REGION Network 63: CONTADOR DE SEGURIDAD DE PRESENCIA - CNTSeg_pHsMx
   RUNG wire#powerrail
      #CNTSeg_pHsMx(IN := wire#w4, R := wire#w7, PV := #V_CNTSeg_pHsMx, BaseUnidades_ms := "CTE_BaseUnidades_1ms", QU =>, QD =>, CVU =>, CVD =>)
   END_RUNG
   RUNG wire#powerrail
      Contact( #Mx_ET10 )
      wire#w1
      Contact( #MAnt_DescargaAct )
      wire#w3
      Contact( #Avance_TR1 )
   END_RUNG wire#w4
   RUNG wire#powerrail
      Contact( #Mx_ET16 )
      wire#w2
      Contact( "ON" )
   END_RUNG wire#w1
   RUNG wire#powerrail
      Contact( #Mx_ET17 )
   END_RUNG wire#w2
   RUNG wire#powerrail
      Contact( #Mx_ET02 )
   END_RUNG wire#w2
   RUNG wire#powerrail
      Contact( #Mx_ET11 )
   END_RUNG wire#w3
   RUNG wire#powerrail
      Contact( #Mx_ET12 )
   END_RUNG wire#w3
   RUNG wire#powerrail
      I_Contact( #Mx_ET10 )
      wire#w5
      I_Contact( #Mx_ET11 )
      I_Contact( #Mx_ET12 )
      wire#w6
      I_Contact( #Mx_ET16 )
      I_Contact( #Mx_ET17 )
      I_Contact( #Mx_ET02 )
   END_RUNG wire#w7
   RUNG wire#powerrail
      I_Contact( #MAnt_DescargaAct )
   END_RUNG wire#w5
   RUNG wire#w6
      I_Contact( #MAnt_DescargaAct )
   END_RUNG wire#w7
   // the same network as SCL:
   #CNTSeg_pHsMx(IN := (((#Mx_ET10 OR ((#Mx_ET16 OR #Mx_ET17 OR #Mx_ET02) AND "ON")) AND #MAnt_DescargaAct) OR #Mx_ET11 OR #Mx_ET12) AND #Avance_TR1,   // "FB910_CNT_UHS"
                 R := (NOT #Mx_ET10 OR NOT #MAnt_DescargaAct) AND NOT #Mx_ET11 AND NOT #Mx_ET12 AND ((NOT #Mx_ET16 AND NOT #Mx_ET17 AND NOT #Mx_ET02) OR NOT #MAnt_DescargaAct),
                 PV := #V_CNTSeg_pHsMx,
                 BaseUnidades_ms := "CTE_BaseUnidades_1ms");
END_REGION

REGION Network 64: CONTADOR DE PRESENCIA - CNT_pHsMx
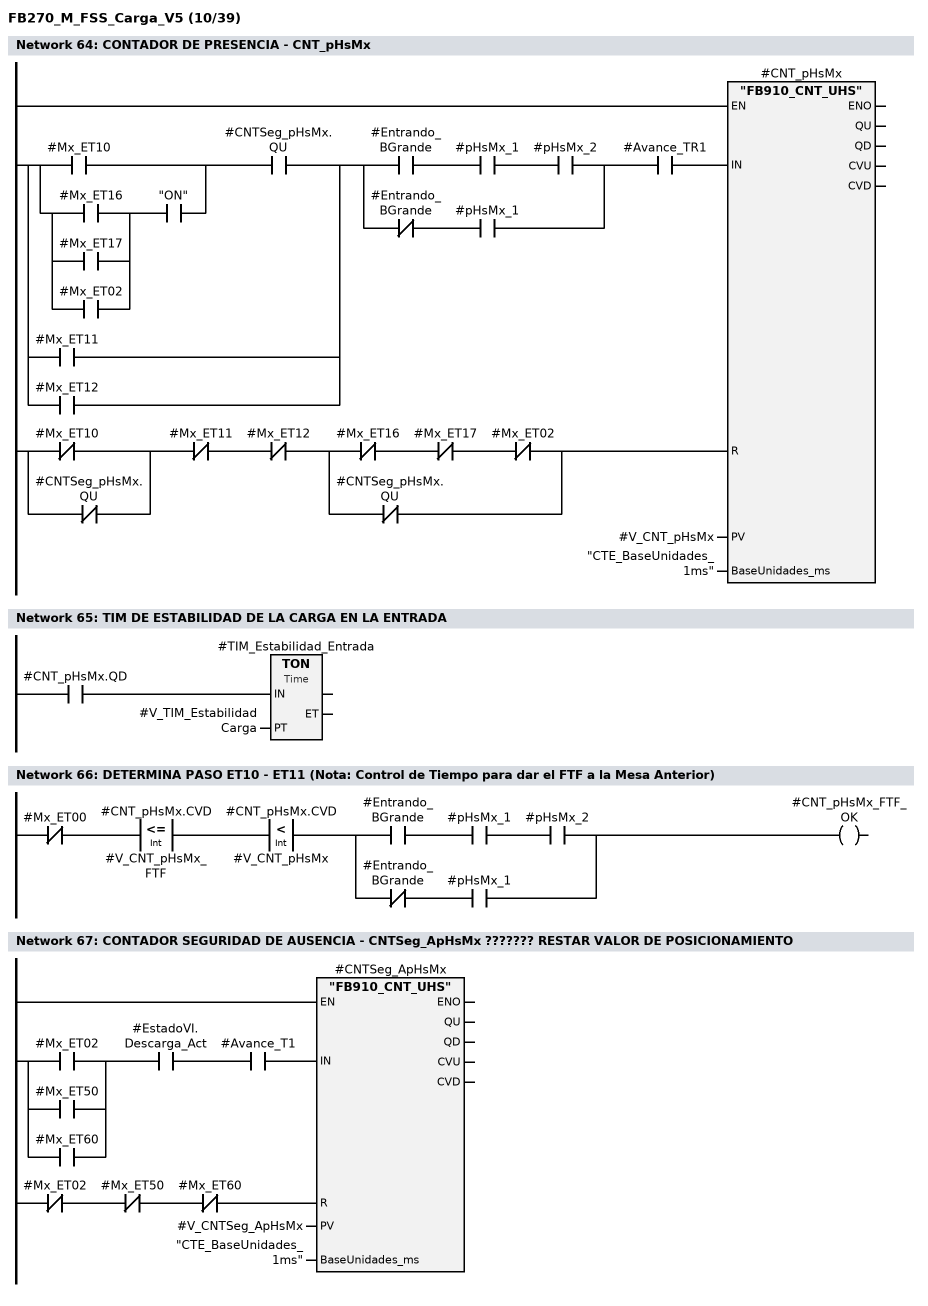
   RUNG wire#powerrail
      #CNT_pHsMx(IN := wire#w5, R := wire#w8, PV := #V_CNT_pHsMx, BaseUnidades_ms := "CTE_BaseUnidades_1ms", QU =>, QD =>, CVU =>, CVD =>)
   END_RUNG
   RUNG wire#powerrail
      Contact( #Mx_ET10 )
      wire#w1
      Contact( #CNTSeg_pHsMx.QU )
      wire#w3
      Contact( #Entrando_BGrande )
      Contact( #pHsMx_1 )
      Contact( #pHsMx_2 )
      wire#w4
      Contact( #Avance_TR1 )
   END_RUNG wire#w5
   RUNG wire#powerrail
      Contact( #Mx_ET16 )
      wire#w2
      Contact( "ON" )
   END_RUNG wire#w1
   RUNG wire#powerrail
      Contact( #Mx_ET17 )
   END_RUNG wire#w2
   RUNG wire#powerrail
      Contact( #Mx_ET02 )
   END_RUNG wire#w2
   RUNG wire#powerrail
      Contact( #Mx_ET11 )
   END_RUNG wire#w3
   RUNG wire#powerrail
      Contact( #Mx_ET12 )
   END_RUNG wire#w3
   RUNG wire#w3
      I_Contact( #Entrando_BGrande )
      Contact( #pHsMx_1 )
   END_RUNG wire#w4
   RUNG wire#powerrail
      I_Contact( #Mx_ET10 )
      wire#w6
      I_Contact( #Mx_ET11 )
      I_Contact( #Mx_ET12 )
      wire#w7
      I_Contact( #Mx_ET16 )
      I_Contact( #Mx_ET17 )
      I_Contact( #Mx_ET02 )
   END_RUNG wire#w8
   RUNG wire#powerrail
      I_Contact( #CNTSeg_pHsMx.QU )
   END_RUNG wire#w6
   RUNG wire#w7
      I_Contact( #CNTSeg_pHsMx.QU )
   END_RUNG wire#w8
   // the same network as SCL:
   #CNT_pHsMx(IN := (((#Mx_ET10 OR ((#Mx_ET16 OR #Mx_ET17 OR #Mx_ET02) AND "ON")) AND #CNTSeg_pHsMx.QU) OR #Mx_ET11 OR #Mx_ET12) AND ((#Entrando_BGrande AND #pHsMx_1 AND #pHsMx_2) OR (NOT #Entrando_BGrande AND #pHsMx_1)) AND #Avance_TR1,   // "FB910_CNT_UHS"
              R := (NOT #Mx_ET10 OR NOT #CNTSeg_pHsMx.QU) AND NOT #Mx_ET11 AND NOT #Mx_ET12 AND ((NOT #Mx_ET16 AND NOT #Mx_ET17 AND NOT #Mx_ET02) OR NOT #CNTSeg_pHsMx.QU),
              PV := #V_CNT_pHsMx,
              BaseUnidades_ms := "CTE_BaseUnidades_1ms");
END_REGION

REGION Network 65: TIM DE ESTABILIDAD DE LA CARGA EN LA ENTRADA
   RUNG wire#powerrail
      Contact( #CNT_pHsMx.QD )
      { S7_Templates := "time_type := Time" } #TIM_Estabilidad_Entrada.TON(pt := #V_TIM_EstabilidadCarga, et =>)
   END_RUNG
   // the same network as SCL:
   #TIM_Estabilidad_Entrada(IN := #CNT_pHsMx.QD, PT := #V_TIM_EstabilidadCarga);   // TON
END_REGION

REGION Network 66: DETERMINA PASO ET10 - ET11 (Nota: Control de Tiempo para dar el FTF a la Mesa Anterior)
   RUNG wire#powerrail
      I_Contact( #Mx_ET00 )
      { S7_Templates := "SrcType := Int" } LE_Contact(in1 := #CNT_pHsMx.CVD, in2 := #V_CNT_pHsMx_FTF)
      { S7_Templates := "SrcType := Int" } LT_Contact(in1 := #CNT_pHsMx.CVD, in2 := #V_CNT_pHsMx)
      wire#w1
      Contact( #Entrando_BGrande )
      Contact( #pHsMx_1 )
      Contact( #pHsMx_2 )
      wire#w2
      Coil( #CNT_pHsMx_FTF_OK )
   END_RUNG
   RUNG wire#w1
      I_Contact( #Entrando_BGrande )
      Contact( #pHsMx_1 )
   END_RUNG wire#w2
   // the same network as SCL:
   #CNT_pHsMx_FTF_OK := NOT #Mx_ET00 AND (#CNT_pHsMx.CVD <= #V_CNT_pHsMx_FTF) AND (#CNT_pHsMx.CVD < #V_CNT_pHsMx) AND ((#Entrando_BGrande AND #pHsMx_1 AND #pHsMx_2) OR (NOT #Entrando_BGrande AND #pHsMx_1));
END_REGION

REGION Network 67: CONTADOR SEGURIDAD DE AUSENCIA - CNTSeg_ApHsMx ??????? RESTAR VALOR DE POSICIONAMIENTO
   RUNG wire#powerrail
      #CNTSeg_ApHsMx(IN := wire#w2, R := wire#w3, PV := #V_CNTSeg_ApHsMx, BaseUnidades_ms := "CTE_BaseUnidades_1ms", QU =>, QD =>, CVU =>, CVD =>)
   END_RUNG
   RUNG wire#powerrail
      Contact( #Mx_ET02 )
      wire#w1
      Contact( #EstadoVI.Descarga_Act )
      Contact( #Avance_T1 )
   END_RUNG wire#w2
   RUNG wire#powerrail
      Contact( #Mx_ET50 )
   END_RUNG wire#w1
   RUNG wire#powerrail
      Contact( #Mx_ET60 )
   END_RUNG wire#w1
   RUNG wire#powerrail
      I_Contact( #Mx_ET02 )
      I_Contact( #Mx_ET50 )
      I_Contact( #Mx_ET60 )
   END_RUNG wire#w3
   // the same network as SCL:
   #CNTSeg_ApHsMx(IN := (#Mx_ET02 OR #Mx_ET50 OR #Mx_ET60) AND #EstadoVI.Descarga_Act AND #Avance_T1,   // "FB910_CNT_UHS"
                  R := NOT #Mx_ET02 AND NOT #Mx_ET50 AND NOT #Mx_ET60,
                  PV := #V_CNTSeg_ApHsMx,
                  BaseUnidades_ms := "CTE_BaseUnidades_1ms");
END_REGION

REGION Network 68: CONTADOR DE LA AUSENCIA - CNT_ApHsMX
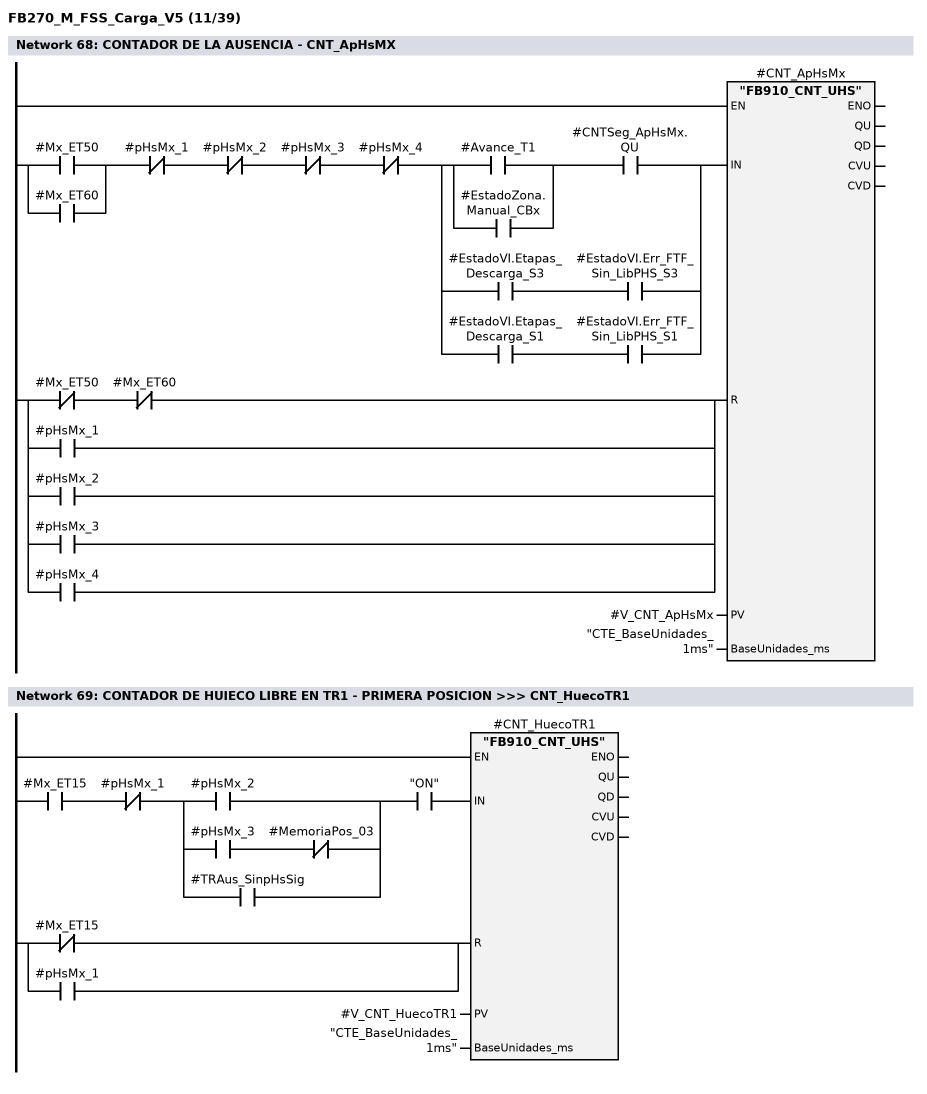
   RUNG wire#powerrail
      #CNT_ApHsMx(IN := wire#w4, R := wire#w5, PV := #V_CNT_ApHsMx, BaseUnidades_ms := "CTE_BaseUnidades_1ms", QU =>, QD =>, CVU =>, CVD =>)
   END_RUNG
   RUNG wire#powerrail
      Contact( #Mx_ET50 )
      wire#w1
      I_Contact( #pHsMx_1 )
      I_Contact( #pHsMx_2 )
      I_Contact( #pHsMx_3 )
      I_Contact( #pHsMx_4 )
      wire#w2
      Contact( #Avance_T1 )
      wire#w3
      Contact( #CNTSeg_ApHsMx.QU )
   END_RUNG wire#w4
   RUNG wire#powerrail
      Contact( #Mx_ET60 )
   END_RUNG wire#w1
   RUNG wire#w2
      Contact( #EstadoZona.Manual_CBx )
   END_RUNG wire#w3
   RUNG wire#w2
      Contact( #EstadoVI.Etapas_Descarga_S3 )
      Contact( #EstadoVI.Err_FTF_Sin_LibPHS_S3 )
   END_RUNG wire#w4
   RUNG wire#w2
      Contact( #EstadoVI.Etapas_Descarga_S1 )
      Contact( #EstadoVI.Err_FTF_Sin_LibPHS_S1 )
   END_RUNG wire#w4
   RUNG wire#powerrail
      I_Contact( #Mx_ET50 )
      I_Contact( #Mx_ET60 )
   END_RUNG wire#w5
   RUNG wire#powerrail
      Contact( #pHsMx_1 )
   END_RUNG wire#w5
   RUNG wire#powerrail
      Contact( #pHsMx_2 )
   END_RUNG wire#w5
   RUNG wire#powerrail
      Contact( #pHsMx_3 )
   END_RUNG wire#w5
   RUNG wire#powerrail
      Contact( #pHsMx_4 )
   END_RUNG wire#w5
   // the same network as SCL:
   #CNT_ApHsMx(IN := (#Mx_ET50 OR #Mx_ET60) AND NOT #pHsMx_1 AND NOT #pHsMx_2 AND NOT #pHsMx_3 AND NOT #pHsMx_4 AND (((#Avance_T1 OR #EstadoZona.Manual_CBx) AND #CNTSeg_ApHsMx.QU) OR (#EstadoVI.Etapas_Descarga_S3 AND #EstadoVI.Err_FTF_Sin_LibPHS_S3) OR (#EstadoVI.Etapas_Descarga_S1 AND #EstadoVI.Err_FTF_Sin_LibPHS_S1)),   // "FB910_CNT_UHS"
               R := (NOT #Mx_ET50 AND NOT #Mx_ET60) OR #pHsMx_1 OR #pHsMx_2 OR #pHsMx_3 OR #pHsMx_4,
               PV := #V_CNT_ApHsMx,
               BaseUnidades_ms := "CTE_BaseUnidades_1ms");
END_REGION

REGION Network 69: CONTADOR DE HUIECO LIBRE EN TR1 - PRIMERA POSICION >>> CNT_HuecoTR1
   RUNG wire#powerrail
      #CNT_HuecoTR1(IN := wire#w3, R := wire#w4, PV := #V_CNT_HuecoTR1, BaseUnidades_ms := "CTE_BaseUnidades_1ms", QU =>, QD =>, CVU =>, CVD =>)
   END_RUNG
   RUNG wire#powerrail
      Contact( #Mx_ET15 )
      I_Contact( #pHsMx_1 )
      wire#w1
      Contact( #pHsMx_2 )
      wire#w2
      Contact( "ON" )
   END_RUNG wire#w3
   RUNG wire#w1
      Contact( #pHsMx_3 )
      I_Contact( #MemoriaPos_03 )
   END_RUNG wire#w2
   RUNG wire#w1
      Contact( #TRAus_SinpHsSig )
   END_RUNG wire#w2
   RUNG wire#powerrail
      I_Contact( #Mx_ET15 )
   END_RUNG wire#w4
   RUNG wire#powerrail
      Contact( #pHsMx_1 )
   END_RUNG wire#w4
   // the same network as SCL:
   #CNT_HuecoTR1(IN := #Mx_ET15 AND NOT #pHsMx_1 AND (#pHsMx_2 OR (#pHsMx_3 AND NOT #MemoriaPos_03) OR #TRAus_SinpHsSig) AND "ON",   // "FB910_CNT_UHS"
                 R := NOT #Mx_ET15 OR #pHsMx_1,
                 PV := #V_CNT_HuecoTR1,
                 BaseUnidades_ms := "CTE_BaseUnidades_1ms");
END_REGION

REGION Network 70: CONTADOR DE HUIECO LIBRE EN TR2 - SEGUNDA POSICION >>> CNT_HuecoTR2
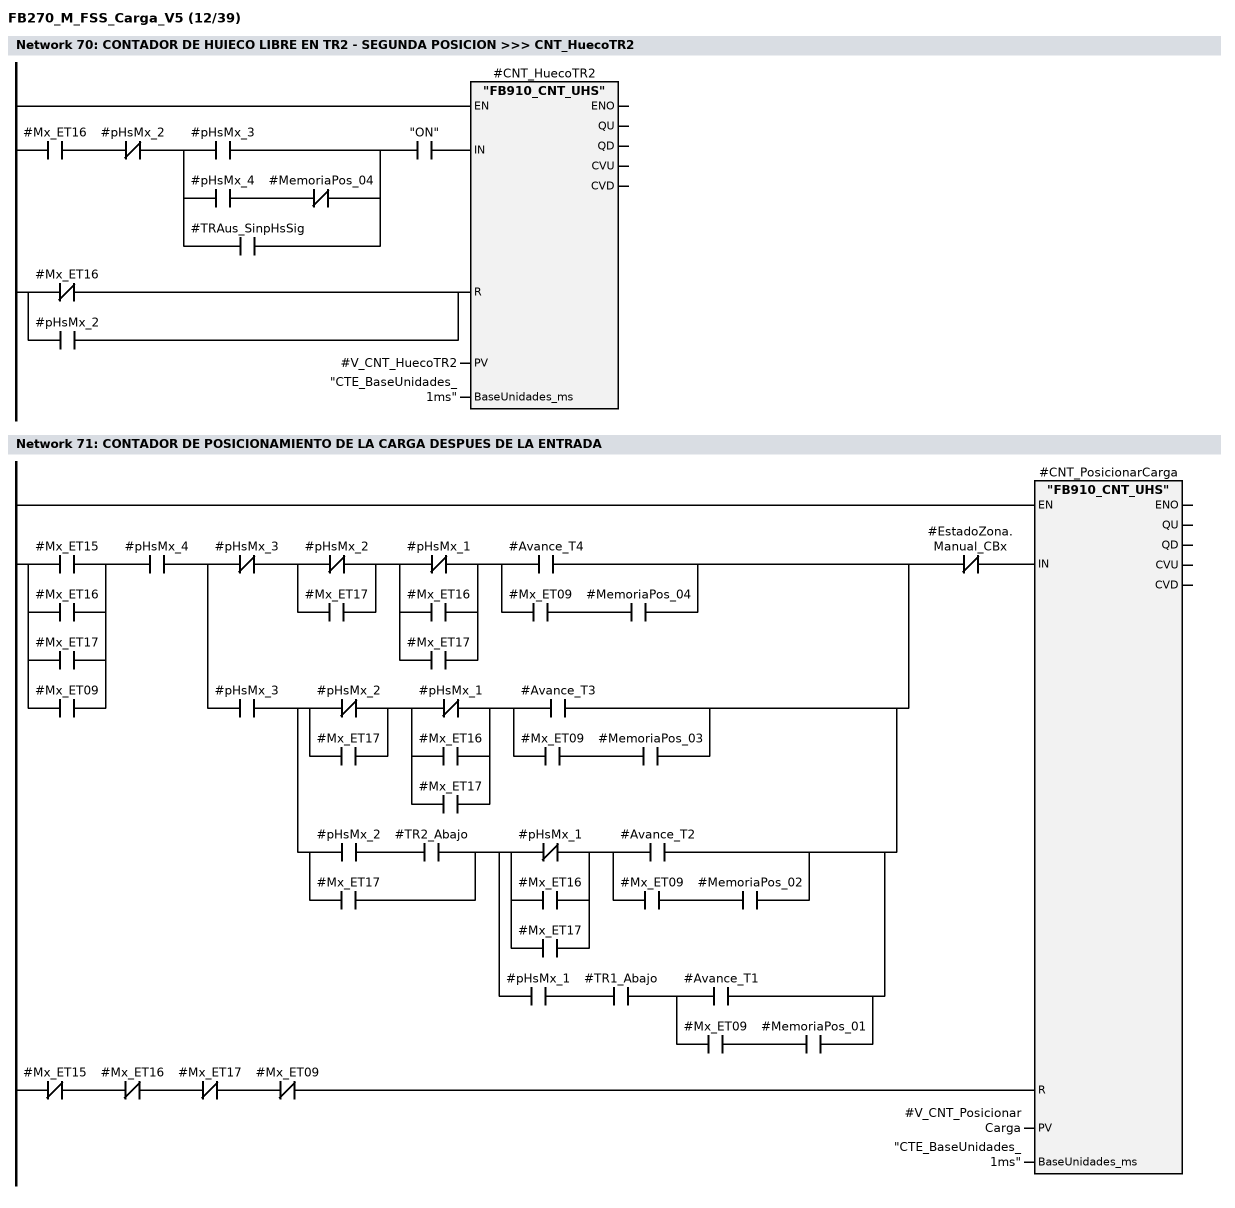
   RUNG wire#powerrail
      #CNT_HuecoTR2(IN := wire#w3, R := wire#w4, PV := #V_CNT_HuecoTR2, BaseUnidades_ms := "CTE_BaseUnidades_1ms", QU =>, QD =>, CVU =>, CVD =>)
   END_RUNG
   RUNG wire#powerrail
      Contact( #Mx_ET16 )
      I_Contact( #pHsMx_2 )
      wire#w1
      Contact( #pHsMx_3 )
      wire#w2
      Contact( "ON" )
   END_RUNG wire#w3
   RUNG wire#w1
      Contact( #pHsMx_4 )
      I_Contact( #MemoriaPos_04 )
   END_RUNG wire#w2
   RUNG wire#w1
      Contact( #TRAus_SinpHsSig )
   END_RUNG wire#w2
   RUNG wire#powerrail
      I_Contact( #Mx_ET16 )
   END_RUNG wire#w4
   RUNG wire#powerrail
      Contact( #pHsMx_2 )
   END_RUNG wire#w4
   // the same network as SCL:
   #CNT_HuecoTR2(IN := #Mx_ET16 AND NOT #pHsMx_2 AND (#pHsMx_3 OR (#pHsMx_4 AND NOT #MemoriaPos_04) OR #TRAus_SinpHsSig) AND "ON",   // "FB910_CNT_UHS"
                 R := NOT #Mx_ET16 OR #pHsMx_2,
                 PV := #V_CNT_HuecoTR2,
                 BaseUnidades_ms := "CTE_BaseUnidades_1ms");
END_REGION

REGION Network 71: CONTADOR DE POSICIONAMIENTO DE LA CARGA DESPUES DE LA ENTRADA
   RUNG wire#powerrail
      #CNT_PosicionarCarga(IN := wire#w13, R := wire#w14, PV := #V_CNT_PosicionarCarga, BaseUnidades_ms := "CTE_BaseUnidades_1ms", QU =>, QD =>, CVU =>, CVD =>)
   END_RUNG
   RUNG wire#powerrail
      Contact( #Mx_ET15 )
      wire#w1
      Contact( #pHsMx_4 )
      wire#w2
      I_Contact( #pHsMx_3 )
      wire#w3
      I_Contact( #pHsMx_2 )
      wire#w4
      I_Contact( #pHsMx_1 )
      wire#w5
      Contact( #Avance_T4 )
      wire#w6
      I_Contact( #EstadoZona.Manual_CBx )
   END_RUNG wire#w13
   RUNG wire#powerrail
      Contact( #Mx_ET16 )
   END_RUNG wire#w1
   RUNG wire#powerrail
      Contact( #Mx_ET17 )
   END_RUNG wire#w1
   RUNG wire#powerrail
      Contact( #Mx_ET09 )
   END_RUNG wire#w1
   RUNG wire#w3
      Contact( #Mx_ET17 )
   END_RUNG wire#w4
   RUNG wire#w4
      Contact( #Mx_ET16 )
   END_RUNG wire#w5
   RUNG wire#w4
      Contact( #Mx_ET17 )
   END_RUNG wire#w5
   RUNG wire#w5
      Contact( #Mx_ET09 )
      Contact( #MemoriaPos_04 )
   END_RUNG wire#w6
   RUNG wire#w2
      Contact( #pHsMx_3 )
      wire#w7
      I_Contact( #pHsMx_2 )
      wire#w8
      I_Contact( #pHsMx_1 )
      wire#w9
      Contact( #Avance_T3 )
   END_RUNG wire#w6
   RUNG wire#w7
      Contact( #Mx_ET17 )
   END_RUNG wire#w8
   RUNG wire#w8
      Contact( #Mx_ET16 )
   END_RUNG wire#w9
   RUNG wire#w8
      Contact( #Mx_ET17 )
   END_RUNG wire#w9
   RUNG wire#w9
      Contact( #Mx_ET09 )
      Contact( #MemoriaPos_03 )
   END_RUNG wire#w6
   RUNG wire#w7
      Contact( #pHsMx_2 )
      Contact( #TR2_Abajo )
      wire#w10
      I_Contact( #pHsMx_1 )
      wire#w11
      Contact( #Avance_T2 )
   END_RUNG wire#w6
   RUNG wire#w7
      Contact( #Mx_ET17 )
   END_RUNG wire#w10
   RUNG wire#w10
      Contact( #Mx_ET16 )
   END_RUNG wire#w11
   RUNG wire#w10
      Contact( #Mx_ET17 )
   END_RUNG wire#w11
   RUNG wire#w11
      Contact( #Mx_ET09 )
      Contact( #MemoriaPos_02 )
   END_RUNG wire#w6
   RUNG wire#w10
      Contact( #pHsMx_1 )
      Contact( #TR1_Abajo )
      wire#w12
      Contact( #Avance_T1 )
   END_RUNG wire#w6
   RUNG wire#w12
      Contact( #Mx_ET09 )
      Contact( #MemoriaPos_01 )
   END_RUNG wire#w6
   RUNG wire#powerrail
      I_Contact( #Mx_ET15 )
      I_Contact( #Mx_ET16 )
      I_Contact( #Mx_ET17 )
      I_Contact( #Mx_ET09 )
   END_RUNG wire#w14
   // the same network as SCL:
   #CNT_PosicionarCarga(IN := (#Mx_ET15 OR #Mx_ET16 OR #Mx_ET17 OR #Mx_ET09) AND #pHsMx_4 AND ((NOT #pHsMx_3 AND (NOT #pHsMx_2 OR #Mx_ET17) AND (NOT #pHsMx_1 OR #Mx_ET16 OR #Mx_ET17) AND (#Avance_T4 OR (#Mx_ET09 AND #MemoriaPos_04))) OR (#pHsMx_3 AND (((NOT #pHsMx_2 OR #Mx_ET17) AND (NOT #pHsMx_1 OR #Mx_ET16 OR #Mx_ET17) AND (#Avance_T3 OR (#Mx_ET09 AND #MemoriaPos_03))) OR (((#pHsMx_2 AND #TR2_Abajo) OR #Mx_ET17) AND (((NOT #pHsMx_1 OR #Mx_ET16 OR #Mx_ET17) AND (#Avance_T2 OR (#Mx_ET09 AND #MemoriaPos_02))) OR (#pHsMx_1 AND #TR1_Abajo AND (#Avance_T1 OR (#Mx_ET09 AND #MemoriaPos_01)))))))) AND NOT #EstadoZona.Manual_CBx,   // "FB910_CNT_UHS"
                        R := NOT #Mx_ET15 AND NOT #Mx_ET16 AND NOT #Mx_ET17 AND NOT #Mx_ET09,
                        PV := #V_CNT_PosicionarCarga,
                        BaseUnidades_ms := "CTE_BaseUnidades_1ms");
END_REGION

REGION Network 72: CONTADOR DE PREPARACION DE CARGA PARA SALIDA POR S1
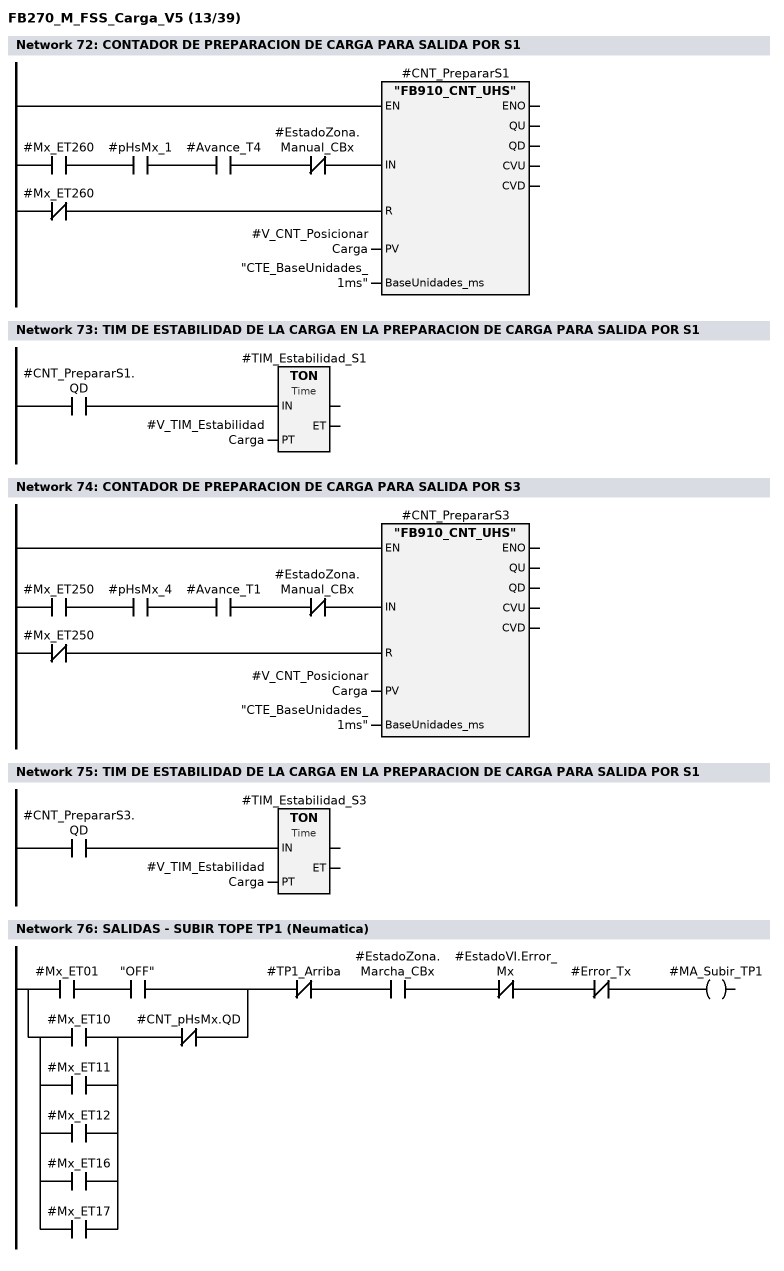
   RUNG wire#powerrail
      #CNT_PrepararS1(IN := wire#w1, R := wire#w2, PV := #V_CNT_PosicionarCarga, BaseUnidades_ms := "CTE_BaseUnidades_1ms", QU =>, QD =>, CVU =>, CVD =>)
   END_RUNG
   RUNG wire#powerrail
      Contact( #Mx_ET260 )
      Contact( #pHsMx_1 )
      Contact( #Avance_T4 )
      I_Contact( #EstadoZona.Manual_CBx )
   END_RUNG wire#w1
   RUNG wire#powerrail
      I_Contact( #Mx_ET260 )
   END_RUNG wire#w2
   // the same network as SCL:
   #CNT_PrepararS1(IN := #Mx_ET260 AND #pHsMx_1 AND #Avance_T4 AND NOT #EstadoZona.Manual_CBx,   // "FB910_CNT_UHS"
                   R := NOT #Mx_ET260,
                   PV := #V_CNT_PosicionarCarga,
                   BaseUnidades_ms := "CTE_BaseUnidades_1ms");
END_REGION

REGION Network 73: TIM DE ESTABILIDAD DE LA CARGA EN LA PREPARACION DE CARGA PARA SALIDA POR S1
   RUNG wire#powerrail
      Contact( #CNT_PrepararS1.QD )
      { S7_Templates := "time_type := Time" } #TIM_Estabilidad_S1.TON(pt := #V_TIM_EstabilidadCarga, et =>)
   END_RUNG
   // the same network as SCL:
   #TIM_Estabilidad_S1(IN := #CNT_PrepararS1.QD, PT := #V_TIM_EstabilidadCarga);   // TON
END_REGION

REGION Network 74: CONTADOR DE PREPARACION DE CARGA PARA SALIDA POR S3
   RUNG wire#powerrail
      #CNT_PrepararS3(IN := wire#w1, R := wire#w2, PV := #V_CNT_PosicionarCarga, BaseUnidades_ms := "CTE_BaseUnidades_1ms", QU =>, QD =>, CVU =>, CVD =>)
   END_RUNG
   RUNG wire#powerrail
      Contact( #Mx_ET250 )
      Contact( #pHsMx_4 )
      Contact( #Avance_T1 )
      I_Contact( #EstadoZona.Manual_CBx )
   END_RUNG wire#w1
   RUNG wire#powerrail
      I_Contact( #Mx_ET250 )
   END_RUNG wire#w2
   // the same network as SCL:
   #CNT_PrepararS3(IN := #Mx_ET250 AND #pHsMx_4 AND #Avance_T1 AND NOT #EstadoZona.Manual_CBx,   // "FB910_CNT_UHS"
                   R := NOT #Mx_ET250,
                   PV := #V_CNT_PosicionarCarga,
                   BaseUnidades_ms := "CTE_BaseUnidades_1ms");
END_REGION

REGION Network 75: TIM DE ESTABILIDAD DE LA CARGA EN LA PREPARACION DE CARGA PARA SALIDA POR S1
   RUNG wire#powerrail
      Contact( #CNT_PrepararS3.QD )
      { S7_Templates := "time_type := Time" } #TIM_Estabilidad_S3.TON(pt := #V_TIM_EstabilidadCarga, et =>)
   END_RUNG
   // the same network as SCL:
   #TIM_Estabilidad_S3(IN := #CNT_PrepararS3.QD, PT := #V_TIM_EstabilidadCarga);   // TON
END_REGION

REGION Network 76: SALIDAS - SUBIR TOPE TP1 (Neumatica)
   RUNG wire#powerrail
      Contact( #Mx_ET01 )
      Contact( "OFF" )
      wire#w1
      I_Contact( #TP1_Arriba )
      Contact( #EstadoZona.Marcha_CBx )
      I_Contact( #EstadoVI.Error_Mx )
      I_Contact( #Error_Tx )
      Coil( #MA_Subir_TP1 )
   END_RUNG
   RUNG wire#powerrail
      Contact( #Mx_ET10 )
      wire#w2
      I_Contact( #CNT_pHsMx.QD )
   END_RUNG wire#w1
   RUNG wire#powerrail
      Contact( #Mx_ET11 )
   END_RUNG wire#w2
   RUNG wire#powerrail
      Contact( #Mx_ET12 )
   END_RUNG wire#w2
   RUNG wire#powerrail
      Contact( #Mx_ET16 )
   END_RUNG wire#w2
   RUNG wire#powerrail
      Contact( #Mx_ET17 )
   END_RUNG wire#w2
   // the same network as SCL:
   #MA_Subir_TP1 := ((#Mx_ET01 AND "OFF") OR ((#Mx_ET10 OR #Mx_ET11 OR #Mx_ET12 OR #Mx_ET16 OR #Mx_ET17) AND NOT #CNT_pHsMx.QD)) AND NOT #TP1_Arriba AND #EstadoZona.Marcha_CBx AND NOT #EstadoVI.Error_Mx AND NOT #Error_Tx;
END_REGION

REGION Network 77: SALIDAS - BAJAR TOPE TP1 (Neumatica)
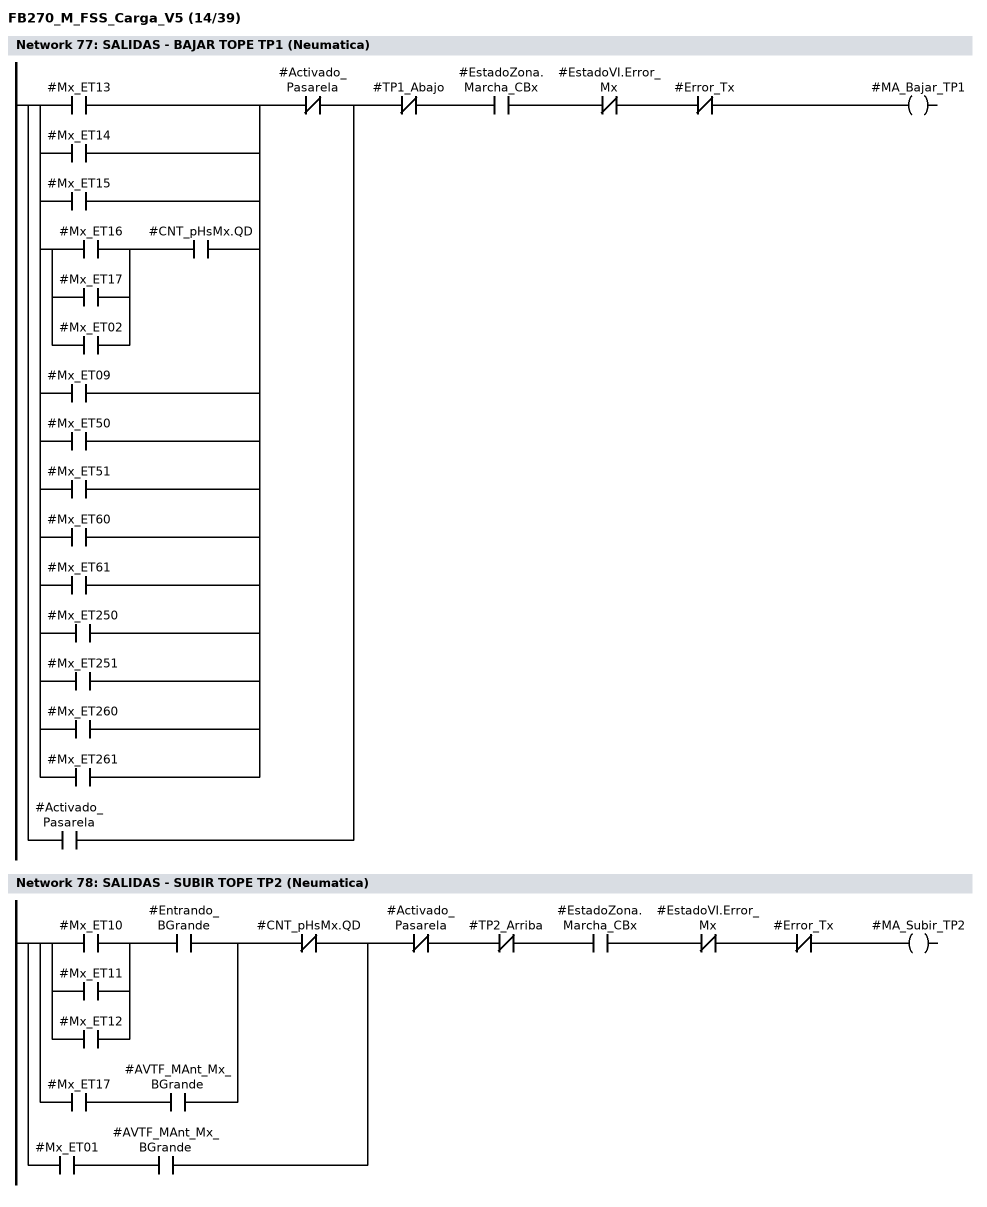
   RUNG wire#powerrail
      Contact( #Mx_ET13 )
      wire#w1
      I_Contact( #Activado_Pasarela )
      wire#w3
      I_Contact( #TP1_Abajo )
      Contact( #EstadoZona.Marcha_CBx )
      I_Contact( #EstadoVI.Error_Mx )
      I_Contact( #Error_Tx )
      Coil( #MA_Bajar_TP1 )
   END_RUNG
   RUNG wire#powerrail
      Contact( #Mx_ET14 )
   END_RUNG wire#w1
   RUNG wire#powerrail
      Contact( #Mx_ET15 )
   END_RUNG wire#w1
   RUNG wire#powerrail
      Contact( #Mx_ET16 )
      wire#w2
      Contact( #CNT_pHsMx.QD )
   END_RUNG wire#w1
   RUNG wire#powerrail
      Contact( #Mx_ET17 )
   END_RUNG wire#w2
   RUNG wire#powerrail
      Contact( #Mx_ET02 )
   END_RUNG wire#w2
   RUNG wire#powerrail
      Contact( #Mx_ET09 )
   END_RUNG wire#w1
   RUNG wire#powerrail
      Contact( #Mx_ET50 )
   END_RUNG wire#w1
   RUNG wire#powerrail
      Contact( #Mx_ET51 )
   END_RUNG wire#w1
   RUNG wire#powerrail
      Contact( #Mx_ET60 )
   END_RUNG wire#w1
   RUNG wire#powerrail
      Contact( #Mx_ET61 )
   END_RUNG wire#w1
   RUNG wire#powerrail
      Contact( #Mx_ET250 )
   END_RUNG wire#w1
   RUNG wire#powerrail
      Contact( #Mx_ET251 )
   END_RUNG wire#w1
   RUNG wire#powerrail
      Contact( #Mx_ET260 )
   END_RUNG wire#w1
   RUNG wire#powerrail
      Contact( #Mx_ET261 )
   END_RUNG wire#w1
   RUNG wire#powerrail
      Contact( #Activado_Pasarela )
   END_RUNG wire#w3
   // the same network as SCL:
   #MA_Bajar_TP1 := (((#Mx_ET13 OR #Mx_ET14 OR #Mx_ET15 OR ((#Mx_ET16 OR #Mx_ET17 OR #Mx_ET02) AND #CNT_pHsMx.QD) OR #Mx_ET09 OR #Mx_ET50 OR #Mx_ET51 OR #Mx_ET60 OR #Mx_ET61 OR #Mx_ET250 OR #Mx_ET251 OR #Mx_ET260 OR #Mx_ET261) AND NOT #Activado_Pasarela) OR #Activado_Pasarela) AND NOT #TP1_Abajo AND #EstadoZona.Marcha_CBx AND NOT #EstadoVI.Error_Mx AND NOT #Error_Tx;
END_REGION

REGION Network 78: SALIDAS - SUBIR TOPE TP2 (Neumatica)
   RUNG wire#powerrail
      Contact( #Mx_ET10 )
      wire#w1
      Contact( #Entrando_BGrande )
      wire#w2
      I_Contact( #CNT_pHsMx.QD )
      wire#w3
      I_Contact( #Activado_Pasarela )
      I_Contact( #TP2_Arriba )
      Contact( #EstadoZona.Marcha_CBx )
      I_Contact( #EstadoVI.Error_Mx )
      I_Contact( #Error_Tx )
      Coil( #MA_Subir_TP2 )
   END_RUNG
   RUNG wire#powerrail
      Contact( #Mx_ET11 )
   END_RUNG wire#w1
   RUNG wire#powerrail
      Contact( #Mx_ET12 )
   END_RUNG wire#w1
   RUNG wire#powerrail
      Contact( #Mx_ET17 )
      Contact( #AVTF_MAnt_Mx_BGrande )
   END_RUNG wire#w2
   RUNG wire#powerrail
      Contact( #Mx_ET01 )
      Contact( #AVTF_MAnt_Mx_BGrande )
   END_RUNG wire#w3
   // the same network as SCL:
   #MA_Subir_TP2 := (((((#Mx_ET10 OR #Mx_ET11 OR #Mx_ET12) AND #Entrando_BGrande) OR (#Mx_ET17 AND #AVTF_MAnt_Mx_BGrande)) AND NOT #CNT_pHsMx.QD) OR (#Mx_ET01 AND #AVTF_MAnt_Mx_BGrande)) AND NOT #Activado_Pasarela AND NOT #TP2_Arriba AND #EstadoZona.Marcha_CBx AND NOT #EstadoVI.Error_Mx AND NOT #Error_Tx;
END_REGION

REGION Network 79: SALIDAS - BAJAR TOPE TP2 (Neumatica)
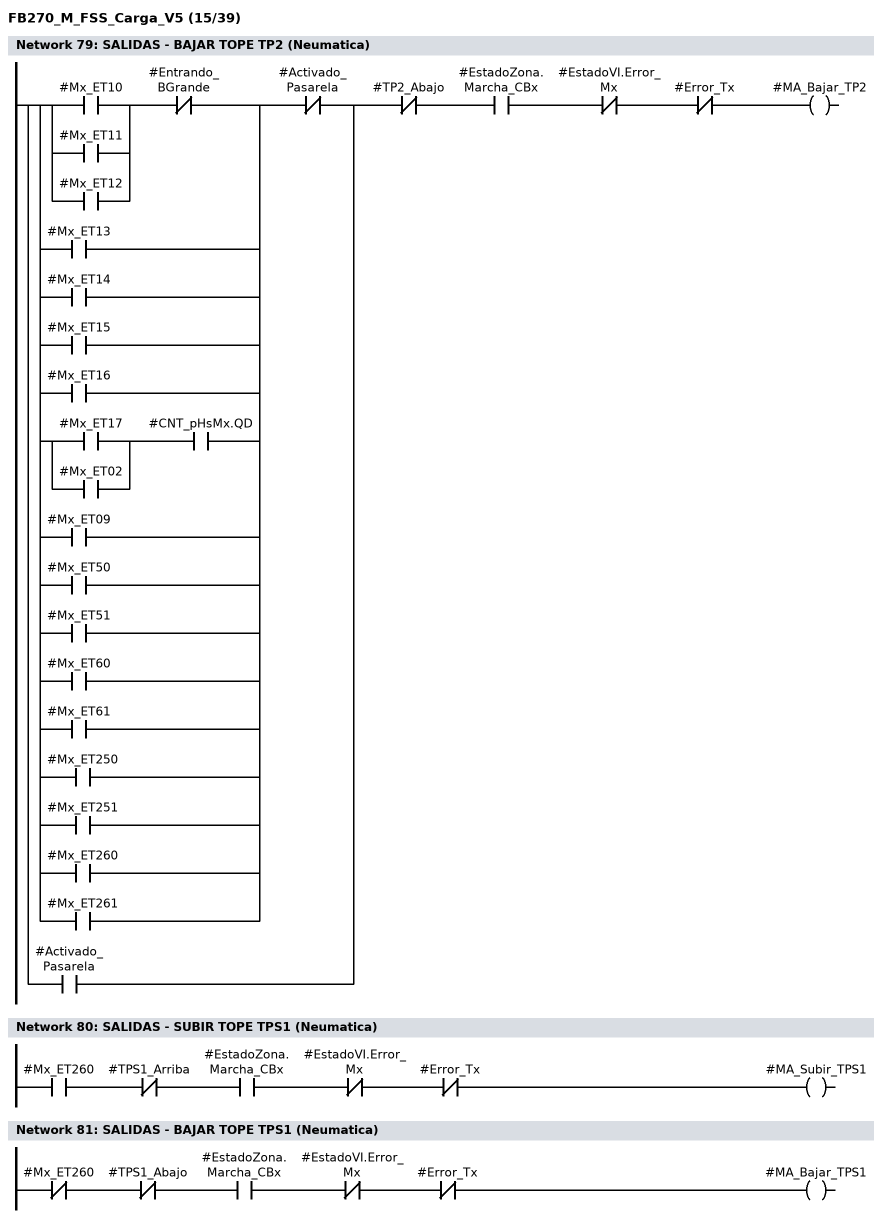
   RUNG wire#powerrail
      Contact( #Mx_ET10 )
      wire#w1
      I_Contact( #Entrando_BGrande )
      wire#w2
      I_Contact( #Activado_Pasarela )
      wire#w4
      I_Contact( #TP2_Abajo )
      Contact( #EstadoZona.Marcha_CBx )
      I_Contact( #EstadoVI.Error_Mx )
      I_Contact( #Error_Tx )
      Coil( #MA_Bajar_TP2 )
   END_RUNG
   RUNG wire#powerrail
      Contact( #Mx_ET11 )
   END_RUNG wire#w1
   RUNG wire#powerrail
      Contact( #Mx_ET12 )
   END_RUNG wire#w1
   RUNG wire#powerrail
      Contact( #Mx_ET13 )
   END_RUNG wire#w2
   RUNG wire#powerrail
      Contact( #Mx_ET14 )
   END_RUNG wire#w2
   RUNG wire#powerrail
      Contact( #Mx_ET15 )
   END_RUNG wire#w2
   RUNG wire#powerrail
      Contact( #Mx_ET16 )
   END_RUNG wire#w2
   RUNG wire#powerrail
      Contact( #Mx_ET17 )
      wire#w3
      Contact( #CNT_pHsMx.QD )
   END_RUNG wire#w2
   RUNG wire#powerrail
      Contact( #Mx_ET02 )
   END_RUNG wire#w3
   RUNG wire#powerrail
      Contact( #Mx_ET09 )
   END_RUNG wire#w2
   RUNG wire#powerrail
      Contact( #Mx_ET50 )
   END_RUNG wire#w2
   RUNG wire#powerrail
      Contact( #Mx_ET51 )
   END_RUNG wire#w2
   RUNG wire#powerrail
      Contact( #Mx_ET60 )
   END_RUNG wire#w2
   RUNG wire#powerrail
      Contact( #Mx_ET61 )
   END_RUNG wire#w2
   RUNG wire#powerrail
      Contact( #Mx_ET250 )
   END_RUNG wire#w2
   RUNG wire#powerrail
      Contact( #Mx_ET251 )
   END_RUNG wire#w2
   RUNG wire#powerrail
      Contact( #Mx_ET260 )
   END_RUNG wire#w2
   RUNG wire#powerrail
      Contact( #Mx_ET261 )
   END_RUNG wire#w2
   RUNG wire#powerrail
      Contact( #Activado_Pasarela )
   END_RUNG wire#w4
   // the same network as SCL:
   #MA_Bajar_TP2 := (((((#Mx_ET10 OR #Mx_ET11 OR #Mx_ET12) AND NOT #Entrando_BGrande) OR #Mx_ET13 OR #Mx_ET14 OR #Mx_ET15 OR #Mx_ET16 OR ((#Mx_ET17 OR #Mx_ET02) AND #CNT_pHsMx.QD) OR #Mx_ET09 OR #Mx_ET50 OR #Mx_ET51 OR #Mx_ET60 OR #Mx_ET61 OR #Mx_ET250 OR #Mx_ET251 OR #Mx_ET260 OR #Mx_ET261) AND NOT #Activado_Pasarela) OR #Activado_Pasarela) AND NOT #TP2_Abajo AND #EstadoZona.Marcha_CBx AND NOT #EstadoVI.Error_Mx AND NOT #Error_Tx;
END_REGION

REGION Network 80: SALIDAS - SUBIR TOPE TPS1 (Neumatica)
   RUNG wire#powerrail
      Contact( #Mx_ET260 )
      I_Contact( #TPS1_Arriba )
      Contact( #EstadoZona.Marcha_CBx )
      I_Contact( #EstadoVI.Error_Mx )
      I_Contact( #Error_Tx )
      Coil( #MA_Subir_TPS1 )
   END_RUNG
   // the same network as SCL:
   #MA_Subir_TPS1 := #Mx_ET260 AND NOT #TPS1_Arriba AND #EstadoZona.Marcha_CBx AND NOT #EstadoVI.Error_Mx AND NOT #Error_Tx;
END_REGION

REGION Network 81: SALIDAS - BAJAR TOPE TPS1 (Neumatica)
   RUNG wire#powerrail
      I_Contact( #Mx_ET260 )
      I_Contact( #TPS1_Abajo )
      Contact( #EstadoZona.Marcha_CBx )
      I_Contact( #EstadoVI.Error_Mx )
      I_Contact( #Error_Tx )
      Coil( #MA_Bajar_TPS1 )
   END_RUNG
   // the same network as SCL:
   #MA_Bajar_TPS1 := NOT #Mx_ET260 AND NOT #TPS1_Abajo AND #EstadoZona.Marcha_CBx AND NOT #EstadoVI.Error_Mx AND NOT #Error_Tx;
END_REGION

REGION Network 82: SALIDAS - SUBIR TOPE TPS3 (Neumatica)
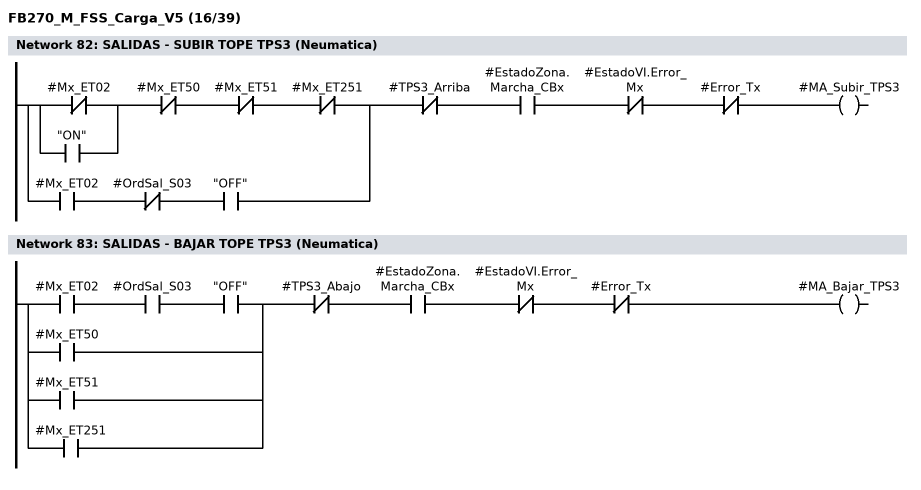
   RUNG wire#powerrail
      I_Contact( #Mx_ET02 )
      wire#w1
      I_Contact( #Mx_ET50 )
      I_Contact( #Mx_ET51 )
      I_Contact( #Mx_ET251 )
      wire#w2
      I_Contact( #TPS3_Arriba )
      Contact( #EstadoZona.Marcha_CBx )
      I_Contact( #EstadoVI.Error_Mx )
      I_Contact( #Error_Tx )
      Coil( #MA_Subir_TPS3 )
   END_RUNG
   RUNG wire#powerrail
      Contact( "ON" )
   END_RUNG wire#w1
   RUNG wire#powerrail
      Contact( #Mx_ET02 )
      I_Contact( #OrdSal_S03 )
      Contact( "OFF" )
   END_RUNG wire#w2
   // the same network as SCL:
   #MA_Subir_TPS3 := (((NOT #Mx_ET02 OR "ON") AND NOT #Mx_ET50 AND NOT #Mx_ET51 AND NOT #Mx_ET251) OR (#Mx_ET02 AND NOT #OrdSal_S03 AND "OFF")) AND NOT #TPS3_Arriba AND #EstadoZona.Marcha_CBx AND NOT #EstadoVI.Error_Mx AND NOT #Error_Tx;
END_REGION

REGION Network 83: SALIDAS - BAJAR TOPE TPS3 (Neumatica)
   RUNG wire#powerrail
      Contact( #Mx_ET02 )
      Contact( #OrdSal_S03 )
      Contact( "OFF" )
      wire#w1
      I_Contact( #TPS3_Abajo )
      Contact( #EstadoZona.Marcha_CBx )
      I_Contact( #EstadoVI.Error_Mx )
      I_Contact( #Error_Tx )
      Coil( #MA_Bajar_TPS3 )
   END_RUNG
   RUNG wire#powerrail
      Contact( #Mx_ET50 )
   END_RUNG wire#w1
   RUNG wire#powerrail
      Contact( #Mx_ET51 )
   END_RUNG wire#w1
   RUNG wire#powerrail
      Contact( #Mx_ET251 )
   END_RUNG wire#w1
   // the same network as SCL:
   #MA_Bajar_TPS3 := ((#Mx_ET02 AND #OrdSal_S03 AND "OFF") OR #Mx_ET50 OR #Mx_ET51 OR #Mx_ET251) AND NOT #TPS3_Abajo AND #EstadoZona.Marcha_CBx AND NOT #EstadoVI.Error_Mx AND NOT #Error_Tx;
END_REGION

REGION Network 84: VARIABLES AUXILIARES - Posición Correcta de los Transfers
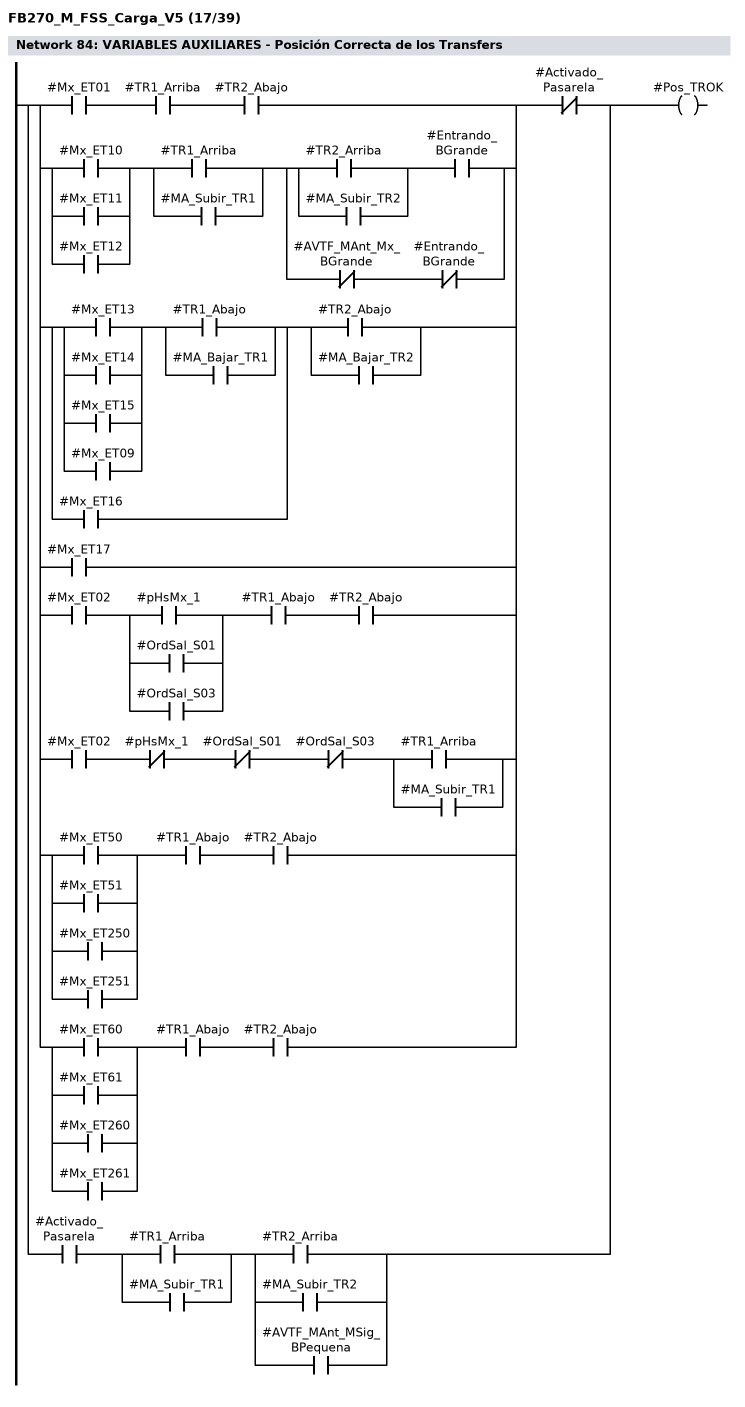
   RUNG wire#powerrail
      Contact( #Mx_ET01 )
      Contact( #TR1_Arriba )
      Contact( #TR2_Abajo )
      wire#w1
      I_Contact( #Activado_Pasarela )
      wire#w12
      Coil( #Pos_TROK )
   END_RUNG
   RUNG wire#powerrail
      Contact( #Mx_ET10 )
      wire#w2
      Contact( #TR1_Arriba )
      wire#w3
      Contact( #TR2_Arriba )
      wire#w4
      Contact( #Entrando_BGrande )
   END_RUNG wire#w1
   RUNG wire#powerrail
      Contact( #Mx_ET11 )
   END_RUNG wire#w2
   RUNG wire#powerrail
      Contact( #Mx_ET12 )
   END_RUNG wire#w2
   RUNG wire#w2
      Contact( #MA_Subir_TR1 )
   END_RUNG wire#w3
   RUNG wire#w3
      Contact( #MA_Subir_TR2 )
   END_RUNG wire#w4
   RUNG wire#w3
      I_Contact( #AVTF_MAnt_Mx_BGrande )
      I_Contact( #Entrando_BGrande )
   END_RUNG wire#w1
   RUNG wire#powerrail
      Contact( #Mx_ET13 )
      wire#w5
      Contact( #TR1_Abajo )
      wire#w6
      Contact( #TR2_Abajo )
   END_RUNG wire#w1
   RUNG wire#powerrail
      Contact( #Mx_ET14 )
   END_RUNG wire#w5
   RUNG wire#powerrail
      Contact( #Mx_ET15 )
   END_RUNG wire#w5
   RUNG wire#powerrail
      Contact( #Mx_ET09 )
   END_RUNG wire#w5
   RUNG wire#w5
      Contact( #MA_Bajar_TR1 )
   END_RUNG wire#w6
   RUNG wire#powerrail
      Contact( #Mx_ET16 )
   END_RUNG wire#w6
   RUNG wire#w6
      Contact( #MA_Bajar_TR2 )
   END_RUNG wire#w1
   RUNG wire#powerrail
      Contact( #Mx_ET17 )
   END_RUNG wire#w1
   RUNG wire#powerrail
      Contact( #Mx_ET02 )
      wire#w7
      Contact( #pHsMx_1 )
      wire#w8
      Contact( #TR1_Abajo )
      Contact( #TR2_Abajo )
   END_RUNG wire#w1
   RUNG wire#w7
      Contact( #OrdSal_S01 )
   END_RUNG wire#w8
   RUNG wire#w7
      Contact( #OrdSal_S03 )
   END_RUNG wire#w8
   RUNG wire#powerrail
      Contact( #Mx_ET02 )
      I_Contact( #pHsMx_1 )
      I_Contact( #OrdSal_S01 )
      I_Contact( #OrdSal_S03 )
      wire#w9
      Contact( #TR1_Arriba )
   END_RUNG wire#w1
   RUNG wire#w9
      Contact( #MA_Subir_TR1 )
   END_RUNG wire#w1
   RUNG wire#powerrail
      Contact( #Mx_ET50 )
      wire#w10
      Contact( #TR1_Abajo )
      Contact( #TR2_Abajo )
   END_RUNG wire#w1
   RUNG wire#powerrail
      Contact( #Mx_ET51 )
   END_RUNG wire#w10
   RUNG wire#powerrail
      Contact( #Mx_ET250 )
   END_RUNG wire#w10
   RUNG wire#powerrail
      Contact( #Mx_ET251 )
   END_RUNG wire#w10
   RUNG wire#powerrail
      Contact( #Mx_ET60 )
      wire#w11
      Contact( #TR1_Abajo )
      Contact( #TR2_Abajo )
   END_RUNG wire#w1
   RUNG wire#powerrail
      Contact( #Mx_ET61 )
   END_RUNG wire#w11
   RUNG wire#powerrail
      Contact( #Mx_ET260 )
   END_RUNG wire#w11
   RUNG wire#powerrail
      Contact( #Mx_ET261 )
   END_RUNG wire#w11
   RUNG wire#powerrail
      Contact( #Activado_Pasarela )
      wire#w13
      Contact( #TR1_Arriba )
      wire#w14
      Contact( #TR2_Arriba )
   END_RUNG wire#w12
   RUNG wire#w13
      Contact( #MA_Subir_TR1 )
   END_RUNG wire#w14
   RUNG wire#w14
      Contact( #MA_Subir_TR2 )
   END_RUNG wire#w12
   RUNG wire#w14
      Contact( #AVTF_MAnt_MSig_BPequena )
   END_RUNG wire#w12
   // the same network as SCL:
   #Pos_TROK := (((#Mx_ET01 AND #TR1_Arriba AND #TR2_Abajo) OR ((#Mx_ET10 OR #Mx_ET11 OR #Mx_ET12) AND (#TR1_Arriba OR #MA_Subir_TR1) AND (((#TR2_Arriba OR #MA_Subir_TR2) AND #Entrando_BGrande) OR (NOT #AVTF_MAnt_Mx_BGrande AND NOT #Entrando_BGrande))) OR ((((#Mx_ET13 OR #Mx_ET14 OR #Mx_ET15 OR #Mx_ET09) AND (#TR1_Abajo OR #MA_Bajar_TR1)) OR #Mx_ET16) AND (#TR2_Abajo OR #MA_Bajar_TR2)) OR #Mx_ET17 OR (#Mx_ET02 AND (#pHsMx_1 OR #OrdSal_S01 OR #OrdSal_S03) AND #TR1_Abajo AND #TR2_Abajo) OR (#Mx_ET02 AND NOT #pHsMx_1 AND NOT #OrdSal_S01 AND NOT #OrdSal_S03 AND (#TR1_Arriba OR #MA_Subir_TR1)) OR ((#Mx_ET50 OR #Mx_ET51 OR #Mx_ET250 OR #Mx_ET251) AND #TR1_Abajo AND #TR2_Abajo) OR ((#Mx_ET60 OR #Mx_ET61 OR #Mx_ET260 OR #Mx_ET261) AND #TR1_Abajo AND #TR2_Abajo)) AND NOT #Activado_Pasarela) OR (#Activado_Pasarela AND (#TR1_Arriba OR #MA_Subir_TR1) AND (#TR2_Arriba OR #MA_Subir_TR2 OR #AVTF_MAnt_MSig_BPequena));
END_REGION

REGION Network 85: VARIABLES AUXILIARES - Posición Correcta de los Topes
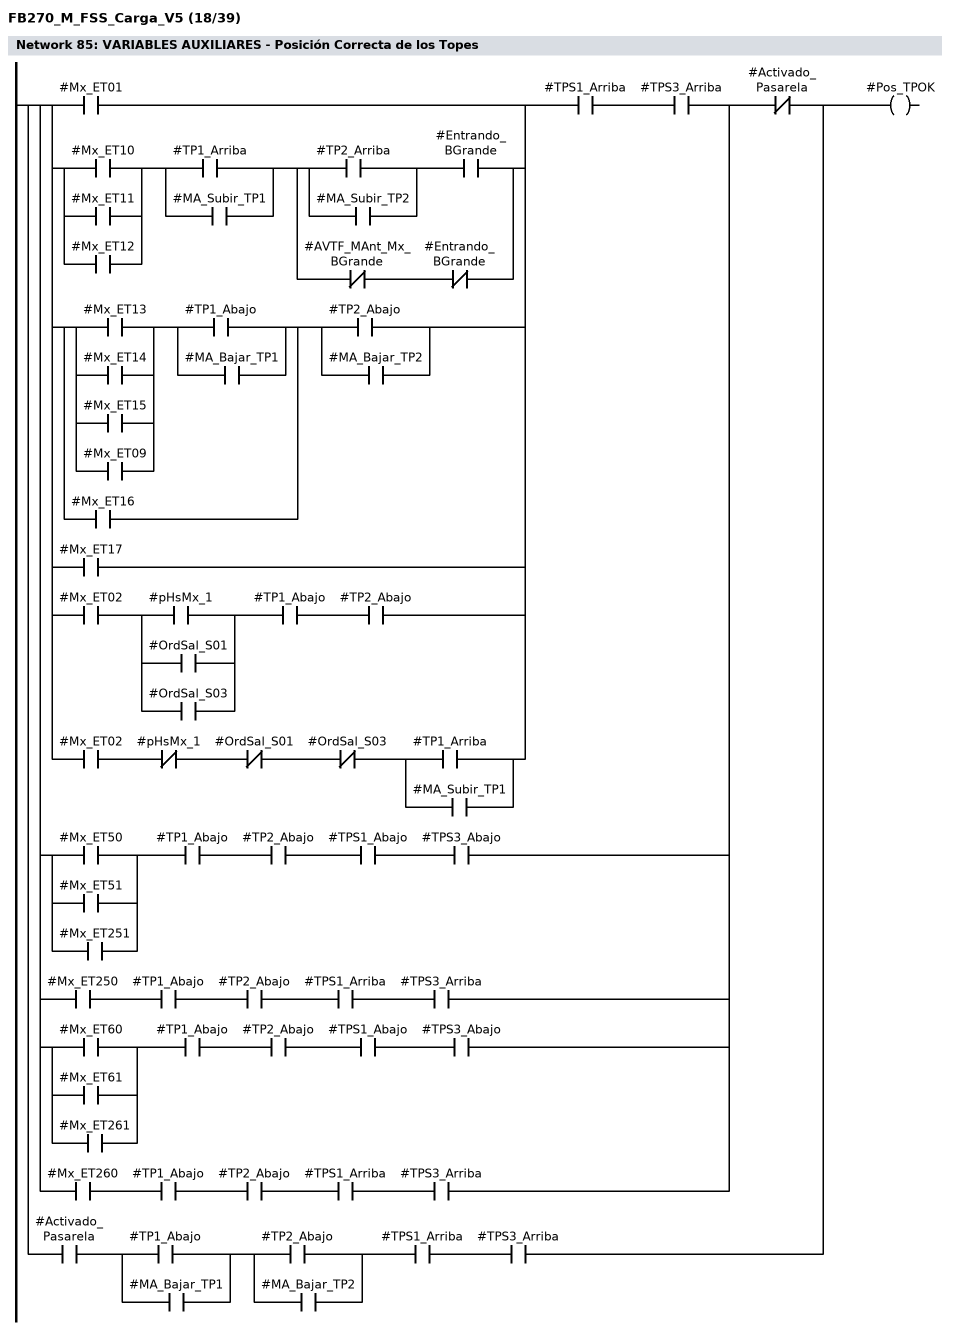
   RUNG wire#powerrail
      Contact( #Mx_ET01 )
      wire#w1
      Contact( #TPS1_Arriba )
      Contact( #TPS3_Arriba )
      wire#w10
      I_Contact( #Activado_Pasarela )
      wire#w13
      Coil( #Pos_TPOK )
   END_RUNG
   RUNG wire#powerrail
      Contact( #Mx_ET10 )
      wire#w2
      Contact( #TP1_Arriba )
      wire#w3
      Contact( #TP2_Arriba )
      wire#w4
      Contact( #Entrando_BGrande )
   END_RUNG wire#w1
   RUNG wire#powerrail
      Contact( #Mx_ET11 )
   END_RUNG wire#w2
   RUNG wire#powerrail
      Contact( #Mx_ET12 )
   END_RUNG wire#w2
   RUNG wire#w2
      Contact( #MA_Subir_TP1 )
   END_RUNG wire#w3
   RUNG wire#w3
      Contact( #MA_Subir_TP2 )
   END_RUNG wire#w4
   RUNG wire#w3
      I_Contact( #AVTF_MAnt_Mx_BGrande )
      I_Contact( #Entrando_BGrande )
   END_RUNG wire#w1
   RUNG wire#powerrail
      Contact( #Mx_ET13 )
      wire#w5
      Contact( #TP1_Abajo )
      wire#w6
      Contact( #TP2_Abajo )
   END_RUNG wire#w1
   RUNG wire#powerrail
      Contact( #Mx_ET14 )
   END_RUNG wire#w5
   RUNG wire#powerrail
      Contact( #Mx_ET15 )
   END_RUNG wire#w5
   RUNG wire#powerrail
      Contact( #Mx_ET09 )
   END_RUNG wire#w5
   RUNG wire#w5
      Contact( #MA_Bajar_TP1 )
   END_RUNG wire#w6
   RUNG wire#powerrail
      Contact( #Mx_ET16 )
   END_RUNG wire#w6
   RUNG wire#w6
      Contact( #MA_Bajar_TP2 )
   END_RUNG wire#w1
   RUNG wire#powerrail
      Contact( #Mx_ET17 )
   END_RUNG wire#w1
   RUNG wire#powerrail
      Contact( #Mx_ET02 )
      wire#w7
      Contact( #pHsMx_1 )
      wire#w8
      Contact( #TP1_Abajo )
      Contact( #TP2_Abajo )
   END_RUNG wire#w1
   RUNG wire#w7
      Contact( #OrdSal_S01 )
   END_RUNG wire#w8
   RUNG wire#w7
      Contact( #OrdSal_S03 )
   END_RUNG wire#w8
   RUNG wire#powerrail
      Contact( #Mx_ET02 )
      I_Contact( #pHsMx_1 )
      I_Contact( #OrdSal_S01 )
      I_Contact( #OrdSal_S03 )
      wire#w9
      Contact( #TP1_Arriba )
   END_RUNG wire#w1
   RUNG wire#w9
      Contact( #MA_Subir_TP1 )
   END_RUNG wire#w1
   RUNG wire#powerrail
      Contact( #Mx_ET50 )
      wire#w11
      Contact( #TP1_Abajo )
      Contact( #TP2_Abajo )
      Contact( #TPS1_Abajo )
      Contact( #TPS3_Abajo )
   END_RUNG wire#w10
   RUNG wire#powerrail
      Contact( #Mx_ET51 )
   END_RUNG wire#w11
   RUNG wire#powerrail
      Contact( #Mx_ET251 )
   END_RUNG wire#w11
   RUNG wire#powerrail
      Contact( #Mx_ET250 )
      Contact( #TP1_Abajo )
      Contact( #TP2_Abajo )
      Contact( #TPS1_Arriba )
      Contact( #TPS3_Arriba )
   END_RUNG wire#w10
   RUNG wire#powerrail
      Contact( #Mx_ET60 )
      wire#w12
      Contact( #TP1_Abajo )
      Contact( #TP2_Abajo )
      Contact( #TPS1_Abajo )
      Contact( #TPS3_Abajo )
   END_RUNG wire#w10
   RUNG wire#powerrail
      Contact( #Mx_ET61 )
   END_RUNG wire#w12
   RUNG wire#powerrail
      Contact( #Mx_ET261 )
   END_RUNG wire#w12
   RUNG wire#powerrail
      Contact( #Mx_ET260 )
      Contact( #TP1_Abajo )
      Contact( #TP2_Abajo )
      Contact( #TPS1_Arriba )
      Contact( #TPS3_Arriba )
   END_RUNG wire#w10
   RUNG wire#powerrail
      Contact( #Activado_Pasarela )
      wire#w14
      Contact( #TP1_Abajo )
      wire#w15
      Contact( #TP2_Abajo )
      wire#w16
      Contact( #TPS1_Arriba )
      Contact( #TPS3_Arriba )
   END_RUNG wire#w13
   RUNG wire#w14
      Contact( #MA_Bajar_TP1 )
   END_RUNG wire#w15
   RUNG wire#w15
      Contact( #MA_Bajar_TP2 )
   END_RUNG wire#w16
   // the same network as SCL:
   #Pos_TPOK := ((((#Mx_ET01 OR ((#Mx_ET10 OR #Mx_ET11 OR #Mx_ET12) AND (#TP1_Arriba OR #MA_Subir_TP1) AND (((#TP2_Arriba OR #MA_Subir_TP2) AND #Entrando_BGrande) OR (NOT #AVTF_MAnt_Mx_BGrande AND NOT #Entrando_BGrande))) OR ((((#Mx_ET13 OR #Mx_ET14 OR #Mx_ET15 OR #Mx_ET09) AND (#TP1_Abajo OR #MA_Bajar_TP1)) OR #Mx_ET16) AND (#TP2_Abajo OR #MA_Bajar_TP2)) OR #Mx_ET17 OR (#Mx_ET02 AND (#pHsMx_1 OR #OrdSal_S01 OR #OrdSal_S03) AND #TP1_Abajo AND #TP2_Abajo) OR (#Mx_ET02 AND NOT #pHsMx_1 AND NOT #OrdSal_S01 AND NOT #OrdSal_S03 AND (#TP1_Arriba OR #MA_Subir_TP1))) AND #TPS1_Arriba AND #TPS3_Arriba) OR ((#Mx_ET50 OR #Mx_ET51 OR #Mx_ET251) AND #TP1_Abajo AND #TP2_Abajo AND #TPS1_Abajo AND #TPS3_Abajo) OR (#Mx_ET250 AND #TP1_Abajo AND #TP2_Abajo AND #TPS1_Arriba AND #TPS3_Arriba) OR ((#Mx_ET60 OR #Mx_ET61 OR #Mx_ET261) AND #TP1_Abajo AND #TP2_Abajo AND #TPS1_Abajo AND #TPS3_Abajo) OR (#Mx_ET260 AND #TP1_Abajo AND #TP2_Abajo AND #TPS1_Arriba AND #TPS3_Arriba)) AND NOT #Activado_Pasarela) OR (#Activado_Pasarela AND (#TP1_Abajo OR #MA_Bajar_TP1) AND (#TP2_Abajo OR #MA_Bajar_TP2) AND #TPS1_Arriba AND #TPS3_Arriba);
END_REGION

REGION Network 86: VARIABLES AUXILIARES - Fin de Reset
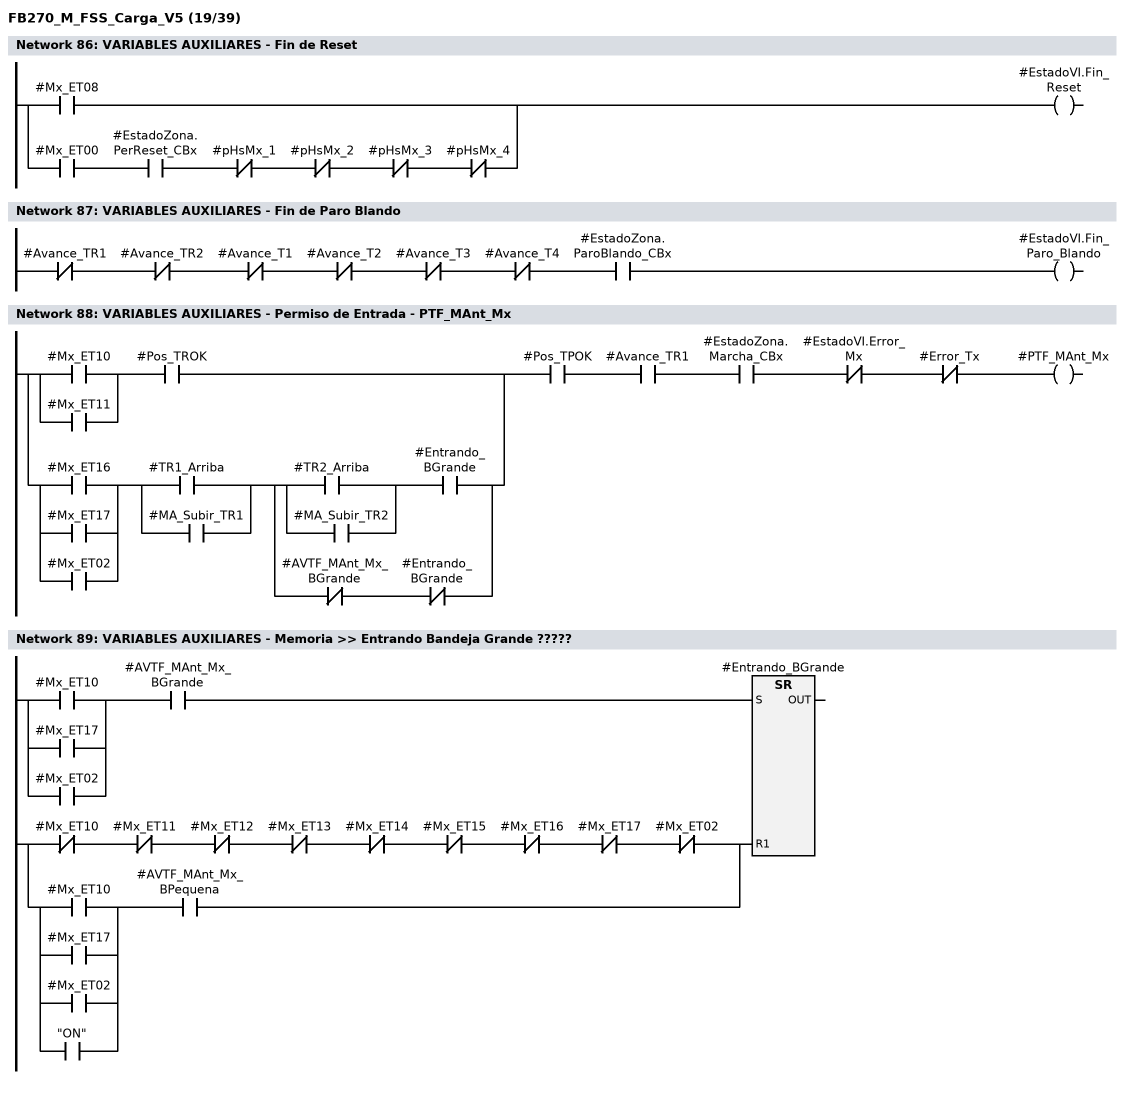
   RUNG wire#powerrail
      Contact( #Mx_ET08 )
      wire#w1
      Coil( #EstadoVI.Fin_Reset )
   END_RUNG
   RUNG wire#powerrail
      Contact( #Mx_ET00 )
      Contact( #EstadoZona.PerReset_CBx )
      I_Contact( #pHsMx_1 )
      I_Contact( #pHsMx_2 )
      I_Contact( #pHsMx_3 )
      I_Contact( #pHsMx_4 )
   END_RUNG wire#w1
   // the same network as SCL:
   #EstadoVI.Fin_Reset := #Mx_ET08 OR (#Mx_ET00 AND #EstadoZona.PerReset_CBx AND NOT #pHsMx_1 AND NOT #pHsMx_2 AND NOT #pHsMx_3 AND NOT #pHsMx_4);
END_REGION

REGION Network 87: VARIABLES AUXILIARES - Fin de Paro Blando
   RUNG wire#powerrail
      I_Contact( #Avance_TR1 )
      I_Contact( #Avance_TR2 )
      I_Contact( #Avance_T1 )
      I_Contact( #Avance_T2 )
      I_Contact( #Avance_T3 )
      I_Contact( #Avance_T4 )
      Contact( #EstadoZona.ParoBlando_CBx )
      Coil( #EstadoVI.Fin_Paro_Blando )
   END_RUNG
   // the same network as SCL:
   #EstadoVI.Fin_Paro_Blando := NOT #Avance_TR1 AND NOT #Avance_TR2 AND NOT #Avance_T1 AND NOT #Avance_T2 AND NOT #Avance_T3 AND NOT #Avance_T4 AND #EstadoZona.ParoBlando_CBx;
END_REGION

REGION Network 88: VARIABLES AUXILIARES - Permiso de Entrada - PTF_MAnt_Mx
   RUNG wire#powerrail
      Contact( #Mx_ET10 )
      wire#w1
      Contact( #Pos_TROK )
      wire#w2
      Contact( #Pos_TPOK )
      Contact( #Avance_TR1 )
      Contact( #EstadoZona.Marcha_CBx )
      I_Contact( #EstadoVI.Error_Mx )
      I_Contact( #Error_Tx )
      Coil( #PTF_MAnt_Mx )
   END_RUNG
   RUNG wire#powerrail
      Contact( #Mx_ET11 )
   END_RUNG wire#w1
   RUNG wire#powerrail
      Contact( #Mx_ET16 )
      wire#w3
      Contact( #TR1_Arriba )
      wire#w4
      Contact( #TR2_Arriba )
      wire#w5
      Contact( #Entrando_BGrande )
   END_RUNG wire#w2
   RUNG wire#powerrail
      Contact( #Mx_ET17 )
   END_RUNG wire#w3
   RUNG wire#powerrail
      Contact( #Mx_ET02 )
   END_RUNG wire#w3
   RUNG wire#w3
      Contact( #MA_Subir_TR1 )
   END_RUNG wire#w4
   RUNG wire#w4
      Contact( #MA_Subir_TR2 )
   END_RUNG wire#w5
   RUNG wire#w4
      I_Contact( #AVTF_MAnt_Mx_BGrande )
      I_Contact( #Entrando_BGrande )
   END_RUNG wire#w2
   // the same network as SCL:
   #PTF_MAnt_Mx := (((#Mx_ET10 OR #Mx_ET11) AND #Pos_TROK) OR ((#Mx_ET16 OR #Mx_ET17 OR #Mx_ET02) AND (#TR1_Arriba OR #MA_Subir_TR1) AND (((#TR2_Arriba OR #MA_Subir_TR2) AND #Entrando_BGrande) OR (NOT #AVTF_MAnt_Mx_BGrande AND NOT #Entrando_BGrande)))) AND #Pos_TPOK AND #Avance_TR1 AND #EstadoZona.Marcha_CBx AND NOT #EstadoVI.Error_Mx AND NOT #Error_Tx;
END_REGION

REGION Network 89: VARIABLES AUXILIARES - Memoria >> Entrando Bandeja Grande ?????
   RUNG wire#powerrail
      Contact( #Mx_ET10 )
      wire#w1
      Contact( #AVTF_MAnt_Mx_BGrande )
      S_SR(operand := #Entrando_BGrande, r1 := wire#w3)
   END_RUNG
   RUNG wire#powerrail
      Contact( #Mx_ET17 )
   END_RUNG wire#w1
   RUNG wire#powerrail
      Contact( #Mx_ET02 )
   END_RUNG wire#w1
   RUNG wire#powerrail
      I_Contact( #Mx_ET10 )
      I_Contact( #Mx_ET11 )
      I_Contact( #Mx_ET12 )
      I_Contact( #Mx_ET13 )
      I_Contact( #Mx_ET14 )
      I_Contact( #Mx_ET15 )
      I_Contact( #Mx_ET16 )
      I_Contact( #Mx_ET17 )
      I_Contact( #Mx_ET02 )
   END_RUNG wire#w3
   RUNG wire#powerrail
      Contact( #Mx_ET10 )
      wire#w2
      Contact( #AVTF_MAnt_Mx_BPequena )
   END_RUNG wire#w3
   RUNG wire#powerrail
      Contact( #Mx_ET17 )
   END_RUNG wire#w2
   RUNG wire#powerrail
      Contact( #Mx_ET02 )
   END_RUNG wire#w2
   RUNG wire#powerrail
      Contact( "ON" )
   END_RUNG wire#w2
   // the same network as SCL:
   IF (#Mx_ET10 OR #Mx_ET17 OR #Mx_ET02) AND #AVTF_MAnt_Mx_BGrande THEN
       #Entrando_BGrande := TRUE;   // SR flip-flop
   END_IF;
   IF (NOT #Mx_ET10 AND NOT #Mx_ET11 AND NOT #Mx_ET12 AND NOT #Mx_ET13 AND NOT #Mx_ET14 AND NOT #Mx_ET15 AND NOT #Mx_ET16 AND NOT #Mx_ET17 AND NOT #Mx_ET02) OR ((#Mx_ET10 OR #Mx_ET17 OR #Mx_ET02 OR "ON") AND #AVTF_MAnt_Mx_BPequena) THEN
       #Entrando_BGrande := FALSE;
   END_IF;
END_REGION

REGION Network 90: VARIABLES AUXILIARES - Memoria de Carga Posicionada >> SET
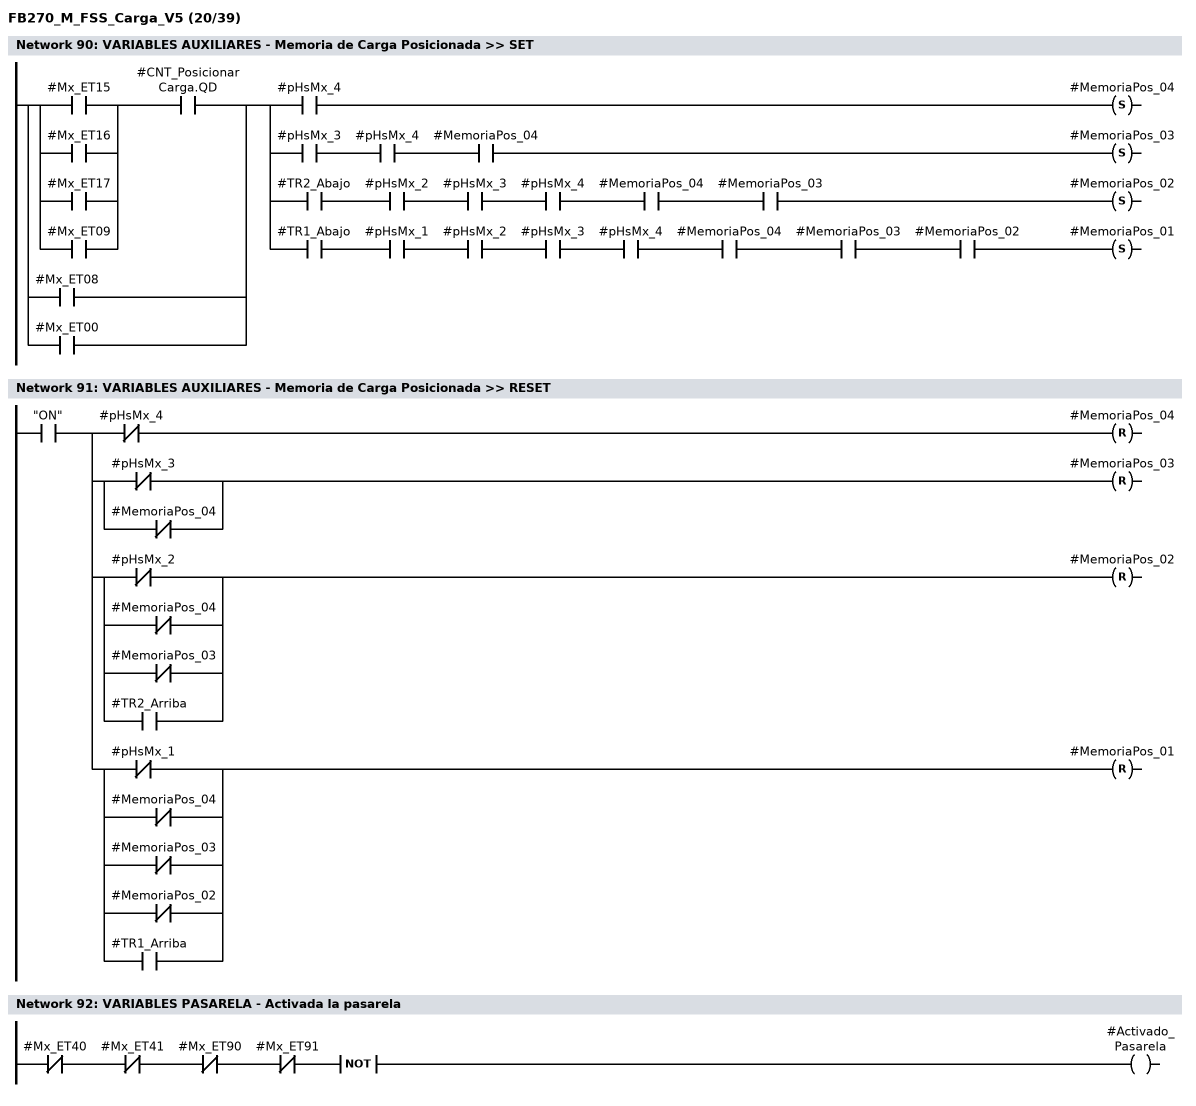
   RUNG wire#powerrail
      Contact( #Mx_ET15 )
      wire#w1
      Contact( #CNT_PosicionarCarga.QD )
      wire#w2
      Contact( #pHsMx_4 )
      S_Coil( #MemoriaPos_04 )
   END_RUNG
   RUNG wire#powerrail
      Contact( #Mx_ET16 )
   END_RUNG wire#w1
   RUNG wire#powerrail
      Contact( #Mx_ET17 )
   END_RUNG wire#w1
   RUNG wire#powerrail
      Contact( #Mx_ET09 )
   END_RUNG wire#w1
   RUNG wire#powerrail
      Contact( #Mx_ET08 )
   END_RUNG wire#w2
   RUNG wire#powerrail
      Contact( #Mx_ET00 )
   END_RUNG wire#w2
   RUNG wire#w2
      Contact( #pHsMx_3 )
      Contact( #pHsMx_4 )
      Contact( #MemoriaPos_04 )
      S_Coil( #MemoriaPos_03 )
   END_RUNG
   RUNG wire#w2
      Contact( #TR2_Abajo )
      Contact( #pHsMx_2 )
      Contact( #pHsMx_3 )
      Contact( #pHsMx_4 )
      Contact( #MemoriaPos_04 )
      Contact( #MemoriaPos_03 )
      S_Coil( #MemoriaPos_02 )
   END_RUNG
   RUNG wire#w2
      Contact( #TR1_Abajo )
      Contact( #pHsMx_1 )
      Contact( #pHsMx_2 )
      Contact( #pHsMx_3 )
      Contact( #pHsMx_4 )
      Contact( #MemoriaPos_04 )
      Contact( #MemoriaPos_03 )
      Contact( #MemoriaPos_02 )
      S_Coil( #MemoriaPos_01 )
   END_RUNG
   // the same network as SCL:
   #_w1 := ((#Mx_ET15 OR #Mx_ET16 OR #Mx_ET17 OR #Mx_ET09) AND #CNT_PosicionarCarga.QD) OR #Mx_ET08 OR #Mx_ET00;
   IF #_w1 AND #pHsMx_4 THEN #MemoriaPos_04 := TRUE; END_IF;
   IF #_w1 AND #pHsMx_3 AND #pHsMx_4 AND #MemoriaPos_04 THEN #MemoriaPos_03 := TRUE; END_IF;
   IF #_w1 AND #TR2_Abajo AND #pHsMx_2 AND #pHsMx_3 AND #pHsMx_4 AND #MemoriaPos_04 AND #MemoriaPos_03 THEN
       #MemoriaPos_02 := TRUE;
   END_IF;
   IF #_w1 AND #TR1_Abajo AND #pHsMx_1 AND #pHsMx_2 AND #pHsMx_3 AND #pHsMx_4 AND #MemoriaPos_04 AND #MemoriaPos_03 AND #MemoriaPos_02 THEN
       #MemoriaPos_01 := TRUE;
   END_IF;
END_REGION

REGION Network 91: VARIABLES AUXILIARES - Memoria de Carga Posicionada >> RESET
   RUNG wire#powerrail
      Contact( "ON" )
      wire#w1
      I_Contact( #pHsMx_4 )
      R_Coil( #MemoriaPos_04 )
   END_RUNG
   RUNG wire#w1
      I_Contact( #pHsMx_3 )
      wire#w2
      R_Coil( #MemoriaPos_03 )
   END_RUNG
   RUNG wire#w1
      I_Contact( #MemoriaPos_04 )
   END_RUNG wire#w2
   RUNG wire#w1
      I_Contact( #pHsMx_2 )
      wire#w3
      R_Coil( #MemoriaPos_02 )
   END_RUNG
   RUNG wire#w1
      I_Contact( #MemoriaPos_04 )
   END_RUNG wire#w3
   RUNG wire#w1
      I_Contact( #MemoriaPos_03 )
   END_RUNG wire#w3
   RUNG wire#w1
      Contact( #TR2_Arriba )
   END_RUNG wire#w3
   RUNG wire#w1
      I_Contact( #pHsMx_1 )
      wire#w4
      R_Coil( #MemoriaPos_01 )
   END_RUNG
   RUNG wire#w1
      I_Contact( #MemoriaPos_04 )
   END_RUNG wire#w4
   RUNG wire#w1
      I_Contact( #MemoriaPos_03 )
   END_RUNG wire#w4
   RUNG wire#w1
      I_Contact( #MemoriaPos_02 )
   END_RUNG wire#w4
   RUNG wire#w1
      Contact( #TR1_Arriba )
   END_RUNG wire#w4
   // the same network as SCL:
   IF "ON" AND NOT #pHsMx_4 THEN #MemoriaPos_04 := FALSE; END_IF;
   IF "ON" AND (NOT #pHsMx_3 OR NOT #MemoriaPos_04) THEN #MemoriaPos_03 := FALSE; END_IF;
   IF "ON" AND (NOT #pHsMx_2 OR NOT #MemoriaPos_04 OR NOT #MemoriaPos_03 OR #TR2_Arriba) THEN
       #MemoriaPos_02 := FALSE;
   END_IF;
   IF "ON" AND (NOT #pHsMx_1 OR NOT #MemoriaPos_04 OR NOT #MemoriaPos_03 OR NOT #MemoriaPos_02 OR #TR1_Arriba) THEN
       #MemoriaPos_01 := FALSE;
   END_IF;
END_REGION

REGION Network 92: VARIABLES PASARELA - Activada la pasarela
   RUNG wire#powerrail
      I_Contact( #Mx_ET40 )
      I_Contact( #Mx_ET41 )
      I_Contact( #Mx_ET90 )
      I_Contact( #Mx_ET91 )
      Not()
      Coil( #Activado_Pasarela )
   END_RUNG
   // the same network as SCL:
   #Activado_Pasarela := NOT (NOT #Mx_ET40 AND NOT #Mx_ET41 AND NOT #Mx_ET90 AND NOT #Mx_ET91);
END_REGION

REGION Network 93: CONTADOR DE PRESENCIA EN PASARELA - CENTRADO DE LA CARGA >>> CNT_PresenciaPasarela
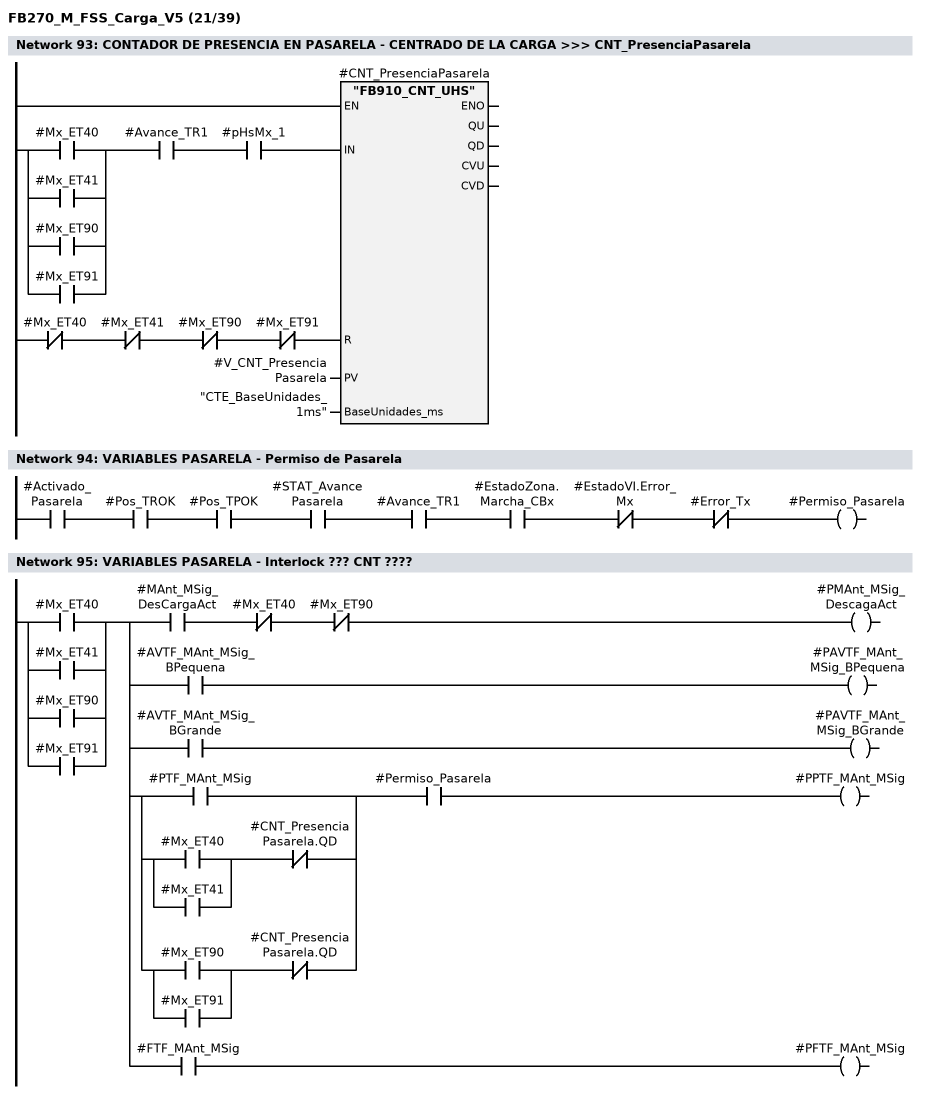
   RUNG wire#powerrail
      #CNT_PresenciaPasarela(IN := wire#w2, R := wire#w3, PV := #V_CNT_PresenciaPasarela, BaseUnidades_ms := "CTE_BaseUnidades_1ms", QU =>, QD =>, CVU =>, CVD =>)
   END_RUNG
   RUNG wire#powerrail
      Contact( #Mx_ET40 )
      wire#w1
      Contact( #Avance_TR1 )
      Contact( #pHsMx_1 )
   END_RUNG wire#w2
   RUNG wire#powerrail
      Contact( #Mx_ET41 )
   END_RUNG wire#w1
   RUNG wire#powerrail
      Contact( #Mx_ET90 )
   END_RUNG wire#w1
   RUNG wire#powerrail
      Contact( #Mx_ET91 )
   END_RUNG wire#w1
   RUNG wire#powerrail
      I_Contact( #Mx_ET40 )
      I_Contact( #Mx_ET41 )
      I_Contact( #Mx_ET90 )
      I_Contact( #Mx_ET91 )
   END_RUNG wire#w3
   // the same network as SCL:
   #CNT_PresenciaPasarela(IN := (#Mx_ET40 OR #Mx_ET41 OR #Mx_ET90 OR #Mx_ET91) AND #Avance_TR1 AND #pHsMx_1,   // "FB910_CNT_UHS"
                          R := NOT #Mx_ET40 AND NOT #Mx_ET41 AND NOT #Mx_ET90 AND NOT #Mx_ET91,
                          PV := #V_CNT_PresenciaPasarela,
                          BaseUnidades_ms := "CTE_BaseUnidades_1ms");
END_REGION

REGION Network 94: VARIABLES PASARELA - Permiso de Pasarela
   RUNG wire#powerrail
      Contact( #Activado_Pasarela )
      Contact( #Pos_TROK )
      Contact( #Pos_TPOK )
      Contact( #STAT_AvancePasarela )
      Contact( #Avance_TR1 )
      Contact( #EstadoZona.Marcha_CBx )
      I_Contact( #EstadoVI.Error_Mx )
      I_Contact( #Error_Tx )
      Coil( #Permiso_Pasarela )
   END_RUNG
   // the same network as SCL:
   #Permiso_Pasarela := #Activado_Pasarela AND #Pos_TROK AND #Pos_TPOK AND #STAT_AvancePasarela AND #Avance_TR1 AND #EstadoZona.Marcha_CBx AND NOT #EstadoVI.Error_Mx AND NOT #Error_Tx;
END_REGION

REGION Network 95: VARIABLES PASARELA - Interlock ??? CNT ????
   RUNG wire#powerrail
      Contact( #Mx_ET40 )
      wire#w1
      Contact( #MAnt_MSig_DesCargaAct )
      I_Contact( #Mx_ET40 )
      I_Contact( #Mx_ET90 )
      Coil( #PMAnt_MSig_DescagaAct )
   END_RUNG
   RUNG wire#powerrail
      Contact( #Mx_ET41 )
   END_RUNG wire#w1
   RUNG wire#powerrail
      Contact( #Mx_ET90 )
   END_RUNG wire#w1
   RUNG wire#powerrail
      Contact( #Mx_ET91 )
   END_RUNG wire#w1
   RUNG wire#w1
      Contact( #AVTF_MAnt_MSig_BPequena )
      Coil( #PAVTF_MAnt_MSig_BPequena )
   END_RUNG
   RUNG wire#w1
      Contact( #AVTF_MAnt_MSig_BGrande )
      Coil( #PAVTF_MAnt_MSig_BGrande )
   END_RUNG
   RUNG wire#w1
      Contact( #PTF_MAnt_MSig )
      wire#w2
      Contact( #Permiso_Pasarela )
      Coil( #PPTF_MAnt_MSig )
   END_RUNG
   RUNG wire#w1
      Contact( #Mx_ET40 )
      wire#w3
      I_Contact( #CNT_PresenciaPasarela.QD )
   END_RUNG wire#w2
   RUNG wire#w1
      Contact( #Mx_ET41 )
   END_RUNG wire#w3
   RUNG wire#w1
      Contact( #Mx_ET90 )
      wire#w4
      I_Contact( #CNT_PresenciaPasarela.QD )
   END_RUNG wire#w2
   RUNG wire#w1
      Contact( #Mx_ET91 )
   END_RUNG wire#w4
   RUNG wire#w1
      Contact( #FTF_MAnt_MSig )
      Coil( #PFTF_MAnt_MSig )
   END_RUNG
   // the same network as SCL:
   #_w1 := #Mx_ET40 OR #Mx_ET41 OR #Mx_ET90 OR #Mx_ET91;
   #PMAnt_MSig_DescagaAct := #_w1 AND #MAnt_MSig_DesCargaAct AND NOT #Mx_ET40 AND NOT #Mx_ET90;
   #PAVTF_MAnt_MSig_BPequena := #_w1 AND #AVTF_MAnt_MSig_BPequena;
   #PAVTF_MAnt_MSig_BGrande := #_w1 AND #AVTF_MAnt_MSig_BGrande;
   #PPTF_MAnt_MSig := #_w1 AND (#PTF_MAnt_MSig OR ((#Mx_ET40 OR #Mx_ET41) AND NOT #CNT_PresenciaPasarela.QD) OR ((#Mx_ET90 OR #Mx_ET91) AND NOT #CNT_PresenciaPasarela.QD)) AND #Permiso_Pasarela;
   #PFTF_MAnt_MSig := #_w1 AND #FTF_MAnt_MSig;
END_REGION

REGION Network 96: MENSAJES - PRESENCIA
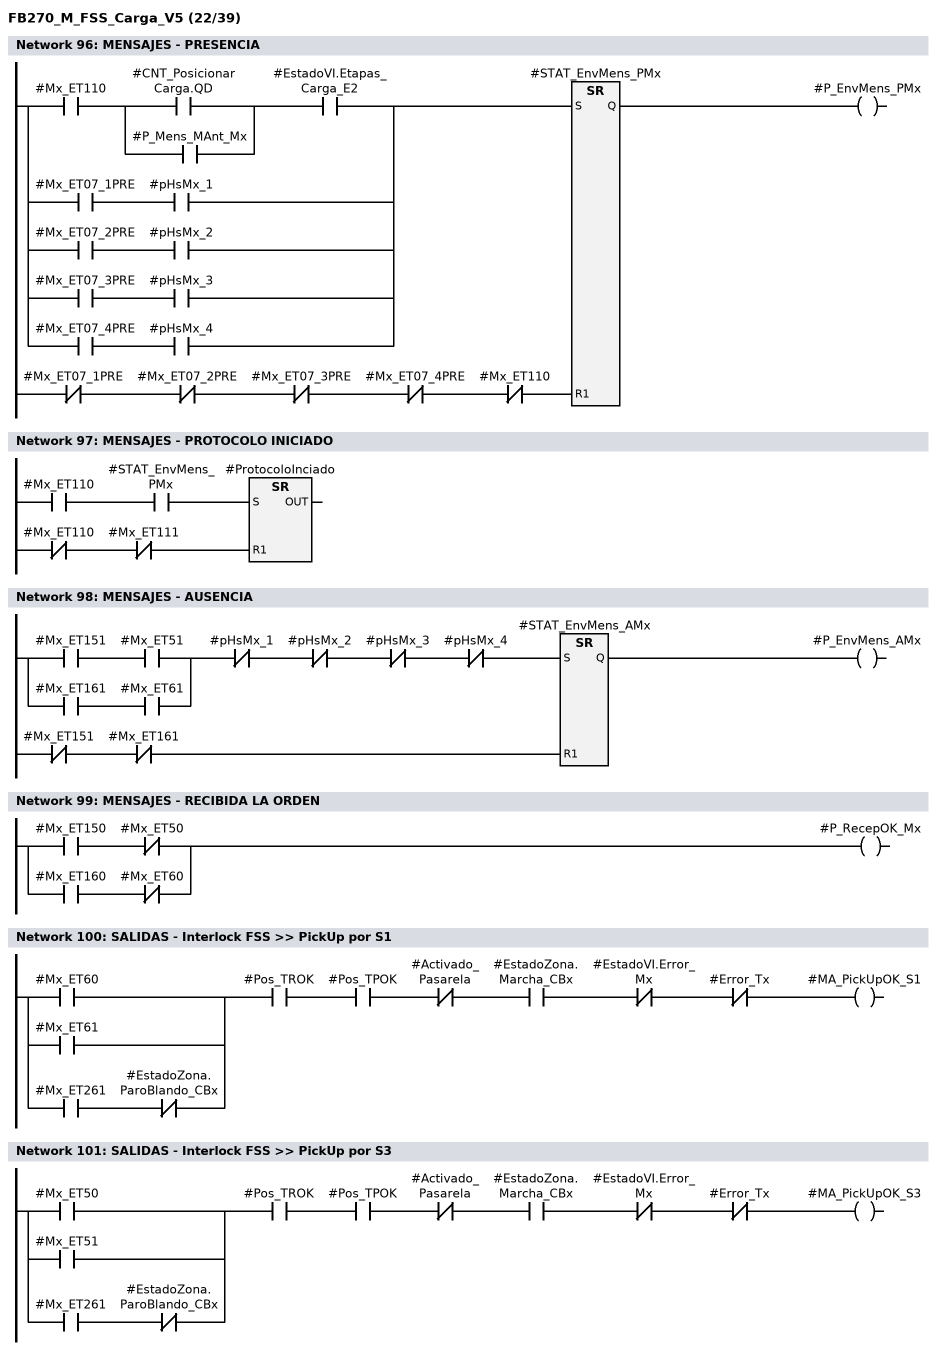
   RUNG wire#powerrail
      Contact( #Mx_ET110 )
      wire#w1
      Contact( #CNT_PosicionarCarga.QD )
      wire#w2
      Contact( #EstadoVI.Etapas_Carga_E2 )
      wire#w3
      S_SR(operand := #STAT_EnvMens_PMx, r1 := wire#w4)
      Coil( #P_EnvMens_PMx )
   END_RUNG
   RUNG wire#w1
      Contact( #P_Mens_MAnt_Mx )
   END_RUNG wire#w2
   RUNG wire#powerrail
      Contact( #Mx_ET07_1PRE )
      Contact( #pHsMx_1 )
   END_RUNG wire#w3
   RUNG wire#powerrail
      Contact( #Mx_ET07_2PRE )
      Contact( #pHsMx_2 )
   END_RUNG wire#w3
   RUNG wire#powerrail
      Contact( #Mx_ET07_3PRE )
      Contact( #pHsMx_3 )
   END_RUNG wire#w3
   RUNG wire#powerrail
      Contact( #Mx_ET07_4PRE )
      Contact( #pHsMx_4 )
   END_RUNG wire#w3
   RUNG wire#powerrail
      I_Contact( #Mx_ET07_1PRE )
      I_Contact( #Mx_ET07_2PRE )
      I_Contact( #Mx_ET07_3PRE )
      I_Contact( #Mx_ET07_4PRE )
      I_Contact( #Mx_ET110 )
   END_RUNG wire#w4
   // the same network as SCL:
   IF (#Mx_ET110 AND (#CNT_PosicionarCarga.QD OR #P_Mens_MAnt_Mx) AND #EstadoVI.Etapas_Carga_E2) OR (#Mx_ET07_1PRE AND #pHsMx_1) OR (#Mx_ET07_2PRE AND #pHsMx_2) OR (#Mx_ET07_3PRE AND #pHsMx_3) OR (#Mx_ET07_4PRE AND #pHsMx_4) THEN
       #STAT_EnvMens_PMx := TRUE;   // SR flip-flop
   END_IF;
   IF NOT #Mx_ET07_1PRE AND NOT #Mx_ET07_2PRE AND NOT #Mx_ET07_3PRE AND NOT #Mx_ET07_4PRE AND NOT #Mx_ET110 THEN
       #STAT_EnvMens_PMx := FALSE;
   END_IF;
   #P_EnvMens_PMx := #STAT_EnvMens_PMx;
END_REGION

REGION Network 97: MENSAJES - PROTOCOLO INICIADO
   RUNG wire#powerrail
      Contact( #Mx_ET110 )
      Contact( #STAT_EnvMens_PMx )
      S_SR(operand := #ProtocoloInciado, r1 := wire#w1)
   END_RUNG
   RUNG wire#powerrail
      I_Contact( #Mx_ET110 )
      I_Contact( #Mx_ET111 )
   END_RUNG wire#w1
   // the same network as SCL:
   IF #Mx_ET110 AND #STAT_EnvMens_PMx THEN
       #ProtocoloInciado := TRUE;   // SR flip-flop
   END_IF;
   IF NOT #Mx_ET110 AND NOT #Mx_ET111 THEN #ProtocoloInciado := FALSE; END_IF;
END_REGION

REGION Network 98: MENSAJES - AUSENCIA
   RUNG wire#powerrail
      Contact( #Mx_ET151 )
      Contact( #Mx_ET51 )
      wire#w1
      I_Contact( #pHsMx_1 )
      I_Contact( #pHsMx_2 )
      I_Contact( #pHsMx_3 )
      I_Contact( #pHsMx_4 )
      S_SR(operand := #STAT_EnvMens_AMx, r1 := wire#w2)
      Coil( #P_EnvMens_AMx )
   END_RUNG
   RUNG wire#powerrail
      Contact( #Mx_ET161 )
      Contact( #Mx_ET61 )
   END_RUNG wire#w1
   RUNG wire#powerrail
      I_Contact( #Mx_ET151 )
      I_Contact( #Mx_ET161 )
   END_RUNG wire#w2
   // the same network as SCL:
   IF ((#Mx_ET151 AND #Mx_ET51) OR (#Mx_ET161 AND #Mx_ET61)) AND NOT #pHsMx_1 AND NOT #pHsMx_2 AND NOT #pHsMx_3 AND NOT #pHsMx_4 THEN
       #STAT_EnvMens_AMx := TRUE;   // SR flip-flop
   END_IF;
   IF NOT #Mx_ET151 AND NOT #Mx_ET161 THEN #STAT_EnvMens_AMx := FALSE; END_IF;
   #P_EnvMens_AMx := #STAT_EnvMens_AMx;
END_REGION

REGION Network 99: MENSAJES - RECIBIDA LA ORDEN
   RUNG wire#powerrail
      Contact( #Mx_ET150 )
      I_Contact( #Mx_ET50 )
      wire#w1
      Coil( #P_RecepOK_Mx )
   END_RUNG
   RUNG wire#powerrail
      Contact( #Mx_ET160 )
      I_Contact( #Mx_ET60 )
   END_RUNG wire#w1
   // the same network as SCL:
   #P_RecepOK_Mx := (#Mx_ET150 AND NOT #Mx_ET50) OR (#Mx_ET160 AND NOT #Mx_ET60);
END_REGION

REGION Network 100: SALIDAS - Interlock FSS >> PickUp por S1
   RUNG wire#powerrail
      Contact( #Mx_ET60 )
      wire#w1
      Contact( #Pos_TROK )
      Contact( #Pos_TPOK )
      I_Contact( #Activado_Pasarela )
      Contact( #EstadoZona.Marcha_CBx )
      I_Contact( #EstadoVI.Error_Mx )
      I_Contact( #Error_Tx )
      Coil( #MA_PickUpOK_S1 )
   END_RUNG
   RUNG wire#powerrail
      Contact( #Mx_ET61 )
   END_RUNG wire#w1
   RUNG wire#powerrail
      Contact( #Mx_ET261 )
      I_Contact( #EstadoZona.ParoBlando_CBx )
   END_RUNG wire#w1
   // the same network as SCL:
   #MA_PickUpOK_S1 := (#Mx_ET60 OR #Mx_ET61 OR (#Mx_ET261 AND NOT #EstadoZona.ParoBlando_CBx)) AND #Pos_TROK AND #Pos_TPOK AND NOT #Activado_Pasarela AND #EstadoZona.Marcha_CBx AND NOT #EstadoVI.Error_Mx AND NOT #Error_Tx;
END_REGION

REGION Network 101: SALIDAS - Interlock FSS >> PickUp por S3
   RUNG wire#powerrail
      Contact( #Mx_ET50 )
      wire#w1
      Contact( #Pos_TROK )
      Contact( #Pos_TPOK )
      I_Contact( #Activado_Pasarela )
      Contact( #EstadoZona.Marcha_CBx )
      I_Contact( #EstadoVI.Error_Mx )
      I_Contact( #Error_Tx )
      Coil( #MA_PickUpOK_S3 )
   END_RUNG
   RUNG wire#powerrail
      Contact( #Mx_ET51 )
   END_RUNG wire#w1
   RUNG wire#powerrail
      Contact( #Mx_ET261 )
      I_Contact( #EstadoZona.ParoBlando_CBx )
   END_RUNG wire#w1
   // the same network as SCL:
   #MA_PickUpOK_S3 := (#Mx_ET50 OR #Mx_ET51 OR (#Mx_ET261 AND NOT #EstadoZona.ParoBlando_CBx)) AND #Pos_TROK AND #Pos_TPOK AND NOT #Activado_Pasarela AND #EstadoZona.Marcha_CBx AND NOT #EstadoVI.Error_Mx AND NOT #Error_Tx;
END_REGION

REGION Network 102: VARIABLES INTERNAS - AVANCE DE CARGA
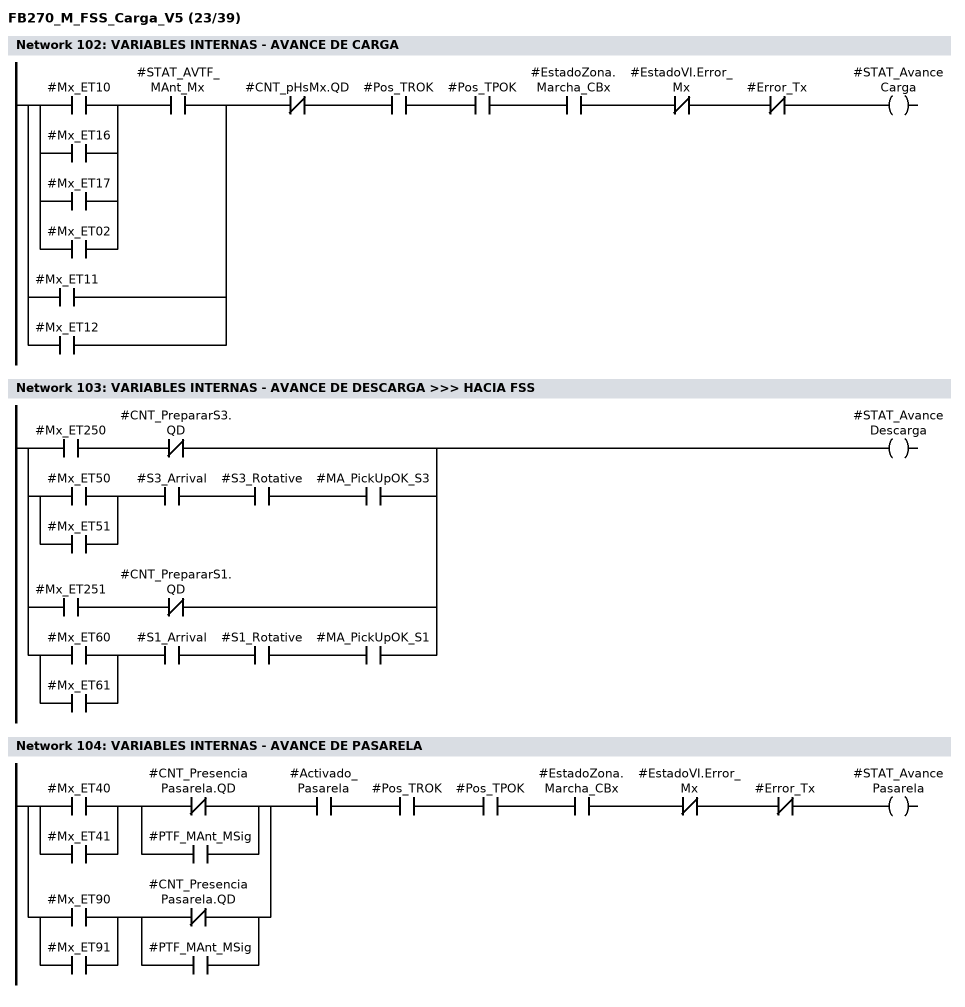
   RUNG wire#powerrail
      Contact( #Mx_ET10 )
      wire#w1
      Contact( #STAT_AVTF_MAnt_Mx )
      wire#w2
      I_Contact( #CNT_pHsMx.QD )
      Contact( #Pos_TROK )
      Contact( #Pos_TPOK )
      Contact( #EstadoZona.Marcha_CBx )
      I_Contact( #EstadoVI.Error_Mx )
      I_Contact( #Error_Tx )
      Coil( #STAT_AvanceCarga )
   END_RUNG
   RUNG wire#powerrail
      Contact( #Mx_ET16 )
   END_RUNG wire#w1
   RUNG wire#powerrail
      Contact( #Mx_ET17 )
   END_RUNG wire#w1
   RUNG wire#powerrail
      Contact( #Mx_ET02 )
   END_RUNG wire#w1
   RUNG wire#powerrail
      Contact( #Mx_ET11 )
   END_RUNG wire#w2
   RUNG wire#powerrail
      Contact( #Mx_ET12 )
   END_RUNG wire#w2
   // the same network as SCL:
   #STAT_AvanceCarga := (((#Mx_ET10 OR #Mx_ET16 OR #Mx_ET17 OR #Mx_ET02) AND #STAT_AVTF_MAnt_Mx) OR #Mx_ET11 OR #Mx_ET12) AND NOT #CNT_pHsMx.QD AND #Pos_TROK AND #Pos_TPOK AND #EstadoZona.Marcha_CBx AND NOT #EstadoVI.Error_Mx AND NOT #Error_Tx;
END_REGION

REGION Network 103: VARIABLES INTERNAS - AVANCE DE DESCARGA >>> HACIA FSS
   RUNG wire#powerrail
      Contact( #Mx_ET250 )
      I_Contact( #CNT_PrepararS3.QD )
      wire#w1
      Coil( #STAT_AvanceDescarga )
   END_RUNG
   RUNG wire#powerrail
      Contact( #Mx_ET50 )
      wire#w2
      Contact( #S3_Arrival )
      Contact( #S3_Rotative )
      Contact( #MA_PickUpOK_S3 )
   END_RUNG wire#w1
   RUNG wire#powerrail
      Contact( #Mx_ET51 )
   END_RUNG wire#w2
   RUNG wire#powerrail
      Contact( #Mx_ET251 )
      I_Contact( #CNT_PrepararS1.QD )
   END_RUNG wire#w1
   RUNG wire#powerrail
      Contact( #Mx_ET60 )
      wire#w3
      Contact( #S1_Arrival )
      Contact( #S1_Rotative )
      Contact( #MA_PickUpOK_S1 )
   END_RUNG wire#w1
   RUNG wire#powerrail
      Contact( #Mx_ET61 )
   END_RUNG wire#w3
   // the same network as SCL:
   #STAT_AvanceDescarga := (#Mx_ET250 AND NOT #CNT_PrepararS3.QD) OR ((#Mx_ET50 OR #Mx_ET51) AND #S3_Arrival AND #S3_Rotative AND #MA_PickUpOK_S3) OR (#Mx_ET251 AND NOT #CNT_PrepararS1.QD) OR ((#Mx_ET60 OR #Mx_ET61) AND #S1_Arrival AND #S1_Rotative AND #MA_PickUpOK_S1);
END_REGION

REGION Network 104: VARIABLES INTERNAS - AVANCE DE PASARELA
   RUNG wire#powerrail
      Contact( #Mx_ET40 )
      wire#w1
      I_Contact( #CNT_PresenciaPasarela.QD )
      wire#w2
      Contact( #Activado_Pasarela )
      Contact( #Pos_TROK )
      Contact( #Pos_TPOK )
      Contact( #EstadoZona.Marcha_CBx )
      I_Contact( #EstadoVI.Error_Mx )
      I_Contact( #Error_Tx )
      Coil( #STAT_AvancePasarela )
   END_RUNG
   RUNG wire#powerrail
      Contact( #Mx_ET41 )
   END_RUNG wire#w1
   RUNG wire#w1
      Contact( #PTF_MAnt_MSig )
   END_RUNG wire#w2
   RUNG wire#powerrail
      Contact( #Mx_ET90 )
      wire#w3
      I_Contact( #CNT_PresenciaPasarela.QD )
   END_RUNG wire#w2
   RUNG wire#powerrail
      Contact( #Mx_ET91 )
   END_RUNG wire#w3
   RUNG wire#w3
      Contact( #PTF_MAnt_MSig )
   END_RUNG wire#w2
   // the same network as SCL:
   #STAT_AvancePasarela := (((#Mx_ET40 OR #Mx_ET41) AND (NOT #CNT_PresenciaPasarela.QD OR #PTF_MAnt_MSig)) OR ((#Mx_ET90 OR #Mx_ET91) AND (NOT #CNT_PresenciaPasarela.QD OR #PTF_MAnt_MSig))) AND #Activado_Pasarela AND #Pos_TROK AND #Pos_TPOK AND #EstadoZona.Marcha_CBx AND NOT #EstadoVI.Error_Mx AND NOT #Error_Tx;
END_REGION

REGION Network 105: VARIABLES INTERNAS - VELOCIDAD BIT 00 >> RODILLOS 00-LenSima 01-Repos 10-Len 11-Rap
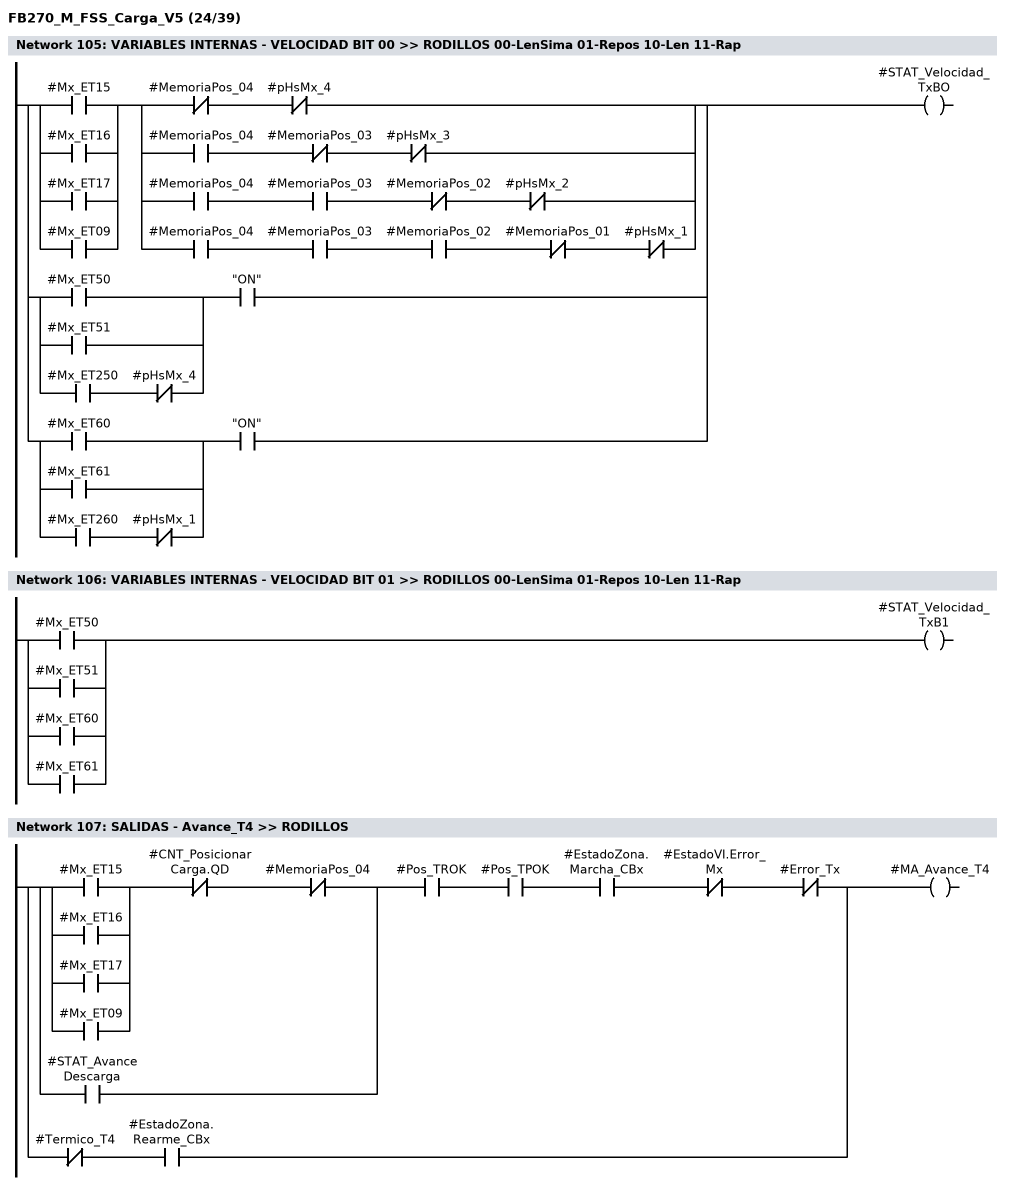
   RUNG wire#powerrail
      Contact( #Mx_ET15 )
      wire#w1
      I_Contact( #MemoriaPos_04 )
      I_Contact( #pHsMx_4 )
      wire#w2
      Coil( #STAT_Velocidad_TxBO )
   END_RUNG
   RUNG wire#powerrail
      Contact( #Mx_ET16 )
   END_RUNG wire#w1
   RUNG wire#powerrail
      Contact( #Mx_ET17 )
   END_RUNG wire#w1
   RUNG wire#powerrail
      Contact( #Mx_ET09 )
   END_RUNG wire#w1
   RUNG wire#w1
      Contact( #MemoriaPos_04 )
      I_Contact( #MemoriaPos_03 )
      I_Contact( #pHsMx_3 )
   END_RUNG wire#w2
   RUNG wire#w1
      Contact( #MemoriaPos_04 )
      Contact( #MemoriaPos_03 )
      I_Contact( #MemoriaPos_02 )
      I_Contact( #pHsMx_2 )
   END_RUNG wire#w2
   RUNG wire#w1
      Contact( #MemoriaPos_04 )
      Contact( #MemoriaPos_03 )
      Contact( #MemoriaPos_02 )
      I_Contact( #MemoriaPos_01 )
      I_Contact( #pHsMx_1 )
   END_RUNG wire#w2
   RUNG wire#powerrail
      Contact( #Mx_ET50 )
      wire#w3
      Contact( "ON" )
   END_RUNG wire#w2
   RUNG wire#powerrail
      Contact( #Mx_ET51 )
   END_RUNG wire#w3
   RUNG wire#powerrail
      Contact( #Mx_ET250 )
      I_Contact( #pHsMx_4 )
   END_RUNG wire#w3
   RUNG wire#powerrail
      Contact( #Mx_ET60 )
      wire#w4
      Contact( "ON" )
   END_RUNG wire#w2
   RUNG wire#powerrail
      Contact( #Mx_ET61 )
   END_RUNG wire#w4
   RUNG wire#powerrail
      Contact( #Mx_ET260 )
      I_Contact( #pHsMx_1 )
   END_RUNG wire#w4
   // the same network as SCL:
   #STAT_Velocidad_TxBO := ((#Mx_ET15 OR #Mx_ET16 OR #Mx_ET17 OR #Mx_ET09) AND ((NOT #MemoriaPos_04 AND NOT #pHsMx_4) OR (#MemoriaPos_04 AND NOT #MemoriaPos_03 AND NOT #pHsMx_3) OR (#MemoriaPos_04 AND #MemoriaPos_03 AND NOT #MemoriaPos_02 AND NOT #pHsMx_2) OR (#MemoriaPos_04 AND #MemoriaPos_03 AND #MemoriaPos_02 AND NOT #MemoriaPos_01 AND NOT #pHsMx_1))) OR ((#Mx_ET50 OR #Mx_ET51 OR (#Mx_ET250 AND NOT #pHsMx_4)) AND "ON") OR ((#Mx_ET60 OR #Mx_ET61 OR (#Mx_ET260 AND NOT #pHsMx_1)) AND "ON");
END_REGION

REGION Network 106: VARIABLES INTERNAS - VELOCIDAD BIT 01 >> RODILLOS 00-LenSima 01-Repos 10-Len 11-Rap
   RUNG wire#powerrail
      Contact( #Mx_ET50 )
      wire#w1
      Coil( #STAT_Velocidad_TxB1 )
   END_RUNG
   RUNG wire#powerrail
      Contact( #Mx_ET51 )
   END_RUNG wire#w1
   RUNG wire#powerrail
      Contact( #Mx_ET60 )
   END_RUNG wire#w1
   RUNG wire#powerrail
      Contact( #Mx_ET61 )
   END_RUNG wire#w1
   // the same network as SCL:
   #STAT_Velocidad_TxB1 := #Mx_ET50 OR #Mx_ET51 OR #Mx_ET60 OR #Mx_ET61;
END_REGION

REGION Network 107: SALIDAS - Avance_T4 >> RODILLOS
   RUNG wire#powerrail
      Contact( #Mx_ET15 )
      wire#w1
      I_Contact( #CNT_PosicionarCarga.QD )
      I_Contact( #MemoriaPos_04 )
      wire#w2
      Contact( #Pos_TROK )
      Contact( #Pos_TPOK )
      Contact( #EstadoZona.Marcha_CBx )
      I_Contact( #EstadoVI.Error_Mx )
      I_Contact( #Error_Tx )
      wire#w3
      Coil( #MA_Avance_T4 )
   END_RUNG
   RUNG wire#powerrail
      Contact( #Mx_ET16 )
   END_RUNG wire#w1
   RUNG wire#powerrail
      Contact( #Mx_ET17 )
   END_RUNG wire#w1
   RUNG wire#powerrail
      Contact( #Mx_ET09 )
   END_RUNG wire#w1
   RUNG wire#powerrail
      Contact( #STAT_AvanceDescarga )
   END_RUNG wire#w2
   RUNG wire#powerrail
      I_Contact( #Termico_T4 )
      Contact( #EstadoZona.Rearme_CBx )
   END_RUNG wire#w3
   // the same network as SCL:
   #MA_Avance_T4 := ((((#Mx_ET15 OR #Mx_ET16 OR #Mx_ET17 OR #Mx_ET09) AND NOT #CNT_PosicionarCarga.QD AND NOT #MemoriaPos_04) OR #STAT_AvanceDescarga) AND #Pos_TROK AND #Pos_TPOK AND #EstadoZona.Marcha_CBx AND NOT #EstadoVI.Error_Mx AND NOT #Error_Tx) OR (NOT #Termico_T4 AND #EstadoZona.Rearme_CBx);
END_REGION

REGION Network 108: SALIDAS - Avance_T3 >> RODILLOS
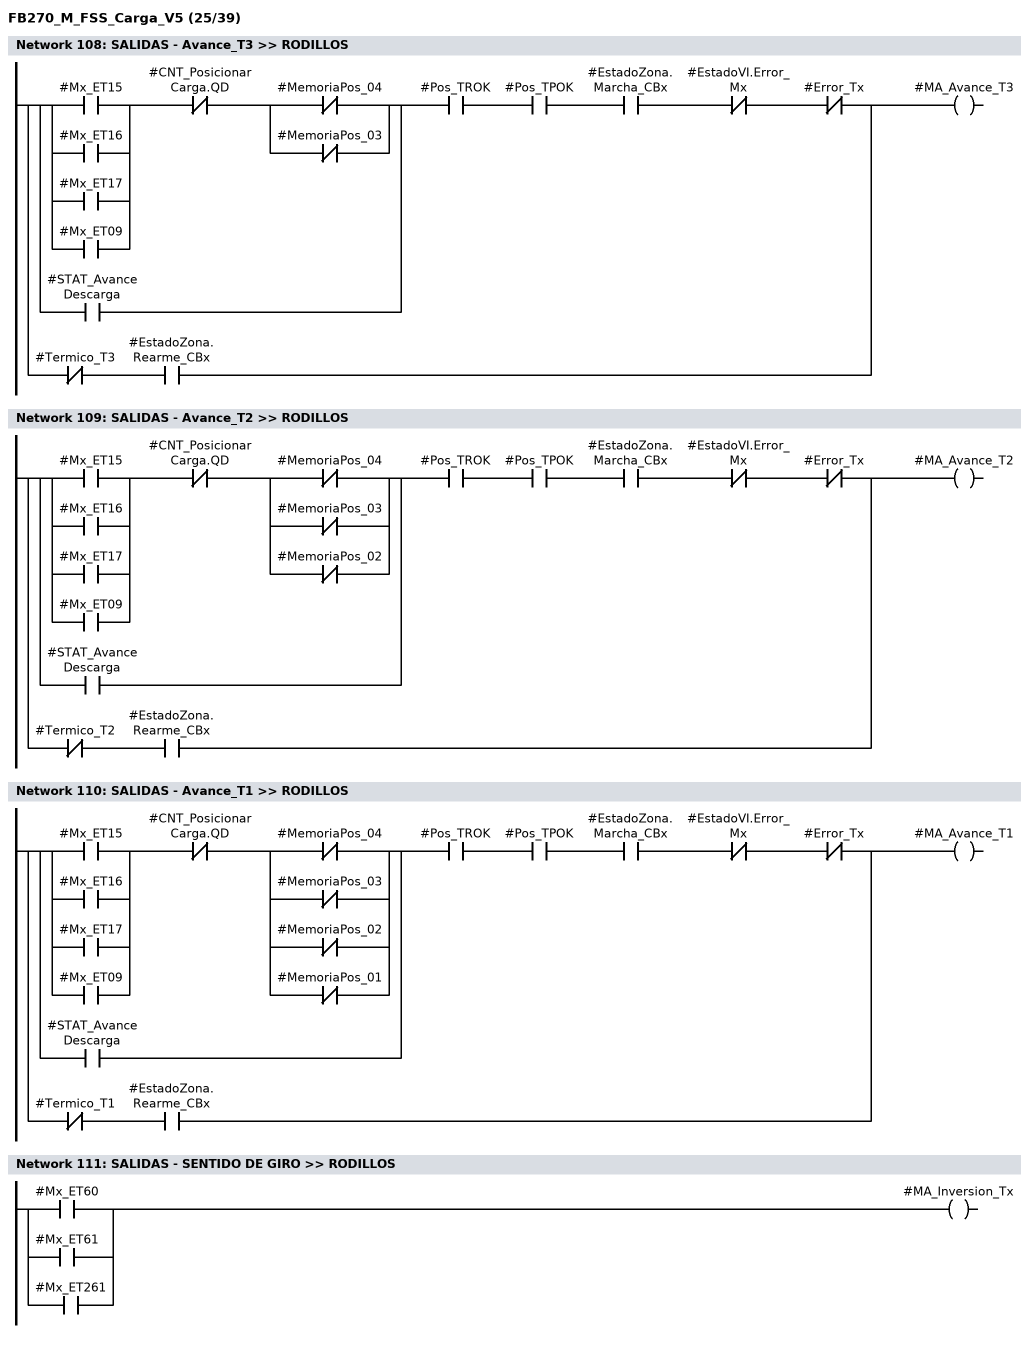
   RUNG wire#powerrail
      Contact( #Mx_ET15 )
      wire#w1
      I_Contact( #CNT_PosicionarCarga.QD )
      wire#w2
      I_Contact( #MemoriaPos_04 )
      wire#w3
      Contact( #Pos_TROK )
      Contact( #Pos_TPOK )
      Contact( #EstadoZona.Marcha_CBx )
      I_Contact( #EstadoVI.Error_Mx )
      I_Contact( #Error_Tx )
      wire#w4
      Coil( #MA_Avance_T3 )
   END_RUNG
   RUNG wire#powerrail
      Contact( #Mx_ET16 )
   END_RUNG wire#w1
   RUNG wire#powerrail
      Contact( #Mx_ET17 )
   END_RUNG wire#w1
   RUNG wire#powerrail
      Contact( #Mx_ET09 )
   END_RUNG wire#w1
   RUNG wire#w2
      I_Contact( #MemoriaPos_03 )
   END_RUNG wire#w3
   RUNG wire#powerrail
      Contact( #STAT_AvanceDescarga )
   END_RUNG wire#w3
   RUNG wire#powerrail
      I_Contact( #Termico_T3 )
      Contact( #EstadoZona.Rearme_CBx )
   END_RUNG wire#w4
   // the same network as SCL:
   #MA_Avance_T3 := ((((#Mx_ET15 OR #Mx_ET16 OR #Mx_ET17 OR #Mx_ET09) AND NOT #CNT_PosicionarCarga.QD AND (NOT #MemoriaPos_04 OR NOT #MemoriaPos_03)) OR #STAT_AvanceDescarga) AND #Pos_TROK AND #Pos_TPOK AND #EstadoZona.Marcha_CBx AND NOT #EstadoVI.Error_Mx AND NOT #Error_Tx) OR (NOT #Termico_T3 AND #EstadoZona.Rearme_CBx);
END_REGION

REGION Network 109: SALIDAS - Avance_T2 >> RODILLOS
   RUNG wire#powerrail
      Contact( #Mx_ET15 )
      wire#w1
      I_Contact( #CNT_PosicionarCarga.QD )
      wire#w2
      I_Contact( #MemoriaPos_04 )
      wire#w3
      Contact( #Pos_TROK )
      Contact( #Pos_TPOK )
      Contact( #EstadoZona.Marcha_CBx )
      I_Contact( #EstadoVI.Error_Mx )
      I_Contact( #Error_Tx )
      wire#w4
      Coil( #MA_Avance_T2 )
   END_RUNG
   RUNG wire#powerrail
      Contact( #Mx_ET16 )
   END_RUNG wire#w1
   RUNG wire#powerrail
      Contact( #Mx_ET17 )
   END_RUNG wire#w1
   RUNG wire#powerrail
      Contact( #Mx_ET09 )
   END_RUNG wire#w1
   RUNG wire#w2
      I_Contact( #MemoriaPos_03 )
   END_RUNG wire#w3
   RUNG wire#w2
      I_Contact( #MemoriaPos_02 )
   END_RUNG wire#w3
   RUNG wire#powerrail
      Contact( #STAT_AvanceDescarga )
   END_RUNG wire#w3
   RUNG wire#powerrail
      I_Contact( #Termico_T2 )
      Contact( #EstadoZona.Rearme_CBx )
   END_RUNG wire#w4
   // the same network as SCL:
   #MA_Avance_T2 := ((((#Mx_ET15 OR #Mx_ET16 OR #Mx_ET17 OR #Mx_ET09) AND NOT #CNT_PosicionarCarga.QD AND (NOT #MemoriaPos_04 OR NOT #MemoriaPos_03 OR NOT #MemoriaPos_02)) OR #STAT_AvanceDescarga) AND #Pos_TROK AND #Pos_TPOK AND #EstadoZona.Marcha_CBx AND NOT #EstadoVI.Error_Mx AND NOT #Error_Tx) OR (NOT #Termico_T2 AND #EstadoZona.Rearme_CBx);
END_REGION

REGION Network 110: SALIDAS - Avance_T1 >> RODILLOS
   RUNG wire#powerrail
      Contact( #Mx_ET15 )
      wire#w1
      I_Contact( #CNT_PosicionarCarga.QD )
      wire#w2
      I_Contact( #MemoriaPos_04 )
      wire#w3
      Contact( #Pos_TROK )
      Contact( #Pos_TPOK )
      Contact( #EstadoZona.Marcha_CBx )
      I_Contact( #EstadoVI.Error_Mx )
      I_Contact( #Error_Tx )
      wire#w4
      Coil( #MA_Avance_T1 )
   END_RUNG
   RUNG wire#powerrail
      Contact( #Mx_ET16 )
   END_RUNG wire#w1
   RUNG wire#powerrail
      Contact( #Mx_ET17 )
   END_RUNG wire#w1
   RUNG wire#powerrail
      Contact( #Mx_ET09 )
   END_RUNG wire#w1
   RUNG wire#w2
      I_Contact( #MemoriaPos_03 )
   END_RUNG wire#w3
   RUNG wire#w2
      I_Contact( #MemoriaPos_02 )
   END_RUNG wire#w3
   RUNG wire#w2
      I_Contact( #MemoriaPos_01 )
   END_RUNG wire#w3
   RUNG wire#powerrail
      Contact( #STAT_AvanceDescarga )
   END_RUNG wire#w3
   RUNG wire#powerrail
      I_Contact( #Termico_T1 )
      Contact( #EstadoZona.Rearme_CBx )
   END_RUNG wire#w4
   // the same network as SCL:
   #MA_Avance_T1 := ((((#Mx_ET15 OR #Mx_ET16 OR #Mx_ET17 OR #Mx_ET09) AND NOT #CNT_PosicionarCarga.QD AND (NOT #MemoriaPos_04 OR NOT #MemoriaPos_03 OR NOT #MemoriaPos_02 OR NOT #MemoriaPos_01)) OR #STAT_AvanceDescarga) AND #Pos_TROK AND #Pos_TPOK AND #EstadoZona.Marcha_CBx AND NOT #EstadoVI.Error_Mx AND NOT #Error_Tx) OR (NOT #Termico_T1 AND #EstadoZona.Rearme_CBx);
END_REGION

REGION Network 111: SALIDAS - SENTIDO DE GIRO >> RODILLOS
   RUNG wire#powerrail
      Contact( #Mx_ET60 )
      wire#w1
      Coil( #MA_Inversion_Tx )
   END_RUNG
   RUNG wire#powerrail
      Contact( #Mx_ET61 )
   END_RUNG wire#w1
   RUNG wire#powerrail
      Contact( #Mx_ET261 )
   END_RUNG wire#w1
   // the same network as SCL:
   #MA_Inversion_Tx := #Mx_ET60 OR #Mx_ET61 OR #Mx_ET261;
END_REGION

REGION Network 112: SALIDAS - VELOCIDAD ANALOGICA >> RODILLOS
   // 25T229A_03 
   // Plantilla_Avance_E1S3_SinVariador_1Mesas.
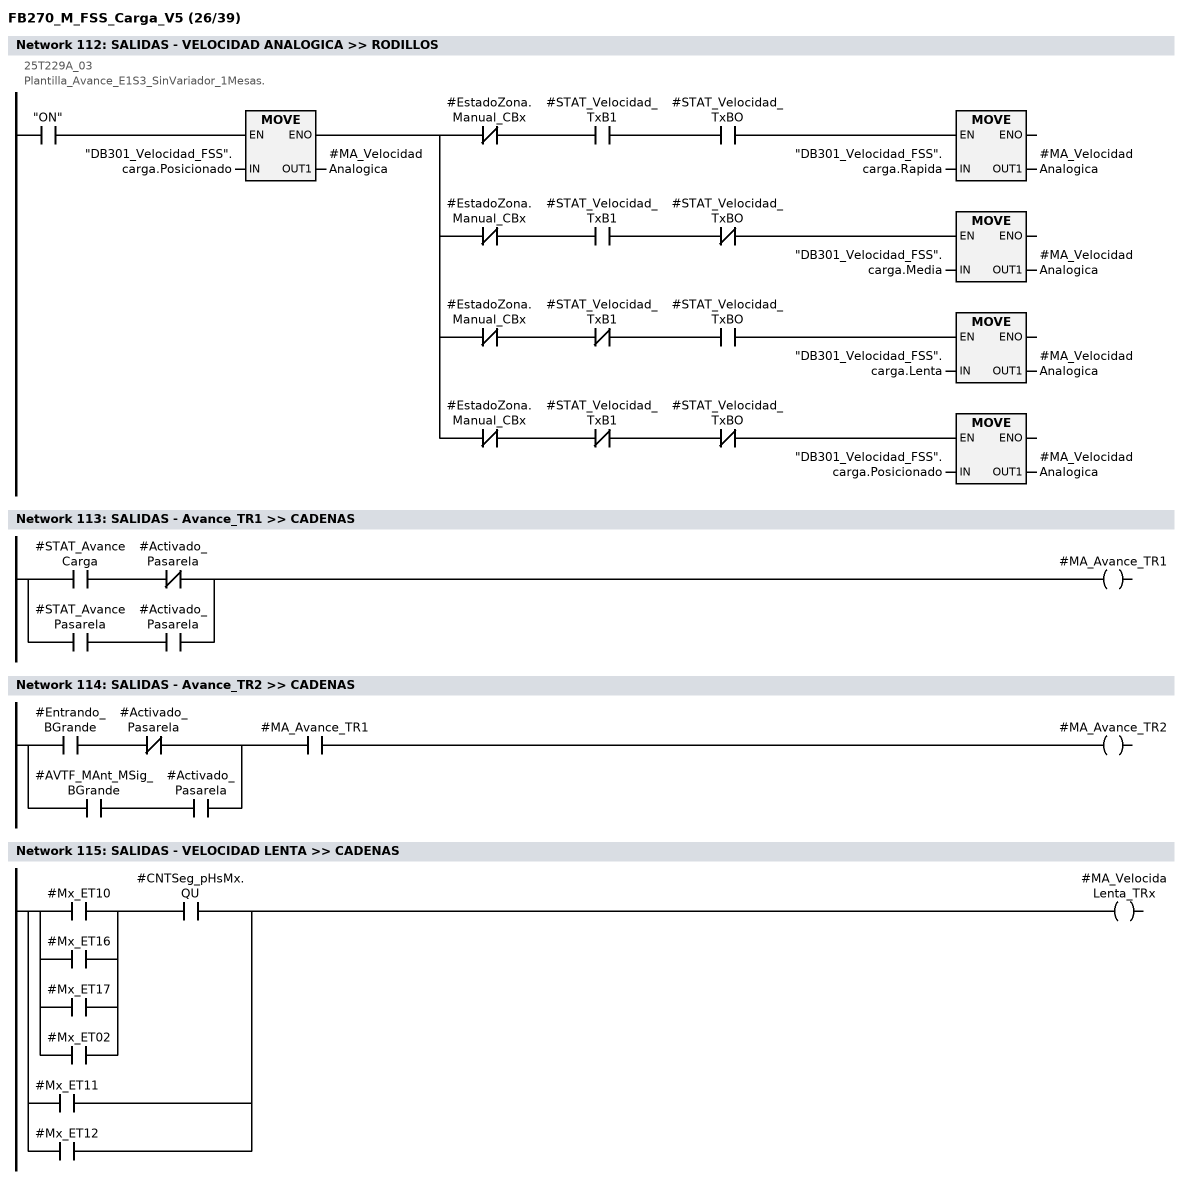
   RUNG wire#powerrail
      Contact( "ON" )
      { S7_GenerateENO := "TRUE" } Move(in := "DB301_Velocidad_FSS".carga.Posicionado, out1 => #MA_VelocidadAnalogica)
      wire#w1
      I_Contact( #EstadoZona.Manual_CBx )
      Contact( #STAT_Velocidad_TxB1 )
      Contact( #STAT_Velocidad_TxBO )
      { S7_GenerateENO := "TRUE" } Move(in := "DB301_Velocidad_FSS".carga.Rapida, out1 => #MA_VelocidadAnalogica)
   END_RUNG
   RUNG wire#w1
      I_Contact( #EstadoZona.Manual_CBx )
      Contact( #STAT_Velocidad_TxB1 )
      I_Contact( #STAT_Velocidad_TxBO )
      { S7_GenerateENO := "TRUE" } Move(in := "DB301_Velocidad_FSS".carga.Media, out1 => #MA_VelocidadAnalogica)
   END_RUNG
   RUNG wire#w1
      I_Contact( #EstadoZona.Manual_CBx )
      I_Contact( #STAT_Velocidad_TxB1 )
      Contact( #STAT_Velocidad_TxBO )
      { S7_GenerateENO := "TRUE" } Move(in := "DB301_Velocidad_FSS".carga.Lenta, out1 => #MA_VelocidadAnalogica)
   END_RUNG
   RUNG wire#w1
      I_Contact( #EstadoZona.Manual_CBx )
      I_Contact( #STAT_Velocidad_TxB1 )
      I_Contact( #STAT_Velocidad_TxBO )
      { S7_GenerateENO := "TRUE" } Move(in := "DB301_Velocidad_FSS".carga.Posicionado, out1 => #MA_VelocidadAnalogica)
   END_RUNG
   // the same network as SCL:
   // ENO of a box is taken as its EN; it also drops when the box reports an error
   IF "ON" THEN #MA_VelocidadAnalogica := "DB301_Velocidad_FSS".carga.Posicionado; END_IF;
   IF "ON" AND NOT #EstadoZona.Manual_CBx AND #STAT_Velocidad_TxB1 AND #STAT_Velocidad_TxBO THEN
       #MA_VelocidadAnalogica := "DB301_Velocidad_FSS".carga.Rapida;
   END_IF;
   IF "ON" AND NOT #EstadoZona.Manual_CBx AND #STAT_Velocidad_TxB1 AND NOT #STAT_Velocidad_TxBO THEN
       #MA_VelocidadAnalogica := "DB301_Velocidad_FSS".carga.Media;
   END_IF;
   IF "ON" AND NOT #EstadoZona.Manual_CBx AND NOT #STAT_Velocidad_TxB1 AND #STAT_Velocidad_TxBO THEN
       #MA_VelocidadAnalogica := "DB301_Velocidad_FSS".carga.Lenta;
   END_IF;
   IF "ON" AND NOT #EstadoZona.Manual_CBx AND NOT #STAT_Velocidad_TxB1 AND NOT #STAT_Velocidad_TxBO THEN
       #MA_VelocidadAnalogica := "DB301_Velocidad_FSS".carga.Posicionado;
   END_IF;
END_REGION

REGION Network 113: SALIDAS - Avance_TR1 >> CADENAS
   RUNG wire#powerrail
      Contact( #STAT_AvanceCarga )
      I_Contact( #Activado_Pasarela )
      wire#w1
      Coil( #MA_Avance_TR1 )
   END_RUNG
   RUNG wire#powerrail
      Contact( #STAT_AvancePasarela )
      Contact( #Activado_Pasarela )
   END_RUNG wire#w1
   // the same network as SCL:
   #MA_Avance_TR1 := (#STAT_AvanceCarga AND NOT #Activado_Pasarela) OR (#STAT_AvancePasarela AND #Activado_Pasarela);
END_REGION

REGION Network 114: SALIDAS - Avance_TR2 >> CADENAS
   RUNG wire#powerrail
      Contact( #Entrando_BGrande )
      I_Contact( #Activado_Pasarela )
      wire#w1
      Contact( #MA_Avance_TR1 )
      Coil( #MA_Avance_TR2 )
   END_RUNG
   RUNG wire#powerrail
      Contact( #AVTF_MAnt_MSig_BGrande )
      Contact( #Activado_Pasarela )
   END_RUNG wire#w1
   // the same network as SCL:
   #MA_Avance_TR2 := ((#Entrando_BGrande AND NOT #Activado_Pasarela) OR (#AVTF_MAnt_MSig_BGrande AND #Activado_Pasarela)) AND #MA_Avance_TR1;
END_REGION

REGION Network 115: SALIDAS - VELOCIDAD LENTA >> CADENAS
   RUNG wire#powerrail
      Contact( #Mx_ET10 )
      wire#w1
      Contact( #CNTSeg_pHsMx.QU )
      wire#w2
      Coil( #MA_VelocidaLenta_TRx )
   END_RUNG
   RUNG wire#powerrail
      Contact( #Mx_ET16 )
   END_RUNG wire#w1
   RUNG wire#powerrail
      Contact( #Mx_ET17 )
   END_RUNG wire#w1
   RUNG wire#powerrail
      Contact( #Mx_ET02 )
   END_RUNG wire#w1
   RUNG wire#powerrail
      Contact( #Mx_ET11 )
   END_RUNG wire#w2
   RUNG wire#powerrail
      Contact( #Mx_ET12 )
   END_RUNG wire#w2
   // the same network as SCL:
   #MA_VelocidaLenta_TRx := ((#Mx_ET10 OR #Mx_ET16 OR #Mx_ET17 OR #Mx_ET02) AND #CNTSeg_pHsMx.QU) OR #Mx_ET11 OR #Mx_ET12;
END_REGION

REGION Network 116: SALIDAS - SUBIR TRANSTER TR1 (Neumatica)
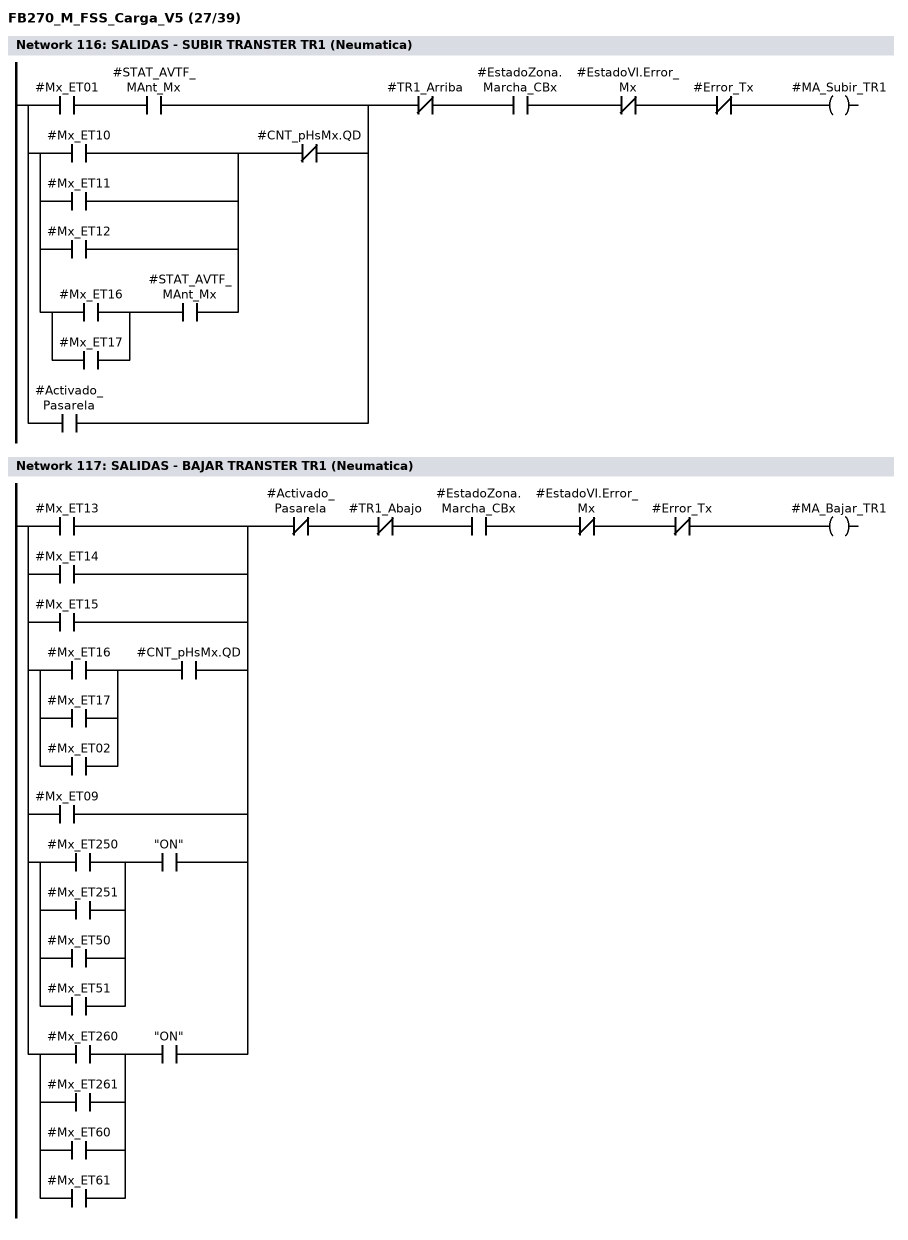
   RUNG wire#powerrail
      Contact( #Mx_ET01 )
      Contact( #STAT_AVTF_MAnt_Mx )
      wire#w1
      I_Contact( #TR1_Arriba )
      Contact( #EstadoZona.Marcha_CBx )
      I_Contact( #EstadoVI.Error_Mx )
      I_Contact( #Error_Tx )
      Coil( #MA_Subir_TR1 )
   END_RUNG
   RUNG wire#powerrail
      Contact( #Mx_ET10 )
      wire#w2
      I_Contact( #CNT_pHsMx.QD )
   END_RUNG wire#w1
   RUNG wire#powerrail
      Contact( #Mx_ET11 )
   END_RUNG wire#w2
   RUNG wire#powerrail
      Contact( #Mx_ET12 )
   END_RUNG wire#w2
   RUNG wire#powerrail
      Contact( #Mx_ET16 )
      wire#w3
      Contact( #STAT_AVTF_MAnt_Mx )
   END_RUNG wire#w2
   RUNG wire#powerrail
      Contact( #Mx_ET17 )
   END_RUNG wire#w3
   RUNG wire#powerrail
      Contact( #Activado_Pasarela )
   END_RUNG wire#w1
   // the same network as SCL:
   #MA_Subir_TR1 := ((#Mx_ET01 AND #STAT_AVTF_MAnt_Mx) OR ((#Mx_ET10 OR #Mx_ET11 OR #Mx_ET12 OR ((#Mx_ET16 OR #Mx_ET17) AND #STAT_AVTF_MAnt_Mx)) AND NOT #CNT_pHsMx.QD) OR #Activado_Pasarela) AND NOT #TR1_Arriba AND #EstadoZona.Marcha_CBx AND NOT #EstadoVI.Error_Mx AND NOT #Error_Tx;
END_REGION

REGION Network 117: SALIDAS - BAJAR TRANSTER TR1 (Neumatica)
   RUNG wire#powerrail
      Contact( #Mx_ET13 )
      wire#w1
      I_Contact( #Activado_Pasarela )
      I_Contact( #TR1_Abajo )
      Contact( #EstadoZona.Marcha_CBx )
      I_Contact( #EstadoVI.Error_Mx )
      I_Contact( #Error_Tx )
      Coil( #MA_Bajar_TR1 )
   END_RUNG
   RUNG wire#powerrail
      Contact( #Mx_ET14 )
   END_RUNG wire#w1
   RUNG wire#powerrail
      Contact( #Mx_ET15 )
   END_RUNG wire#w1
   RUNG wire#powerrail
      Contact( #Mx_ET16 )
      wire#w2
      Contact( #CNT_pHsMx.QD )
   END_RUNG wire#w1
   RUNG wire#powerrail
      Contact( #Mx_ET17 )
   END_RUNG wire#w2
   RUNG wire#powerrail
      Contact( #Mx_ET02 )
   END_RUNG wire#w2
   RUNG wire#powerrail
      Contact( #Mx_ET09 )
   END_RUNG wire#w1
   RUNG wire#powerrail
      Contact( #Mx_ET250 )
      wire#w3
      Contact( "ON" )
   END_RUNG wire#w1
   RUNG wire#powerrail
      Contact( #Mx_ET251 )
   END_RUNG wire#w3
   RUNG wire#powerrail
      Contact( #Mx_ET50 )
   END_RUNG wire#w3
   RUNG wire#powerrail
      Contact( #Mx_ET51 )
   END_RUNG wire#w3
   RUNG wire#powerrail
      Contact( #Mx_ET260 )
      wire#w4
      Contact( "ON" )
   END_RUNG wire#w1
   RUNG wire#powerrail
      Contact( #Mx_ET261 )
   END_RUNG wire#w4
   RUNG wire#powerrail
      Contact( #Mx_ET60 )
   END_RUNG wire#w4
   RUNG wire#powerrail
      Contact( #Mx_ET61 )
   END_RUNG wire#w4
   // the same network as SCL:
   #MA_Bajar_TR1 := (#Mx_ET13 OR #Mx_ET14 OR #Mx_ET15 OR ((#Mx_ET16 OR #Mx_ET17 OR #Mx_ET02) AND #CNT_pHsMx.QD) OR #Mx_ET09 OR ((#Mx_ET250 OR #Mx_ET251 OR #Mx_ET50 OR #Mx_ET51) AND "ON") OR ((#Mx_ET260 OR #Mx_ET261 OR #Mx_ET60 OR #Mx_ET61) AND "ON")) AND NOT #Activado_Pasarela AND NOT #TR1_Abajo AND #EstadoZona.Marcha_CBx AND NOT #EstadoVI.Error_Mx AND NOT #Error_Tx;
END_REGION

REGION Network 118: SALIDAS - SUBIR TRANSTER TR2 (Neumatica)
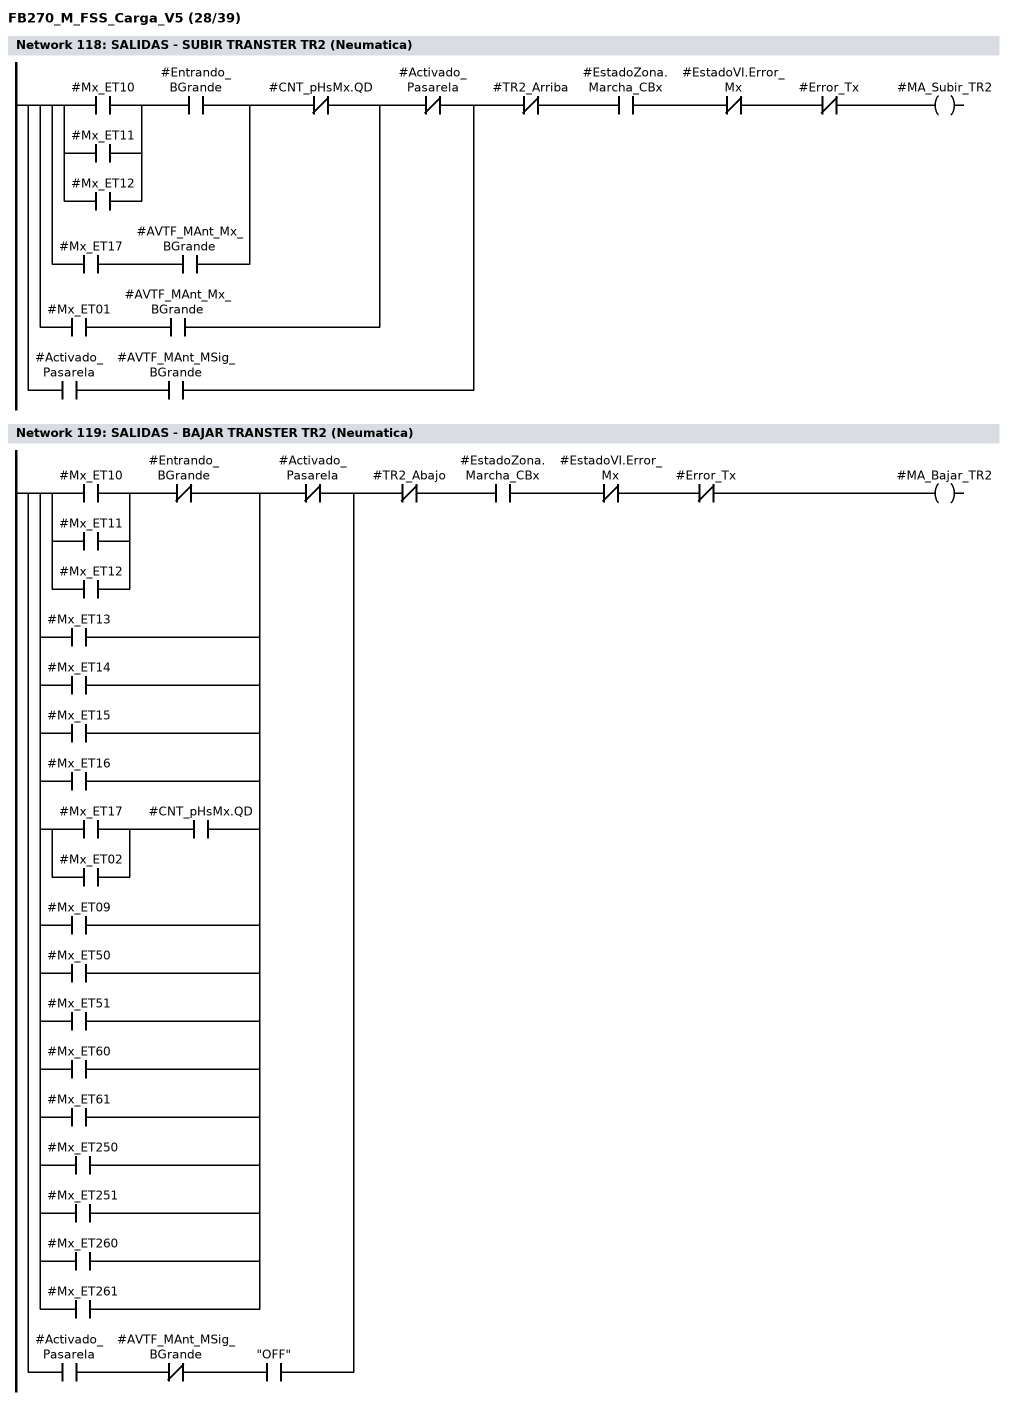
   RUNG wire#powerrail
      Contact( #Mx_ET10 )
      wire#w1
      Contact( #Entrando_BGrande )
      wire#w2
      I_Contact( #CNT_pHsMx.QD )
      wire#w3
      I_Contact( #Activado_Pasarela )
      wire#w4
      I_Contact( #TR2_Arriba )
      Contact( #EstadoZona.Marcha_CBx )
      I_Contact( #EstadoVI.Error_Mx )
      I_Contact( #Error_Tx )
      Coil( #MA_Subir_TR2 )
   END_RUNG
   RUNG wire#powerrail
      Contact( #Mx_ET11 )
   END_RUNG wire#w1
   RUNG wire#powerrail
      Contact( #Mx_ET12 )
   END_RUNG wire#w1
   RUNG wire#powerrail
      Contact( #Mx_ET17 )
      Contact( #AVTF_MAnt_Mx_BGrande )
   END_RUNG wire#w2
   RUNG wire#powerrail
      Contact( #Mx_ET01 )
      Contact( #AVTF_MAnt_Mx_BGrande )
   END_RUNG wire#w3
   RUNG wire#powerrail
      Contact( #Activado_Pasarela )
      Contact( #AVTF_MAnt_MSig_BGrande )
   END_RUNG wire#w4
   // the same network as SCL:
   #MA_Subir_TR2 := (((((((#Mx_ET10 OR #Mx_ET11 OR #Mx_ET12) AND #Entrando_BGrande) OR (#Mx_ET17 AND #AVTF_MAnt_Mx_BGrande)) AND NOT #CNT_pHsMx.QD) OR (#Mx_ET01 AND #AVTF_MAnt_Mx_BGrande)) AND NOT #Activado_Pasarela) OR (#Activado_Pasarela AND #AVTF_MAnt_MSig_BGrande)) AND NOT #TR2_Arriba AND #EstadoZona.Marcha_CBx AND NOT #EstadoVI.Error_Mx AND NOT #Error_Tx;
END_REGION

REGION Network 119: SALIDAS - BAJAR TRANSTER TR2 (Neumatica)
   RUNG wire#powerrail
      Contact( #Mx_ET10 )
      wire#w1
      I_Contact( #Entrando_BGrande )
      wire#w2
      I_Contact( #Activado_Pasarela )
      wire#w4
      I_Contact( #TR2_Abajo )
      Contact( #EstadoZona.Marcha_CBx )
      I_Contact( #EstadoVI.Error_Mx )
      I_Contact( #Error_Tx )
      Coil( #MA_Bajar_TR2 )
   END_RUNG
   RUNG wire#powerrail
      Contact( #Mx_ET11 )
   END_RUNG wire#w1
   RUNG wire#powerrail
      Contact( #Mx_ET12 )
   END_RUNG wire#w1
   RUNG wire#powerrail
      Contact( #Mx_ET13 )
   END_RUNG wire#w2
   RUNG wire#powerrail
      Contact( #Mx_ET14 )
   END_RUNG wire#w2
   RUNG wire#powerrail
      Contact( #Mx_ET15 )
   END_RUNG wire#w2
   RUNG wire#powerrail
      Contact( #Mx_ET16 )
   END_RUNG wire#w2
   RUNG wire#powerrail
      Contact( #Mx_ET17 )
      wire#w3
      Contact( #CNT_pHsMx.QD )
   END_RUNG wire#w2
   RUNG wire#powerrail
      Contact( #Mx_ET02 )
   END_RUNG wire#w3
   RUNG wire#powerrail
      Contact( #Mx_ET09 )
   END_RUNG wire#w2
   RUNG wire#powerrail
      Contact( #Mx_ET50 )
   END_RUNG wire#w2
   RUNG wire#powerrail
      Contact( #Mx_ET51 )
   END_RUNG wire#w2
   RUNG wire#powerrail
      Contact( #Mx_ET60 )
   END_RUNG wire#w2
   RUNG wire#powerrail
      Contact( #Mx_ET61 )
   END_RUNG wire#w2
   RUNG wire#powerrail
      Contact( #Mx_ET250 )
   END_RUNG wire#w2
   RUNG wire#powerrail
      Contact( #Mx_ET251 )
   END_RUNG wire#w2
   RUNG wire#powerrail
      Contact( #Mx_ET260 )
   END_RUNG wire#w2
   RUNG wire#powerrail
      Contact( #Mx_ET261 )
   END_RUNG wire#w2
   RUNG wire#powerrail
      Contact( #Activado_Pasarela )
      I_Contact( #AVTF_MAnt_MSig_BGrande )
      Contact( "OFF" )
   END_RUNG wire#w4
   // the same network as SCL:
   #MA_Bajar_TR2 := (((((#Mx_ET10 OR #Mx_ET11 OR #Mx_ET12) AND NOT #Entrando_BGrande) OR #Mx_ET13 OR #Mx_ET14 OR #Mx_ET15 OR #Mx_ET16 OR ((#Mx_ET17 OR #Mx_ET02) AND #CNT_pHsMx.QD) OR #Mx_ET09 OR #Mx_ET50 OR #Mx_ET51 OR #Mx_ET60 OR #Mx_ET61 OR #Mx_ET250 OR #Mx_ET251 OR #Mx_ET260 OR #Mx_ET261) AND NOT #Activado_Pasarela) OR (#Activado_Pasarela AND NOT #AVTF_MAnt_MSig_BGrande AND "OFF")) AND NOT #TR2_Abajo AND #EstadoZona.Marcha_CBx AND NOT #EstadoVI.Error_Mx AND NOT #Error_Tx;
END_REGION

REGION Network 120: TMP - Espera En Tension
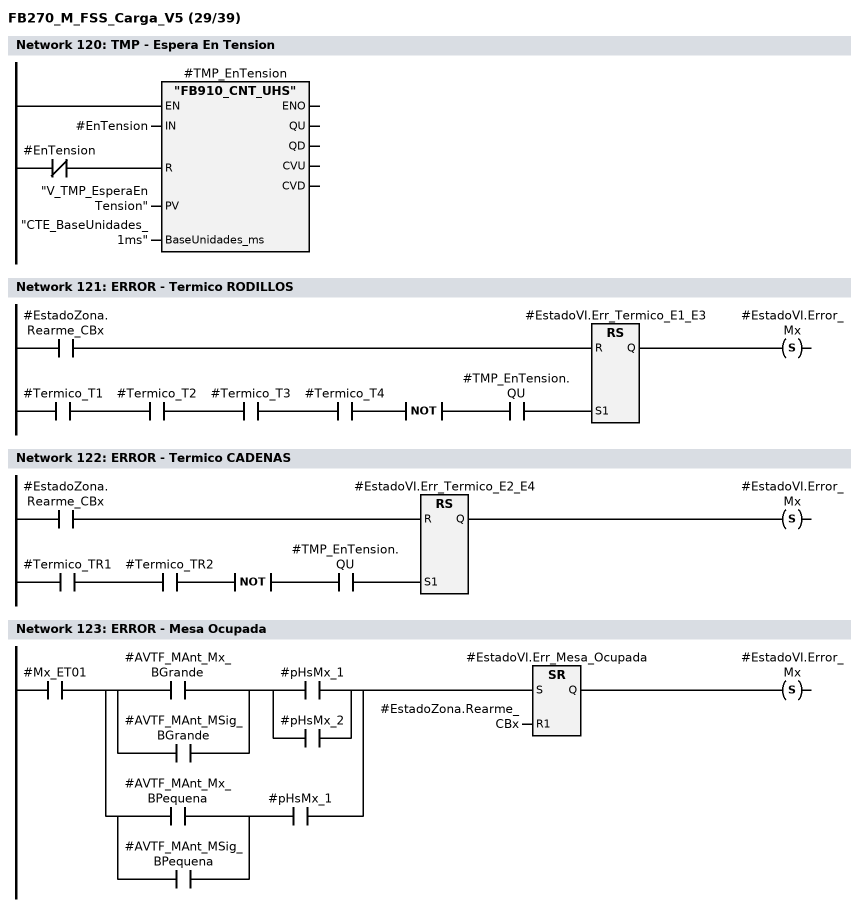
   RUNG wire#powerrail
      #TMP_EnTension(R := wire#w1, IN := #EnTension, PV := "V_TMP_EsperaEnTension", BaseUnidades_ms := "CTE_BaseUnidades_1ms", QU =>, QD =>, CVU =>, CVD =>)
   END_RUNG
   RUNG wire#powerrail
      I_Contact( #EnTension )
   END_RUNG wire#w1
   // the same network as SCL:
   #TMP_EnTension(IN := #EnTension,   // "FB910_CNT_UHS"
                  R := NOT #EnTension,
                  PV := "V_TMP_EsperaEnTension",
                  BaseUnidades_ms := "CTE_BaseUnidades_1ms");
END_REGION

REGION Network 121: ERROR - Termico RODILLOS
   RUNG wire#powerrail
      Contact( #EstadoZona.Rearme_CBx )
      S_RS(operand := #EstadoVI.Err_Termico_E1_E3, s1 := wire#w1)
      S_Coil( #EstadoVI.Error_Mx )
   END_RUNG
   RUNG wire#powerrail
      Contact( #Termico_T1 )
      Contact( #Termico_T2 )
      Contact( #Termico_T3 )
      Contact( #Termico_T4 )
      Not()
      Contact( #TMP_EnTension.QU )
   END_RUNG wire#w1
   // the same network as SCL:
   IF #EstadoZona.Rearme_CBx THEN
       #EstadoVI.Err_Termico_E1_E3 := FALSE;   // RS flip-flop
   END_IF;
   IF NOT (#Termico_T1 AND #Termico_T2 AND #Termico_T3 AND #Termico_T4) AND #TMP_EnTension.QU THEN
       #EstadoVI.Err_Termico_E1_E3 := TRUE;
   END_IF;
   IF #EstadoVI.Err_Termico_E1_E3 THEN #EstadoVI.Error_Mx := TRUE; END_IF;
END_REGION

REGION Network 122: ERROR - Termico CADENAS
   RUNG wire#powerrail
      Contact( #EstadoZona.Rearme_CBx )
      S_RS(operand := #EstadoVI.Err_Termico_E2_E4, s1 := wire#w1)
      S_Coil( #EstadoVI.Error_Mx )
   END_RUNG
   RUNG wire#powerrail
      Contact( #Termico_TR1 )
      Contact( #Termico_TR2 )
      Not()
      Contact( #TMP_EnTension.QU )
   END_RUNG wire#w1
   // the same network as SCL:
   IF #EstadoZona.Rearme_CBx THEN
       #EstadoVI.Err_Termico_E2_E4 := FALSE;   // RS flip-flop
   END_IF;
   IF NOT (#Termico_TR1 AND #Termico_TR2) AND #TMP_EnTension.QU THEN
       #EstadoVI.Err_Termico_E2_E4 := TRUE;
   END_IF;
   IF #EstadoVI.Err_Termico_E2_E4 THEN #EstadoVI.Error_Mx := TRUE; END_IF;
END_REGION

REGION Network 123: ERROR - Mesa Ocupada
   RUNG wire#powerrail
      Contact( #Mx_ET01 )
      wire#w1
      Contact( #AVTF_MAnt_Mx_BGrande )
      wire#w2
      Contact( #pHsMx_1 )
      wire#w3
      S_SR(operand := #EstadoVI.Err_Mesa_Ocupada, r1 := #EstadoZona.Rearme_CBx)
      S_Coil( #EstadoVI.Error_Mx )
   END_RUNG
   RUNG wire#w1
      Contact( #AVTF_MAnt_MSig_BGrande )
   END_RUNG wire#w2
   RUNG wire#w2
      Contact( #pHsMx_2 )
   END_RUNG wire#w3
   RUNG wire#w1
      Contact( #AVTF_MAnt_Mx_BPequena )
      wire#w4
      Contact( #pHsMx_1 )
   END_RUNG wire#w3
   RUNG wire#w1
      Contact( #AVTF_MAnt_MSig_BPequena )
   END_RUNG wire#w4
   // the same network as SCL:
   IF #Mx_ET01 AND (((#AVTF_MAnt_Mx_BGrande OR #AVTF_MAnt_MSig_BGrande) AND (#pHsMx_1 OR #pHsMx_2)) OR ((#AVTF_MAnt_Mx_BPequena OR #AVTF_MAnt_MSig_BPequena) AND #pHsMx_1)) THEN
       #EstadoVI.Err_Mesa_Ocupada := TRUE;   // SR flip-flop
   END_IF;
   IF #EstadoZona.Rearme_CBx THEN #EstadoVI.Err_Mesa_Ocupada := FALSE; END_IF;
   IF #EstadoVI.Err_Mesa_Ocupada THEN #EstadoVI.Error_Mx := TRUE; END_IF;
END_REGION

REGION Network 124: CNT - ERROR - Arrastre
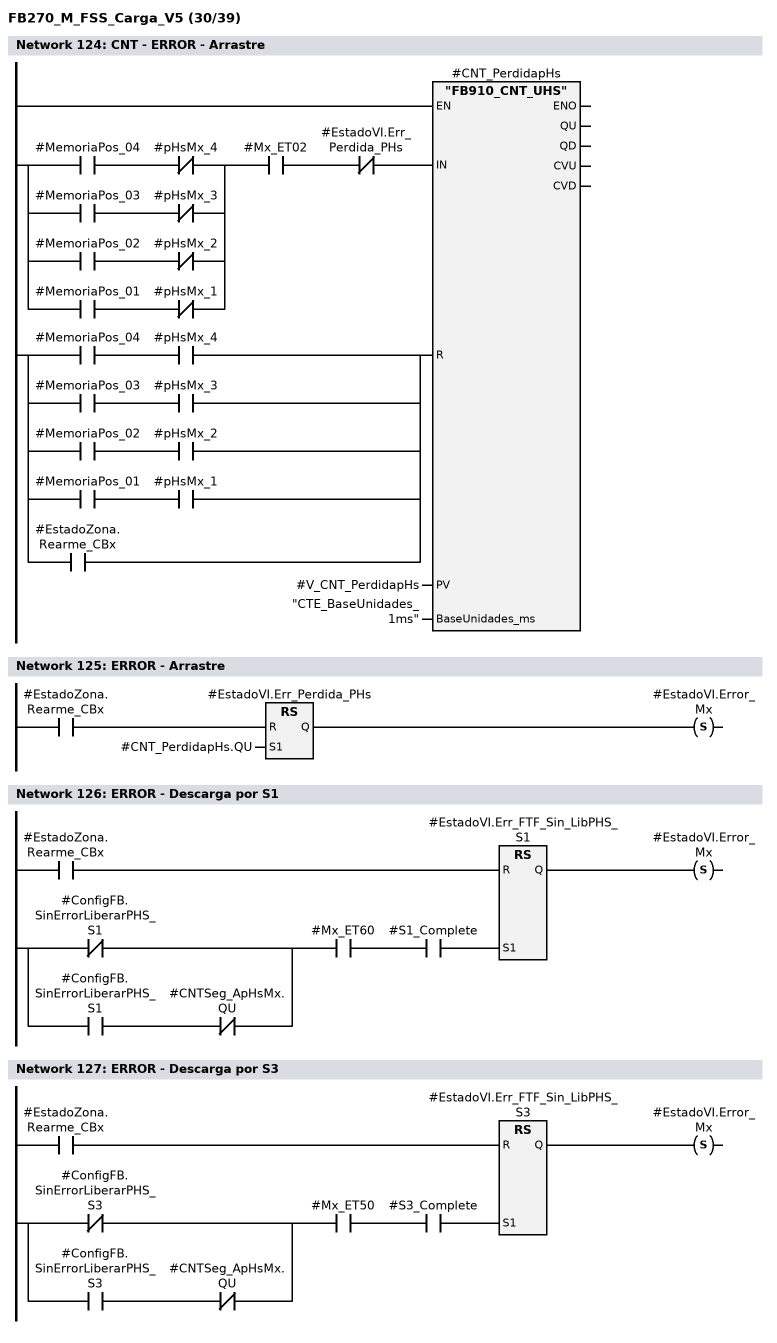
   RUNG wire#powerrail
      #CNT_PerdidapHs(IN := wire#w2, R := wire#w3, PV := #V_CNT_PerdidapHs, BaseUnidades_ms := "CTE_BaseUnidades_1ms", QU =>, QD =>, CVU =>, CVD =>)
   END_RUNG
   RUNG wire#powerrail
      Contact( #MemoriaPos_04 )
      I_Contact( #pHsMx_4 )
      wire#w1
      Contact( #Mx_ET02 )
      I_Contact( #EstadoVI.Err_Perdida_PHs )
   END_RUNG wire#w2
   RUNG wire#powerrail
      Contact( #MemoriaPos_03 )
      I_Contact( #pHsMx_3 )
   END_RUNG wire#w1
   RUNG wire#powerrail
      Contact( #MemoriaPos_02 )
      I_Contact( #pHsMx_2 )
   END_RUNG wire#w1
   RUNG wire#powerrail
      Contact( #MemoriaPos_01 )
      I_Contact( #pHsMx_1 )
   END_RUNG wire#w1
   RUNG wire#powerrail
      Contact( #MemoriaPos_04 )
      Contact( #pHsMx_4 )
   END_RUNG wire#w3
   RUNG wire#powerrail
      Contact( #MemoriaPos_03 )
      Contact( #pHsMx_3 )
   END_RUNG wire#w3
   RUNG wire#powerrail
      Contact( #MemoriaPos_02 )
      Contact( #pHsMx_2 )
   END_RUNG wire#w3
   RUNG wire#powerrail
      Contact( #MemoriaPos_01 )
      Contact( #pHsMx_1 )
   END_RUNG wire#w3
   RUNG wire#powerrail
      Contact( #EstadoZona.Rearme_CBx )
   END_RUNG wire#w3
   // the same network as SCL:
   #CNT_PerdidapHs(IN := ((#MemoriaPos_04 AND NOT #pHsMx_4) OR (#MemoriaPos_03 AND NOT #pHsMx_3) OR (#MemoriaPos_02 AND NOT #pHsMx_2) OR (#MemoriaPos_01 AND NOT #pHsMx_1)) AND #Mx_ET02 AND NOT #EstadoVI.Err_Perdida_PHs,   // "FB910_CNT_UHS"
                   R := (#MemoriaPos_04 AND #pHsMx_4) OR (#MemoriaPos_03 AND #pHsMx_3) OR (#MemoriaPos_02 AND #pHsMx_2) OR (#MemoriaPos_01 AND #pHsMx_1) OR #EstadoZona.Rearme_CBx,
                   PV := #V_CNT_PerdidapHs,
                   BaseUnidades_ms := "CTE_BaseUnidades_1ms");
END_REGION

REGION Network 125: ERROR - Arrastre
   RUNG wire#powerrail
      Contact( #EstadoZona.Rearme_CBx )
      S_RS(operand := #EstadoVI.Err_Perdida_PHs, s1 := #CNT_PerdidapHs.QU)
      S_Coil( #EstadoVI.Error_Mx )
   END_RUNG
   // the same network as SCL:
   IF #EstadoZona.Rearme_CBx THEN
       #EstadoVI.Err_Perdida_PHs := FALSE;   // RS flip-flop
   END_IF;
   IF #CNT_PerdidapHs.QU THEN #EstadoVI.Err_Perdida_PHs := TRUE; END_IF;
   IF #EstadoVI.Err_Perdida_PHs THEN #EstadoVI.Error_Mx := TRUE; END_IF;
END_REGION

REGION Network 126: ERROR - Descarga por S1
   RUNG wire#powerrail
      Contact( #EstadoZona.Rearme_CBx )
      S_RS(operand := #EstadoVI.Err_FTF_Sin_LibPHS_S1, s1 := wire#w2)
      S_Coil( #EstadoVI.Error_Mx )
   END_RUNG
   RUNG wire#powerrail
      I_Contact( #ConfigFB.SinErrorLiberarPHS_S1 )
      wire#w1
      Contact( #Mx_ET60 )
      Contact( #S1_Complete )
   END_RUNG wire#w2
   RUNG wire#powerrail
      Contact( #ConfigFB.SinErrorLiberarPHS_S1 )
      I_Contact( #CNTSeg_ApHsMx.QU )
   END_RUNG wire#w1
   // the same network as SCL:
   IF #EstadoZona.Rearme_CBx THEN
       #EstadoVI.Err_FTF_Sin_LibPHS_S1 := FALSE;   // RS flip-flop
   END_IF;
   IF (NOT #ConfigFB.SinErrorLiberarPHS_S1 OR (#ConfigFB.SinErrorLiberarPHS_S1 AND NOT #CNTSeg_ApHsMx.QU)) AND #Mx_ET60 AND #S1_Complete THEN
       #EstadoVI.Err_FTF_Sin_LibPHS_S1 := TRUE;
   END_IF;
   IF #EstadoVI.Err_FTF_Sin_LibPHS_S1 THEN #EstadoVI.Error_Mx := TRUE; END_IF;
END_REGION

REGION Network 127: ERROR - Descarga por S3
   RUNG wire#powerrail
      Contact( #EstadoZona.Rearme_CBx )
      S_RS(operand := #EstadoVI.Err_FTF_Sin_LibPHS_S3, s1 := wire#w2)
      S_Coil( #EstadoVI.Error_Mx )
   END_RUNG
   RUNG wire#powerrail
      I_Contact( #ConfigFB.SinErrorLiberarPHS_S3 )
      wire#w1
      Contact( #Mx_ET50 )
      Contact( #S3_Complete )
   END_RUNG wire#w2
   RUNG wire#powerrail
      Contact( #ConfigFB.SinErrorLiberarPHS_S3 )
      I_Contact( #CNTSeg_ApHsMx.QU )
   END_RUNG wire#w1
   // the same network as SCL:
   IF #EstadoZona.Rearme_CBx THEN
       #EstadoVI.Err_FTF_Sin_LibPHS_S3 := FALSE;   // RS flip-flop
   END_IF;
   IF (NOT #ConfigFB.SinErrorLiberarPHS_S3 OR (#ConfigFB.SinErrorLiberarPHS_S3 AND NOT #CNTSeg_ApHsMx.QU)) AND #Mx_ET50 AND #S3_Complete THEN
       #EstadoVI.Err_FTF_Sin_LibPHS_S3 := TRUE;
   END_IF;
   IF #EstadoVI.Err_FTF_Sin_LibPHS_S3 THEN #EstadoVI.Error_Mx := TRUE; END_IF;
END_REGION

REGION Network 128: TMP - ERROR - TimeOut Avance TRx >>> ENTRADA
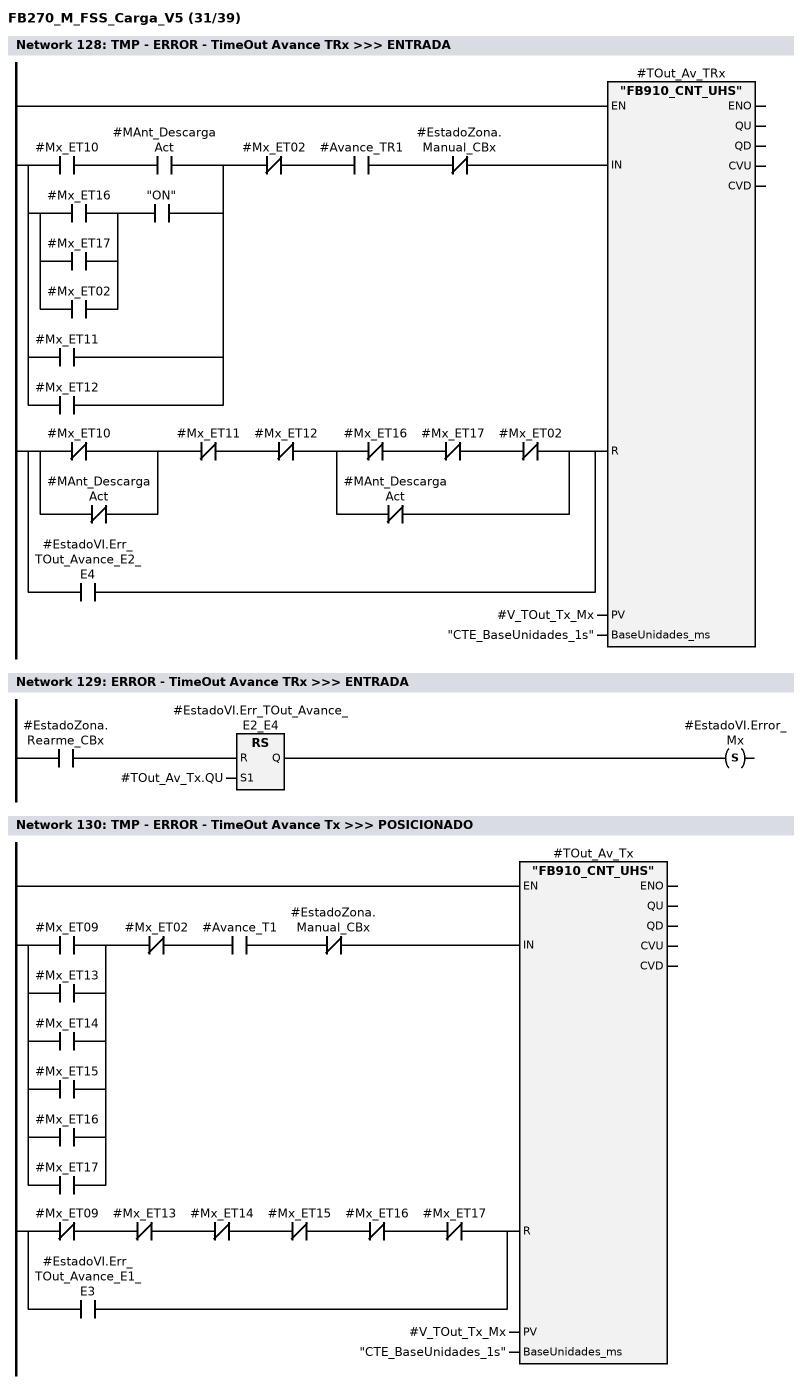
   RUNG wire#powerrail
      #TOut_Av_TRx(IN := wire#w3, R := wire#w6, PV := #V_TOut_Tx_Mx, BaseUnidades_ms := "CTE_BaseUnidades_1s", QU =>, QD =>, CVU =>, CVD =>)
   END_RUNG
   RUNG wire#powerrail
      Contact( #Mx_ET10 )
      Contact( #MAnt_DescargaAct )
      wire#w1
      I_Contact( #Mx_ET02 )
      Contact( #Avance_TR1 )
      I_Contact( #EstadoZona.Manual_CBx )
   END_RUNG wire#w3
   RUNG wire#powerrail
      Contact( #Mx_ET16 )
      wire#w2
      Contact( "ON" )
   END_RUNG wire#w1
   RUNG wire#powerrail
      Contact( #Mx_ET17 )
   END_RUNG wire#w2
   RUNG wire#powerrail
      Contact( #Mx_ET02 )
   END_RUNG wire#w2
   RUNG wire#powerrail
      Contact( #Mx_ET11 )
   END_RUNG wire#w1
   RUNG wire#powerrail
      Contact( #Mx_ET12 )
   END_RUNG wire#w1
   RUNG wire#powerrail
      I_Contact( #Mx_ET10 )
      wire#w4
      I_Contact( #Mx_ET11 )
      I_Contact( #Mx_ET12 )
      wire#w5
      I_Contact( #Mx_ET16 )
      I_Contact( #Mx_ET17 )
      I_Contact( #Mx_ET02 )
   END_RUNG wire#w6
   RUNG wire#powerrail
      I_Contact( #MAnt_DescargaAct )
   END_RUNG wire#w4
   RUNG wire#w5
      I_Contact( #MAnt_DescargaAct )
   END_RUNG wire#w6
   RUNG wire#powerrail
      Contact( #EstadoVI.Err_TOut_Avance_E2_E4 )
   END_RUNG wire#w6
   // the same network as SCL:
   #TOut_Av_TRx(IN := ((#Mx_ET10 AND #MAnt_DescargaAct) OR ((#Mx_ET16 OR #Mx_ET17 OR #Mx_ET02) AND "ON") OR #Mx_ET11 OR #Mx_ET12) AND NOT #Mx_ET02 AND #Avance_TR1 AND NOT #EstadoZona.Manual_CBx,   // "FB910_CNT_UHS"
                R := ((NOT #Mx_ET10 OR NOT #MAnt_DescargaAct) AND NOT #Mx_ET11 AND NOT #Mx_ET12 AND ((NOT #Mx_ET16 AND NOT #Mx_ET17 AND NOT #Mx_ET02) OR NOT #MAnt_DescargaAct)) OR #EstadoVI.Err_TOut_Avance_E2_E4,
                PV := #V_TOut_Tx_Mx,
                BaseUnidades_ms := "CTE_BaseUnidades_1s");
END_REGION

REGION Network 129: ERROR - TimeOut Avance TRx >>> ENTRADA
   RUNG wire#powerrail
      Contact( #EstadoZona.Rearme_CBx )
      S_RS(operand := #EstadoVI.Err_TOut_Avance_E2_E4, s1 := #TOut_Av_Tx.QU)
      S_Coil( #EstadoVI.Error_Mx )
   END_RUNG
   // the same network as SCL:
   IF #EstadoZona.Rearme_CBx THEN
       #EstadoVI.Err_TOut_Avance_E2_E4 := FALSE;   // RS flip-flop
   END_IF;
   IF #TOut_Av_Tx.QU THEN #EstadoVI.Err_TOut_Avance_E2_E4 := TRUE; END_IF;
   IF #EstadoVI.Err_TOut_Avance_E2_E4 THEN #EstadoVI.Error_Mx := TRUE; END_IF;
END_REGION

REGION Network 130: TMP - ERROR - TimeOut Avance Tx >>> POSICIONADO
   RUNG wire#powerrail
      #TOut_Av_Tx(IN := wire#w2, R := wire#w3, PV := #V_TOut_Tx_Mx, BaseUnidades_ms := "CTE_BaseUnidades_1s", QU =>, QD =>, CVU =>, CVD =>)
   END_RUNG
   RUNG wire#powerrail
      Contact( #Mx_ET09 )
      wire#w1
      I_Contact( #Mx_ET02 )
      Contact( #Avance_T1 )
      I_Contact( #EstadoZona.Manual_CBx )
   END_RUNG wire#w2
   RUNG wire#powerrail
      Contact( #Mx_ET13 )
   END_RUNG wire#w1
   RUNG wire#powerrail
      Contact( #Mx_ET14 )
   END_RUNG wire#w1
   RUNG wire#powerrail
      Contact( #Mx_ET15 )
   END_RUNG wire#w1
   RUNG wire#powerrail
      Contact( #Mx_ET16 )
   END_RUNG wire#w1
   RUNG wire#powerrail
      Contact( #Mx_ET17 )
   END_RUNG wire#w1
   RUNG wire#powerrail
      I_Contact( #Mx_ET09 )
      I_Contact( #Mx_ET13 )
      I_Contact( #Mx_ET14 )
      I_Contact( #Mx_ET15 )
      I_Contact( #Mx_ET16 )
      I_Contact( #Mx_ET17 )
   END_RUNG wire#w3
   RUNG wire#powerrail
      Contact( #EstadoVI.Err_TOut_Avance_E1_E3 )
   END_RUNG wire#w3
   // the same network as SCL:
   #TOut_Av_Tx(IN := (#Mx_ET09 OR #Mx_ET13 OR #Mx_ET14 OR #Mx_ET15 OR #Mx_ET16 OR #Mx_ET17) AND NOT #Mx_ET02 AND #Avance_T1 AND NOT #EstadoZona.Manual_CBx,   // "FB910_CNT_UHS"
               R := (NOT #Mx_ET09 AND NOT #Mx_ET13 AND NOT #Mx_ET14 AND NOT #Mx_ET15 AND NOT #Mx_ET16 AND NOT #Mx_ET17) OR #EstadoVI.Err_TOut_Avance_E1_E3,
               PV := #V_TOut_Tx_Mx,
               BaseUnidades_ms := "CTE_BaseUnidades_1s");
END_REGION

REGION Network 131: ERROR - TimeOut Avance Tx >>> POSICIONADO
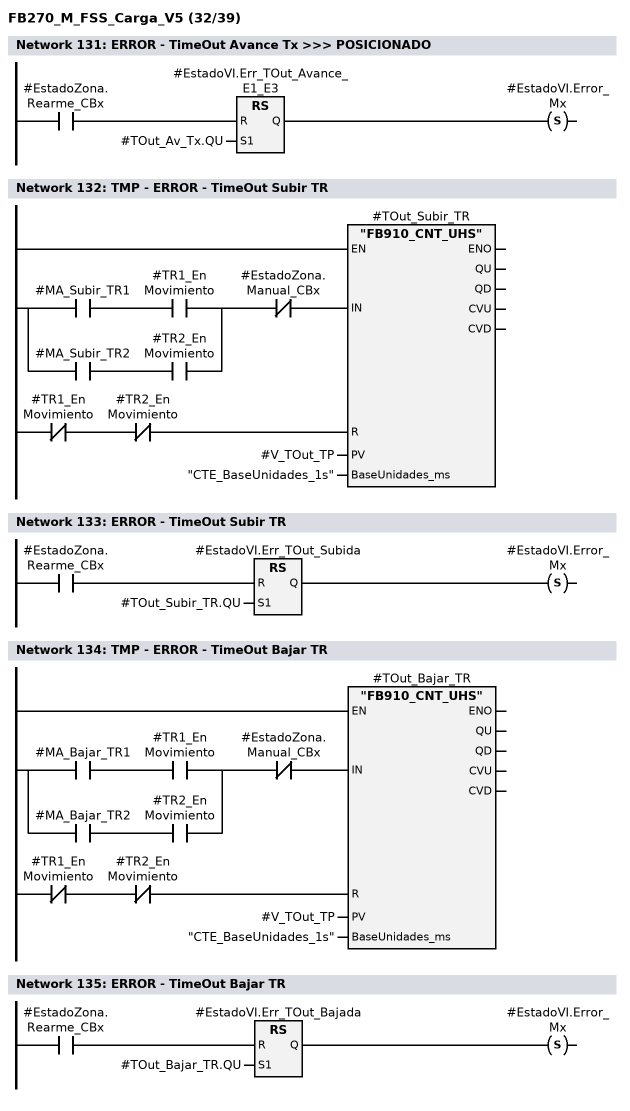
   RUNG wire#powerrail
      Contact( #EstadoZona.Rearme_CBx )
      S_RS(operand := #EstadoVI.Err_TOut_Avance_E1_E3, s1 := #TOut_Av_Tx.QU)
      S_Coil( #EstadoVI.Error_Mx )
   END_RUNG
   // the same network as SCL:
   IF #EstadoZona.Rearme_CBx THEN
       #EstadoVI.Err_TOut_Avance_E1_E3 := FALSE;   // RS flip-flop
   END_IF;
   IF #TOut_Av_Tx.QU THEN #EstadoVI.Err_TOut_Avance_E1_E3 := TRUE; END_IF;
   IF #EstadoVI.Err_TOut_Avance_E1_E3 THEN #EstadoVI.Error_Mx := TRUE; END_IF;
END_REGION

REGION Network 132: TMP - ERROR - TimeOut Subir TR
   RUNG wire#powerrail
      #TOut_Subir_TR(IN := wire#w2, R := wire#w3, PV := #V_TOut_TP, BaseUnidades_ms := "CTE_BaseUnidades_1s", QU =>, QD =>, CVU =>, CVD =>)
   END_RUNG
   RUNG wire#powerrail
      Contact( #MA_Subir_TR1 )
      Contact( #TR1_EnMovimiento )
      wire#w1
      I_Contact( #EstadoZona.Manual_CBx )
   END_RUNG wire#w2
   RUNG wire#powerrail
      Contact( #MA_Subir_TR2 )
      Contact( #TR2_EnMovimiento )
   END_RUNG wire#w1
   RUNG wire#powerrail
      I_Contact( #TR1_EnMovimiento )
      I_Contact( #TR2_EnMovimiento )
   END_RUNG wire#w3
   // the same network as SCL:
   #TOut_Subir_TR(IN := ((#MA_Subir_TR1 AND #TR1_EnMovimiento) OR (#MA_Subir_TR2 AND #TR2_EnMovimiento)) AND NOT #EstadoZona.Manual_CBx,   // "FB910_CNT_UHS"
                  R := NOT #TR1_EnMovimiento AND NOT #TR2_EnMovimiento,
                  PV := #V_TOut_TP,
                  BaseUnidades_ms := "CTE_BaseUnidades_1s");
END_REGION

REGION Network 133: ERROR - TimeOut Subir TR
   RUNG wire#powerrail
      Contact( #EstadoZona.Rearme_CBx )
      S_RS(operand := #EstadoVI.Err_TOut_Subida, s1 := #TOut_Subir_TR.QU)
      S_Coil( #EstadoVI.Error_Mx )
   END_RUNG
   // the same network as SCL:
   IF #EstadoZona.Rearme_CBx THEN
       #EstadoVI.Err_TOut_Subida := FALSE;   // RS flip-flop
   END_IF;
   IF #TOut_Subir_TR.QU THEN #EstadoVI.Err_TOut_Subida := TRUE; END_IF;
   IF #EstadoVI.Err_TOut_Subida THEN #EstadoVI.Error_Mx := TRUE; END_IF;
END_REGION

REGION Network 134: TMP - ERROR - TimeOut Bajar TR
   RUNG wire#powerrail
      #TOut_Bajar_TR(IN := wire#w2, R := wire#w3, PV := #V_TOut_TP, BaseUnidades_ms := "CTE_BaseUnidades_1s", QU =>, QD =>, CVU =>, CVD =>)
   END_RUNG
   RUNG wire#powerrail
      Contact( #MA_Bajar_TR1 )
      Contact( #TR1_EnMovimiento )
      wire#w1
      I_Contact( #EstadoZona.Manual_CBx )
   END_RUNG wire#w2
   RUNG wire#powerrail
      Contact( #MA_Bajar_TR2 )
      Contact( #TR2_EnMovimiento )
   END_RUNG wire#w1
   RUNG wire#powerrail
      I_Contact( #TR1_EnMovimiento )
      I_Contact( #TR2_EnMovimiento )
   END_RUNG wire#w3
   // the same network as SCL:
   #TOut_Bajar_TR(IN := ((#MA_Bajar_TR1 AND #TR1_EnMovimiento) OR (#MA_Bajar_TR2 AND #TR2_EnMovimiento)) AND NOT #EstadoZona.Manual_CBx,   // "FB910_CNT_UHS"
                  R := NOT #TR1_EnMovimiento AND NOT #TR2_EnMovimiento,
                  PV := #V_TOut_TP,
                  BaseUnidades_ms := "CTE_BaseUnidades_1s");
END_REGION

REGION Network 135: ERROR - TimeOut Bajar TR
   RUNG wire#powerrail
      Contact( #EstadoZona.Rearme_CBx )
      S_RS(operand := #EstadoVI.Err_TOut_Bajada, s1 := #TOut_Bajar_TR.QU)
      S_Coil( #EstadoVI.Error_Mx )
   END_RUNG
   // the same network as SCL:
   IF #EstadoZona.Rearme_CBx THEN
       #EstadoVI.Err_TOut_Bajada := FALSE;   // RS flip-flop
   END_IF;
   IF #TOut_Bajar_TR.QU THEN #EstadoVI.Err_TOut_Bajada := TRUE; END_IF;
   IF #EstadoVI.Err_TOut_Bajada THEN #EstadoVI.Error_Mx := TRUE; END_IF;
END_REGION

REGION Network 136: TMP - ERROR - TimeOut Subir TP E1E3
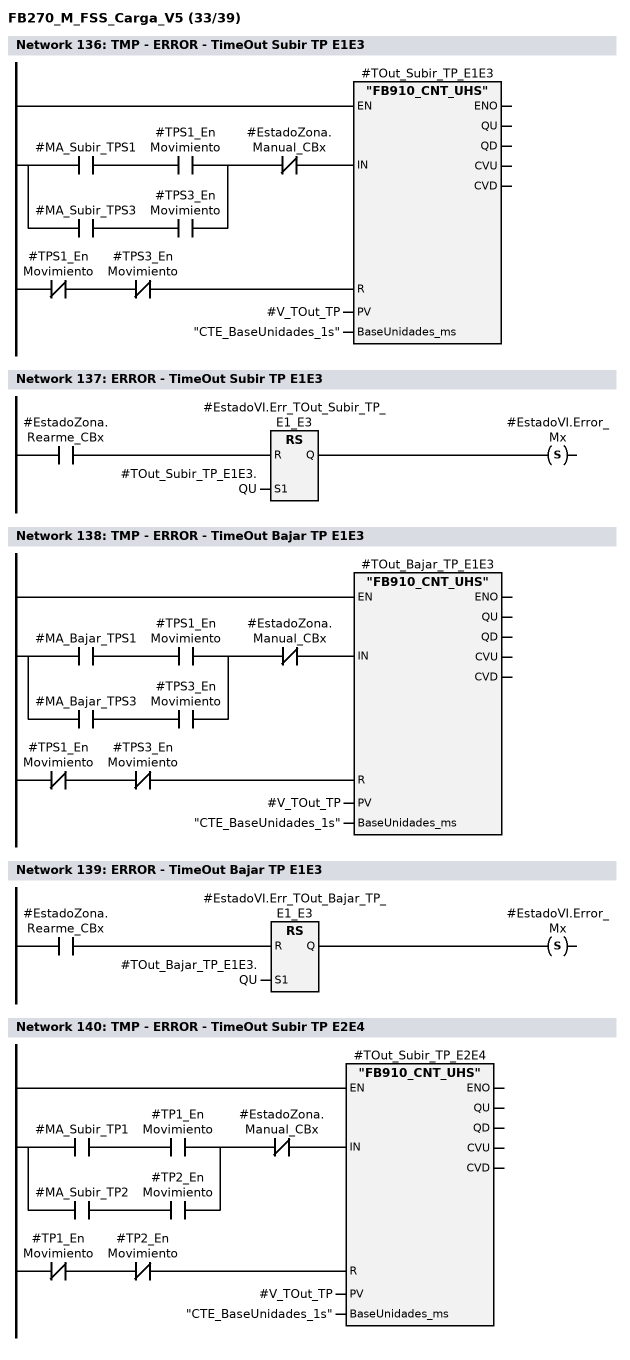
   RUNG wire#powerrail
      #TOut_Subir_TP_E1E3(IN := wire#w2, R := wire#w3, PV := #V_TOut_TP, BaseUnidades_ms := "CTE_BaseUnidades_1s", QU =>, QD =>, CVU =>, CVD =>)
   END_RUNG
   RUNG wire#powerrail
      Contact( #MA_Subir_TPS1 )
      Contact( #TPS1_EnMovimiento )
      wire#w1
      I_Contact( #EstadoZona.Manual_CBx )
   END_RUNG wire#w2
   RUNG wire#powerrail
      Contact( #MA_Subir_TPS3 )
      Contact( #TPS3_EnMovimiento )
   END_RUNG wire#w1
   RUNG wire#powerrail
      I_Contact( #TPS1_EnMovimiento )
      I_Contact( #TPS3_EnMovimiento )
   END_RUNG wire#w3
   // the same network as SCL:
   #TOut_Subir_TP_E1E3(IN := ((#MA_Subir_TPS1 AND #TPS1_EnMovimiento) OR (#MA_Subir_TPS3 AND #TPS3_EnMovimiento)) AND NOT #EstadoZona.Manual_CBx,   // "FB910_CNT_UHS"
                       R := NOT #TPS1_EnMovimiento AND NOT #TPS3_EnMovimiento,
                       PV := #V_TOut_TP,
                       BaseUnidades_ms := "CTE_BaseUnidades_1s");
END_REGION

REGION Network 137: ERROR - TimeOut Subir TP E1E3
   RUNG wire#powerrail
      Contact( #EstadoZona.Rearme_CBx )
      S_RS(operand := #EstadoVI.Err_TOut_Subir_TP_E1_E3, s1 := #TOut_Subir_TP_E1E3.QU)
      S_Coil( #EstadoVI.Error_Mx )
   END_RUNG
   // the same network as SCL:
   IF #EstadoZona.Rearme_CBx THEN
       #EstadoVI.Err_TOut_Subir_TP_E1_E3 := FALSE;   // RS flip-flop
   END_IF;
   IF #TOut_Subir_TP_E1E3.QU THEN #EstadoVI.Err_TOut_Subir_TP_E1_E3 := TRUE; END_IF;
   IF #EstadoVI.Err_TOut_Subir_TP_E1_E3 THEN #EstadoVI.Error_Mx := TRUE; END_IF;
END_REGION

REGION Network 138: TMP - ERROR - TimeOut Bajar TP E1E3
   RUNG wire#powerrail
      #TOut_Bajar_TP_E1E3(IN := wire#w2, R := wire#w3, PV := #V_TOut_TP, BaseUnidades_ms := "CTE_BaseUnidades_1s", QU =>, QD =>, CVU =>, CVD =>)
   END_RUNG
   RUNG wire#powerrail
      Contact( #MA_Bajar_TPS1 )
      Contact( #TPS1_EnMovimiento )
      wire#w1
      I_Contact( #EstadoZona.Manual_CBx )
   END_RUNG wire#w2
   RUNG wire#powerrail
      Contact( #MA_Bajar_TPS3 )
      Contact( #TPS3_EnMovimiento )
   END_RUNG wire#w1
   RUNG wire#powerrail
      I_Contact( #TPS1_EnMovimiento )
      I_Contact( #TPS3_EnMovimiento )
   END_RUNG wire#w3
   // the same network as SCL:
   #TOut_Bajar_TP_E1E3(IN := ((#MA_Bajar_TPS1 AND #TPS1_EnMovimiento) OR (#MA_Bajar_TPS3 AND #TPS3_EnMovimiento)) AND NOT #EstadoZona.Manual_CBx,   // "FB910_CNT_UHS"
                       R := NOT #TPS1_EnMovimiento AND NOT #TPS3_EnMovimiento,
                       PV := #V_TOut_TP,
                       BaseUnidades_ms := "CTE_BaseUnidades_1s");
END_REGION

REGION Network 139: ERROR - TimeOut Bajar TP E1E3
   RUNG wire#powerrail
      Contact( #EstadoZona.Rearme_CBx )
      S_RS(operand := #EstadoVI.Err_TOut_Bajar_TP_E1_E3, s1 := #TOut_Bajar_TP_E1E3.QU)
      S_Coil( #EstadoVI.Error_Mx )
   END_RUNG
   // the same network as SCL:
   IF #EstadoZona.Rearme_CBx THEN
       #EstadoVI.Err_TOut_Bajar_TP_E1_E3 := FALSE;   // RS flip-flop
   END_IF;
   IF #TOut_Bajar_TP_E1E3.QU THEN #EstadoVI.Err_TOut_Bajar_TP_E1_E3 := TRUE; END_IF;
   IF #EstadoVI.Err_TOut_Bajar_TP_E1_E3 THEN #EstadoVI.Error_Mx := TRUE; END_IF;
END_REGION

REGION Network 140: TMP - ERROR - TimeOut Subir TP E2E4
   RUNG wire#powerrail
      #TOut_Subir_TP_E2E4(IN := wire#w2, R := wire#w3, PV := #V_TOut_TP, BaseUnidades_ms := "CTE_BaseUnidades_1s", QU =>, QD =>, CVU =>, CVD =>)
   END_RUNG
   RUNG wire#powerrail
      Contact( #MA_Subir_TP1 )
      Contact( #TP1_EnMovimiento )
      wire#w1
      I_Contact( #EstadoZona.Manual_CBx )
   END_RUNG wire#w2
   RUNG wire#powerrail
      Contact( #MA_Subir_TP2 )
      Contact( #TP2_EnMovimiento )
   END_RUNG wire#w1
   RUNG wire#powerrail
      I_Contact( #TP1_EnMovimiento )
      I_Contact( #TP2_EnMovimiento )
   END_RUNG wire#w3
   // the same network as SCL:
   #TOut_Subir_TP_E2E4(IN := ((#MA_Subir_TP1 AND #TP1_EnMovimiento) OR (#MA_Subir_TP2 AND #TP2_EnMovimiento)) AND NOT #EstadoZona.Manual_CBx,   // "FB910_CNT_UHS"
                       R := NOT #TP1_EnMovimiento AND NOT #TP2_EnMovimiento,
                       PV := #V_TOut_TP,
                       BaseUnidades_ms := "CTE_BaseUnidades_1s");
END_REGION

REGION Network 141: ERROR - TimeOut Subir TP E2E4
